REGION Network 5: Trạng thái cân Ag4
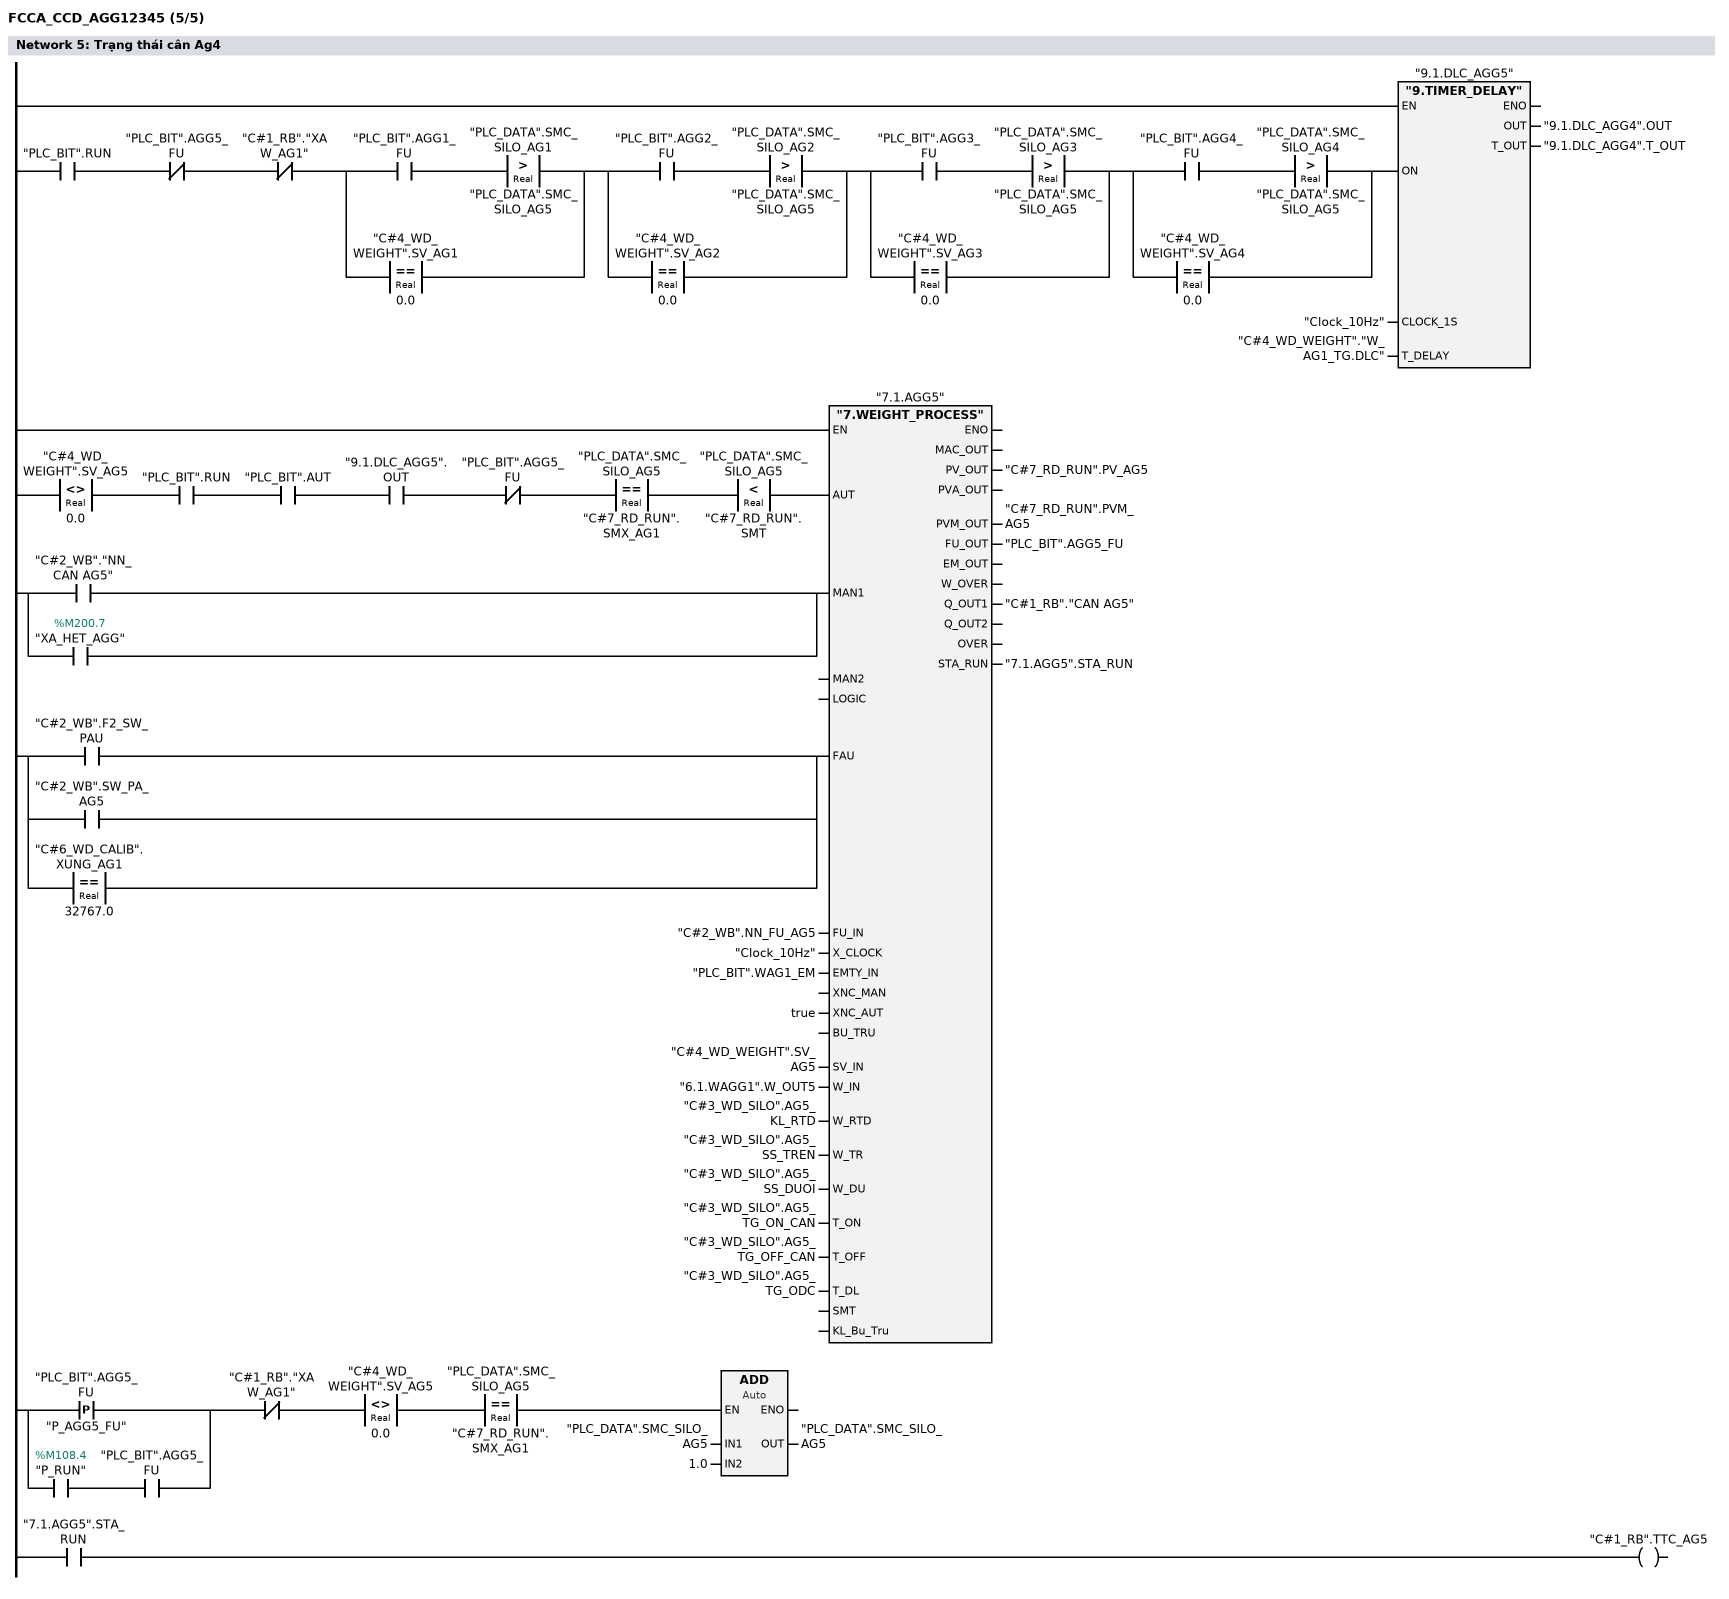
   RUNG wire#powerrail
      "9.1.DLC_AGG5"(ON := wire#w5, CLOCK_1S := "Clock_10Hz", T_DELAY := "C#4_WD_WEIGHT"."W_AG1_TG.DLC", OUT => "9.1.DLC_AGG4".OUT, T_OUT => "9.1.DLC_AGG4".T_OUT)
   END_RUNG
   RUNG wire#powerrail
      Contact( "PLC_BIT".RUN )
      I_Contact( "PLC_BIT".AGG5_FU )
      I_Contact( "C#1_RB"."XA W_AG1" )
      wire#w1
      Contact( "PLC_BIT".AGG1_FU )
      { S7_Templates := "SrcType := Real" } GT_Contact(in1 := "PLC_DATA".SMC_SILO_AG1, in2 := "PLC_DATA".SMC_SILO_AG5)
      wire#w2
      Contact( "PLC_BIT".AGG2_FU )
      { S7_Templates := "SrcType := Real" } GT_Contact(in1 := "PLC_DATA".SMC_SILO_AG2, in2 := "PLC_DATA".SMC_SILO_AG5)
      wire#w3
      Contact( "PLC_BIT".AGG3_FU )
      { S7_Templates := "SrcType := Real" } GT_Contact(in1 := "PLC_DATA".SMC_SILO_AG3, in2 := "PLC_DATA".SMC_SILO_AG5)
      wire#w4
      Contact( "PLC_BIT".AGG4_FU )
      { S7_Templates := "SrcType := Real" } GT_Contact(in1 := "PLC_DATA".SMC_SILO_AG4, in2 := "PLC_DATA".SMC_SILO_AG5)
   END_RUNG wire#w5
   RUNG wire#w1
      { S7_Templates := "SrcType := Real" } EQ_Contact(in1 := "C#4_WD_WEIGHT".SV_AG1, in2 := 0.0)
   END_RUNG wire#w2
   RUNG wire#w2
      { S7_Templates := "SrcType := Real" } EQ_Contact(in1 := "C#4_WD_WEIGHT".SV_AG2, in2 := 0.0)
   END_RUNG wire#w3
   RUNG wire#w3
      { S7_Templates := "SrcType := Real" } EQ_Contact(in1 := "C#4_WD_WEIGHT".SV_AG3, in2 := 0.0)
   END_RUNG wire#w4
   RUNG wire#w4
      { S7_Templates := "SrcType := Real" } EQ_Contact(in1 := "C#4_WD_WEIGHT".SV_AG4, in2 := 0.0)
   END_RUNG wire#w5
   RUNG wire#powerrail
      "7.1.AGG5"(AUT := wire#w6, MAN1 := wire#w7, FAU := wire#w8, MAN2 :=, LOGIC :=, FU_IN := "C#2_WB".NN_FU_AG5, X_CLOCK := "Clock_10Hz", EMTY_IN := "PLC_BIT".WAG1_EM, XNC_MAN :=, XNC_AUT := true, BU_TRU :=, SV_IN := "C#4_WD_WEIGHT".SV_AG5, W_IN := "6.1.WAGG1".W_OUT5, W_RTD := "C#3_WD_SILO".AG5_KL_RTD, W_TR := "C#3_WD_SILO".AG5_SS_TREN, W_DU := "C#3_WD_SILO".AG5_SS_DUOI, T_ON := "C#3_WD_SILO".AG5_TG_ON_CAN, T_OFF := "C#3_WD_SILO".AG5_TG_OFF_CAN, T_DL := "C#3_WD_SILO".AG5_TG_ODC, SMT :=, KL_Bu_Tru :=, MAC_OUT =>, PV_OUT => "C#7_RD_RUN".PV_AG5, PVA_OUT =>, PVM_OUT => "C#7_RD_RUN".PVM_AG5, FU_OUT => "PLC_BIT".AGG5_FU, EM_OUT =>, W_OVER =>, Q_OUT1 => "C#1_RB"."CAN AG5", Q_OUT2 =>, OVER =>, STA_RUN => "7.1.AGG5".STA_RUN)
   END_RUNG
   RUNG wire#powerrail
      { S7_Templates := "SrcType := Real" } NE_Contact(in1 := "C#4_WD_WEIGHT".SV_AG5, in2 := 0.0)
      Contact( "PLC_BIT".RUN )
      Contact( "PLC_BIT".AUT )
      Contact( "9.1.DLC_AGG5".OUT )
      I_Contact( "PLC_BIT".AGG5_FU )
      { S7_Templates := "SrcType := Real" } EQ_Contact(in1 := "PLC_DATA".SMC_SILO_AG5, in2 := "C#7_RD_RUN".SMX_AG1)
      { S7_Templates := "SrcType := Real" } LT_Contact(in1 := "PLC_DATA".SMC_SILO_AG5, in2 := "C#7_RD_RUN".SMT)
   END_RUNG wire#w6
   RUNG wire#powerrail
      Contact( "C#2_WB"."NN_CAN AG5" )
   END_RUNG wire#w7
   RUNG wire#powerrail
      Contact( "XA_HET_AGG" )
   END_RUNG wire#w7
   RUNG wire#powerrail
      Contact( "C#2_WB".F2_SW_PAU )
   END_RUNG wire#w8
   RUNG wire#powerrail
      Contact( "C#2_WB".SW_PA_AG5 )
   END_RUNG wire#w8
   RUNG wire#powerrail
      { S7_Templates := "SrcType := Real" } EQ_Contact(in1 := "C#6_WD_CALIB".XUNG_AG1, in2 := 32767.0)
   END_RUNG wire#w8
   RUNG wire#powerrail
      P_Contact(operand := "PLC_BIT".AGG5_FU, bit := "P_AGG5_FU")
      wire#w9
      I_Contact( "C#1_RB"."XA W_AG1" )
      { S7_Templates := "SrcType := Real" } NE_Contact(in1 := "C#4_WD_WEIGHT".SV_AG5, in2 := 0.0)
      { S7_Templates := "SrcType := Real" } EQ_Contact(in1 := "PLC_DATA".SMC_SILO_AG5, in2 := "C#7_RD_RUN".SMX_AG1)
      Add(in1 := "PLC_DATA".SMC_SILO_AG5, in2 := 1.0, out => "PLC_DATA".SMC_SILO_AG5)
   END_RUNG
   RUNG wire#powerrail
      Contact( "P_RUN" )
      Contact( "PLC_BIT".AGG5_FU )
   END_RUNG wire#w9
   RUNG wire#powerrail
      Contact( "7.1.AGG5".STA_RUN )
      Coil( "C#1_RB".TTC_AG5 )
   END_RUNG
   // the same network as SCL:
   "9.1.DLC_AGG5"(ON := "PLC_BIT".RUN AND NOT "PLC_BIT".AGG5_FU AND NOT "C#1_RB"."XA W_AG1" AND (("PLC_BIT".AGG1_FU AND ("PLC_DATA".SMC_SILO_AG1 > "PLC_DATA".SMC_SILO_AG5)) OR ("C#4_WD_WEIGHT".SV_AG1 = 0.0)) AND (("PLC_BIT".AGG2_FU AND ("PLC_DATA".SMC_SILO_AG2 > "PLC_DATA".SMC_SILO_AG5)) OR ("C#4_WD_WEIGHT".SV_AG2 = 0.0)) AND (("PLC_BIT".AGG3_FU AND ("PLC_DATA".SMC_SILO_AG3 > "PLC_DATA".SMC_SILO_AG5)) OR ("C#4_WD_WEIGHT".SV_AG3 = 0.0)) AND (("PLC_BIT".AGG4_FU AND ("PLC_DATA".SMC_SILO_AG4 > "PLC_DATA".SMC_SILO_AG5)) OR ("C#4_WD_WEIGHT".SV_AG4 = 0.0)),   // "9.TIMER_DELAY"
                  CLOCK_1S := "Clock_10Hz",
                  T_DELAY := "C#4_WD_WEIGHT"."W_AG1_TG.DLC",
                  OUT => "9.1.DLC_AGG4".OUT,
                  T_OUT => "9.1.DLC_AGG4".T_OUT);
   "7.1.AGG5"(AUT := ("C#4_WD_WEIGHT".SV_AG5 <> 0.0) AND "PLC_BIT".RUN AND "PLC_BIT".AUT AND "9.1.DLC_AGG5".OUT AND NOT "PLC_BIT".AGG5_FU AND ("PLC_DATA".SMC_SILO_AG5 = "C#7_RD_RUN".SMX_AG1) AND ("PLC_DATA".SMC_SILO_AG5 < "C#7_RD_RUN".SMT),   // "7.WEIGHT_PROCESS"
              MAN1 := "C#2_WB"."NN_CAN AG5" OR "XA_HET_AGG",
              FAU := "C#2_WB".F2_SW_PAU OR "C#2_WB".SW_PA_AG5 OR ("C#6_WD_CALIB".XUNG_AG1 = 32767.0),
              FU_IN := "C#2_WB".NN_FU_AG5,
              X_CLOCK := "Clock_10Hz",
              EMTY_IN := "PLC_BIT".WAG1_EM,
              XNC_AUT := true,
              SV_IN := "C#4_WD_WEIGHT".SV_AG5,
              W_IN := "6.1.WAGG1".W_OUT5,
              W_RTD := "C#3_WD_SILO".AG5_KL_RTD,
              W_TR := "C#3_WD_SILO".AG5_SS_TREN,
              W_DU := "C#3_WD_SILO".AG5_SS_DUOI,
              T_ON := "C#3_WD_SILO".AG5_TG_ON_CAN,
              T_OFF := "C#3_WD_SILO".AG5_TG_OFF_CAN,
              T_DL := "C#3_WD_SILO".AG5_TG_ODC,
              PV_OUT => "C#7_RD_RUN".PV_AG5,
              PVM_OUT => "C#7_RD_RUN".PVM_AG5,
              FU_OUT => "PLC_BIT".AGG5_FU,
              Q_OUT1 => "C#1_RB"."CAN AG5",
              STA_RUN => "7.1.AGG5".STA_RUN);
   #_w1 := "PLC_BIT".AGG5_FU AND NOT "P_AGG5_FU";   // rising edge of "PLC_BIT".AGG5_FU
   "P_AGG5_FU" := "PLC_BIT".AGG5_FU;
   IF (#_w1 OR ("P_RUN" AND "PLC_BIT".AGG5_FU)) AND NOT "C#1_RB"."XA W_AG1" AND ("C#4_WD_WEIGHT".SV_AG5 <> 0.0) AND ("PLC_DATA".SMC_SILO_AG5 = "C#7_RD_RUN".SMX_AG1) THEN
       "PLC_DATA".SMC_SILO_AG5 := "PLC_DATA".SMC_SILO_AG5 + 1.0;
   END_IF;
   "C#1_RB".TTC_AG5 := "7.1.AGG5".STA_RUN;
END_REGION
END_FUNCTION

FUNCTION_BLOCK "7.WEIGHT_PROCESS"   // FB7, LAD
{ S7_Optimized_Access := 'TRUE' }
VERSION : 0.1
// Chú ý:
// W_DU: nhập khối lượng giớ hạn dưới để tính SS_DUOI sai số dưới, ví dụ SV_IN cài là 1000kg, giới hạn dưới cài là W_DU=55kg, vì KL_BU=0.0 nên> SS_DUOI=1000-55=945kg
// W_RTD: cài đặt khối lượng rơi tự do, từ đó tính điểm cắt Rơi tự do, ví dụ W_RTD=95kg, khi đó điểm cắt Rơi tự do KL_RTD=1000-95=905kg
// Thực tế khi đó: cân sẽ được cân thô đến điểm cắt RTD là 905kg thì nó sẽ bắt đầu chuyển sang Cân Tinh,
// stored: AutoNumber false, CodeModifiedDate 2026-01-04T10:59:07.612582Z, CompileDate 2026-01-04T14:27:04.4561281Z, CreationDate 2024-10-12T12:36:08.0193576Z, DownloadWithoutReinit false, HandleErrorsWithinBlock false, InterfaceModifiedDate 2024-08-06T09:13:34.3012657Z, IsConsistent true, IsIECCheckEnabled false, IsKnowHowProtected false, IsRetainMemResEnabled false, IsWriteProtected false, LibraryConformanceStatus Warning: The object contains access to global data blocks., MemoryReserve 100, ModifiedDate 2026-01-04T11:31:32.9722655Z, ParameterModified 2024-08-06T08:53:48.4792275Z, PLCSimAdvancedSupport false, SetENOAutomatically False, StructureModified 2024-08-06T09:13:34.3012657Z, UDAEnableTagReadback false
   VAR_INPUT
      AUT : Bool;
      MAN1 : Bool;
      MAN2 : Bool;
      LOGIC : Bool;
      FAU : Bool;   // Tạm dừng cân trong mode Auto
      FU_IN : Bool;   // Nút nhấn báo đầy Silo (phần mềm ghi xuống)
      X_CLOCK : Bool;
      EMTY_IN : Bool;   // Nút nhấn (hoặc tín hiệu trên phần mềm) báo cân rỗng
      XNC_MAN : Bool;
      XNC_AUT : Bool;
      BU_TRU : Bool;   // Nếu =false thì CAN_DƯ luôn bằng 0
      SV_IN : Real;
      W_IN : Real;   // Khối lượng cân hiện tại
      W_RTD : Real;   // Khối lựng rơi tự do
      W_TR : Real;   // KL giới hạn trên
      W_DU : Real;   // KL giới hạn dưới
      T_ON : Real;   // Thời gian cân mở
      T_OFF : Real;   // Thời gian cân đóng
      T_DL : Real;   // Thời gian đợi rơi thêm
      SMT : Real;
      KL_Bu_Tru : Real;   // >0.0 là bù chủ động vào KL_BU, ngược lại sẽ dùng CAN DƯ
   END_VAR
   VAR_OUTPUT
      MAC_OUT : Real;
      PV_OUT : Real;
      PVA_OUT : Real;
      PVM_OUT : Real;
      FU_OUT : Bool;   // Báo cân đầy
      EM_OUT : Bool;
      W_OVER : Real;
      Q_OUT1 : Bool;
      Q_OUT2 : Bool;
      OVER : Bool;
      STA_RUN : Bool;
   END_VAR
   VAR RETAIN
      FU { ExternalAccessible := 'False'; ExternalVisible := 'False'; ExternalWritable := 'False'} : Bool;   // Bít nhớ báo cân đầy
      EM { ExternalAccessible := 'False'; ExternalVisible := 'False'; ExternalWritable := 'False'} : Bool;
      "CAN DU" { ExternalAccessible := 'False'; ExternalVisible := 'False'; ExternalWritable := 'False'} : Real;   // Nếu BU_TRU=false thì CAN_DU luôn =0
      PVA { ExternalAccessible := 'False'; ExternalVisible := 'False'; ExternalWritable := 'False'} : Real;
      PVM { ExternalAccessible := 'False'; ExternalVisible := 'False'; ExternalWritable := 'False'} : Real;
      TOFF { ExternalAccessible := 'False'; ExternalVisible := 'False'; ExternalWritable := 'False'} : Real;
      TON { ExternalAccessible := 'False'; ExternalVisible := 'False'; ExternalWritable := 'False'} : Real;
      T_DLFULL { ExternalAccessible := 'False'; ExternalVisible := 'False'; ExternalWritable := 'False'} : Real;   // Đếm thời gian báo đầy
      "T_DLT/T" { ExternalAccessible := 'False'; ExternalVisible := 'False'; ExternalWritable := 'False'} : Real;   // Đếm thời gian cho lượng rơi thêm
      KL_BU : Real;   // Nhập băng KL_tru_bu hoặc nếu cân bị Cân Dư
      CLK_DLE { ExternalAccessible := 'False'; ExternalVisible := 'False'; ExternalWritable := 'False'} : Bool;
      CLK_DLF { ExternalAccessible := 'False'; ExternalVisible := 'False'; ExternalWritable := 'False'} : Bool;
      "CLK_DLT/T" { ExternalAccessible := 'False'; ExternalVisible := 'False'; ExternalWritable := 'False'} : Bool;
      CLK_TT { ExternalAccessible := 'False'; ExternalVisible := 'False'; ExternalWritable := 'False'} : Bool;
      "TEMP_T/T" { ExternalAccessible := 'False'; ExternalVisible := 'False'; ExternalWritable := 'False'} : Bool;   // Hết thời gian đóng cân ==> mở cân
      "RUN_T/T" { ExternalAccessible := 'False'; ExternalVisible := 'False'; ExternalWritable := 'False'} : Bool;   // Bật chạy thô tinh sau khi hết thời gian đợi rơi thêm
   END_VAR
   VAR
      RUN_MAN : Bool;
      RUN_AUT : Bool;
      "CUA_T/T" : Bool;
      P_OUT1 : Bool;
      P_OUT2 : Bool;
      P_EMTY : Bool;
      P_FU : Bool;
   END_VAR
   VAR_TEMP
      "SS TREN" : Real;
      "SS DUOI" : Real;
      "KL RTD" : Real;   // Điểm cắt Rơi tự do
   END_VAR
   VAR_TEMP   // added for the SCL form of the ladder/FBD networks
      _w1 : Bool;
      _w2 : Bool;
      _w3 : Bool;
   END_VAR
BEGIN

REGION Network 1: MOVE MAC
   // Nếu BU_TRU=false thì CAN_Du luôn bằng 0, khi đó nếu KL_Bu_Tru không được nhập thì KL_BU luôn =0.0
   // Thực tế trong chưng trình này, các điều kiện đang khiến CAN_DU=0.0 và KL_BU=0.0
   // Khi đó SS_DUOI=SV_IN - W_DU
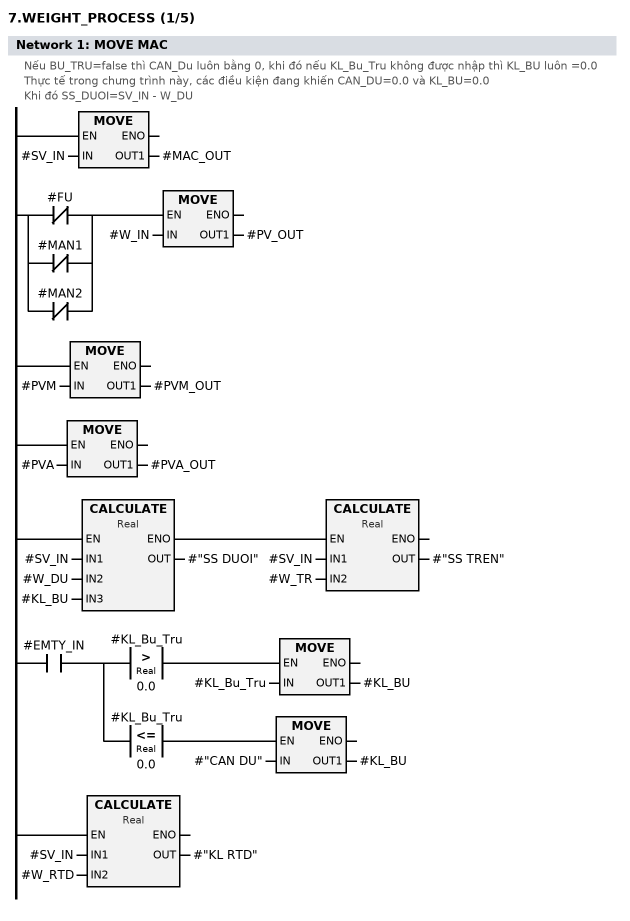
   RUNG wire#powerrail
      Move(in := #SV_IN, out1 => #MAC_OUT)
   END_RUNG
   RUNG wire#powerrail
      I_Contact( #FU )
      wire#w1
      Move(in := #W_IN, out1 => #PV_OUT)
   END_RUNG
   RUNG wire#powerrail
      I_Contact( #MAN1 )
   END_RUNG wire#w1
   RUNG wire#powerrail
      I_Contact( #MAN2 )
   END_RUNG wire#w1
   RUNG wire#powerrail
      Move(in := #PVM, out1 => #PVM_OUT)
   END_RUNG
   RUNG wire#powerrail
      Move(in := #PVA, out1 => #PVA_OUT)
   END_RUNG
   RUNG wire#powerrail
      { S7_Templates := "SrcType := Real"; S7_Expression := "IN1-IN2-IN3" } Calculate(in1 := #SV_IN, in2 := #W_DU, in3 := #KL_BU, out => #"SS DUOI")
      { S7_Templates := "SrcType := Real"; S7_Expression := "IN1+IN2" } Calculate(in1 := #SV_IN, in2 := #W_TR, out => #"SS TREN")
   END_RUNG
   RUNG wire#powerrail
      Contact( #EMTY_IN )
      wire#w2
      { S7_Templates := "SrcType := Real" } GT_Contact(in1 := #KL_Bu_Tru, in2 := 0.0)
      Move(in := #KL_Bu_Tru, out1 => #KL_BU)
   END_RUNG
   RUNG wire#w2
      { S7_Templates := "SrcType := Real" } LE_Contact(in1 := #KL_Bu_Tru, in2 := 0.0)
      Move(in := #"CAN DU", out1 => #KL_BU)
   END_RUNG
   RUNG wire#powerrail
      { S7_Templates := "SrcType := Real"; S7_Expression := "IN1-IN2" } Calculate(in1 := #SV_IN, in2 := #W_RTD, out => #"KL RTD")
   END_RUNG
   // the same network as SCL:
   #MAC_OUT := #SV_IN;
   IF NOT #FU OR NOT #MAN1 OR NOT #MAN2 THEN #PV_OUT := #W_IN; END_IF;
   #PVM_OUT := #PVM;
   #PVA_OUT := #PVA;
   #"SS DUOI" := #SV_IN-#W_DU-#KL_BU;
   #"SS TREN" := #SV_IN+#W_TR;
   IF #EMTY_IN AND (#KL_Bu_Tru > 0.0) THEN #KL_BU := #KL_Bu_Tru; END_IF;
   IF #EMTY_IN AND (#KL_Bu_Tru <= 0.0) THEN #KL_BU := #"CAN DU"; END_IF;
   #"KL RTD" := #SV_IN-#W_RTD;
END_REGION

REGION Network 2: KHOI LUONG CAN DU
   // Tính lượng CAN DƯ, khi cân FU, nếu vì lý do nào đó mà W_IN tiếp tục tăng, túc cân tiếp tục được nạp, thì  giá trị Dư đó xẽ được lưu lại vào biến #CAN DU
   // Báo tràn OVER: trong chế độ AUTO, nếu W_IN lớn hơn SS TRÊN sẽ báo tràn, khi bật FU_OUT thì không kích báo tràn tiếp được
   // Nhưng OVER này được giữ, nó chỉ bị reset khi xả cân, khi đó W_IN nhỏ hơn SS_TREN
   // W_OVER chính là lượng cân dư
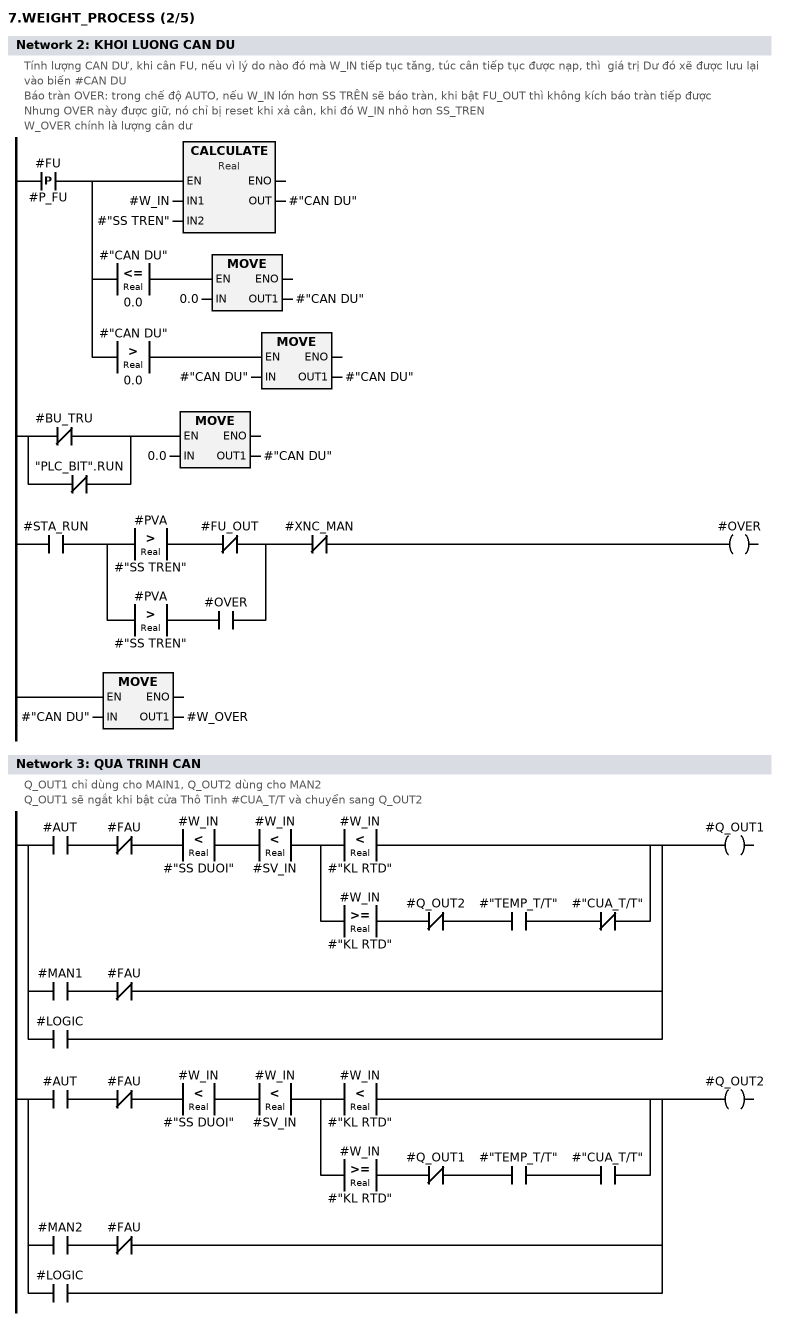
   RUNG wire#powerrail
      P_Contact(operand := #FU, bit := #P_FU)
      wire#w1
      { S7_Templates := "SrcType := Real"; S7_Expression := "IN1-IN2" } Calculate(in1 := #W_IN, in2 := #"SS TREN", out => #"CAN DU")
   END_RUNG
   RUNG wire#w1
      { S7_Templates := "SrcType := Real" } LE_Contact(in1 := #"CAN DU", in2 := 0.0)
      Move(in := 0.0, out1 => #"CAN DU")
   END_RUNG
   RUNG wire#w1
      { S7_Templates := "SrcType := Real" } GT_Contact(in1 := #"CAN DU", in2 := 0.0)
      Move(in := #"CAN DU", out1 => #"CAN DU")
   END_RUNG
   RUNG wire#powerrail
      I_Contact( #BU_TRU )
      wire#w2
      Move(in := 0.0, out1 => #"CAN DU")
   END_RUNG
   RUNG wire#powerrail
      I_Contact( "PLC_BIT".RUN )
   END_RUNG wire#w2
   RUNG wire#powerrail
      Contact( #STA_RUN )
      wire#w3
      { S7_Templates := "SrcType := Real" } GT_Contact(in1 := #PVA, in2 := #"SS TREN")
      I_Contact( #FU_OUT )
      wire#w4
      I_Contact( #XNC_MAN )
      Coil( #OVER )
   END_RUNG
   RUNG wire#w3
      { S7_Templates := "SrcType := Real" } GT_Contact(in1 := #PVA, in2 := #"SS TREN")
      Contact( #OVER )
   END_RUNG wire#w4
   RUNG wire#powerrail
      Move(in := #"CAN DU", out1 => #W_OVER)
   END_RUNG
   // the same network as SCL:
   #_w1 := #FU AND NOT #P_FU;   // rising edge of #FU
   #P_FU := #FU;
   IF #_w1 THEN #"CAN DU" := #W_IN-#"SS TREN"; END_IF;
   IF #_w1 AND (#"CAN DU" <= 0.0) THEN #"CAN DU" := 0.0; END_IF;
   IF #_w1 AND (#"CAN DU" > 0.0) THEN #"CAN DU" := #"CAN DU"; END_IF;
   IF NOT #BU_TRU OR NOT "PLC_BIT".RUN THEN #"CAN DU" := 0.0; END_IF;
   #OVER := #STA_RUN AND (((#PVA > #"SS TREN") AND NOT #FU_OUT) OR ((#PVA > #"SS TREN") AND #OVER)) AND NOT #XNC_MAN;
   #W_OVER := #"CAN DU";
END_REGION

REGION Network 3: QUA TRINH CAN
   // Q_OUT1 chỉ dùng cho MAIN1, Q_OUT2 dùng cho MAN2
   // Q_OUT1 sẽ ngắt khi bật cửa Thô Tinh #CUA_T/T và chuyển sang Q_OUT2
   RUNG wire#powerrail
      Contact( #AUT )
      I_Contact( #FAU )
      { S7_Templates := "SrcType := Real" } LT_Contact(in1 := #W_IN, in2 := #"SS DUOI")
      { S7_Templates := "SrcType := Real" } LT_Contact(in1 := #W_IN, in2 := #SV_IN)
      wire#w1
      { S7_Templates := "SrcType := Real" } LT_Contact(in1 := #W_IN, in2 := #"KL RTD")
      wire#w2
      Coil( #Q_OUT1 )
   END_RUNG
   RUNG wire#w1
      { S7_Templates := "SrcType := Real" } GE_Contact(in1 := #W_IN, in2 := #"KL RTD")
      I_Contact( #Q_OUT2 )
      Contact( #"TEMP_T/T" )
      I_Contact( #"CUA_T/T" )
   END_RUNG wire#w2
   RUNG wire#powerrail
      Contact( #MAN1 )
      I_Contact( #FAU )
   END_RUNG wire#w2
   RUNG wire#powerrail
      Contact( #LOGIC )
   END_RUNG wire#w2
   RUNG wire#powerrail
      Contact( #AUT )
      I_Contact( #FAU )
      { S7_Templates := "SrcType := Real" } LT_Contact(in1 := #W_IN, in2 := #"SS DUOI")
      { S7_Templates := "SrcType := Real" } LT_Contact(in1 := #W_IN, in2 := #SV_IN)
      wire#w3
      { S7_Templates := "SrcType := Real" } LT_Contact(in1 := #W_IN, in2 := #"KL RTD")
      wire#w4
      Coil( #Q_OUT2 )
   END_RUNG
   RUNG wire#w3
      { S7_Templates := "SrcType := Real" } GE_Contact(in1 := #W_IN, in2 := #"KL RTD")
      I_Contact( #Q_OUT1 )
      Contact( #"TEMP_T/T" )
      Contact( #"CUA_T/T" )
   END_RUNG wire#w4
   RUNG wire#powerrail
      Contact( #MAN2 )
      I_Contact( #FAU )
   END_RUNG wire#w4
   RUNG wire#powerrail
      Contact( #LOGIC )
   END_RUNG wire#w4
   // the same network as SCL:
   #Q_OUT1 := (#AUT AND NOT #FAU AND (#W_IN < #"SS DUOI") AND (#W_IN < #SV_IN) AND ((#W_IN < #"KL RTD") OR ((#W_IN >= #"KL RTD") AND NOT #Q_OUT2 AND #"TEMP_T/T" AND NOT #"CUA_T/T"))) OR (#MAN1 AND NOT #FAU) OR #LOGIC;
   #Q_OUT2 := (#AUT AND NOT #FAU AND (#W_IN < #"SS DUOI") AND (#W_IN < #SV_IN) AND ((#W_IN < #"KL RTD") OR ((#W_IN >= #"KL RTD") AND NOT #Q_OUT1 AND #"TEMP_T/T" AND #"CUA_T/T"))) OR (#MAN2 AND NOT #FAU) OR #LOGIC;
END_REGION

REGION Network 4: CHIA PV
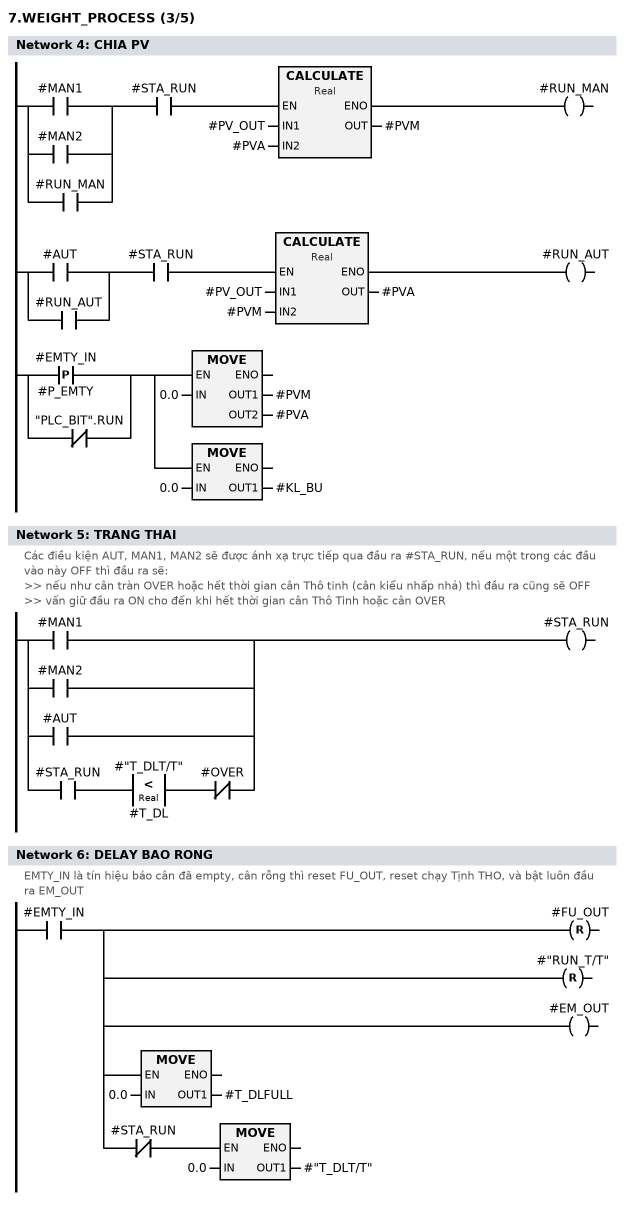
   RUNG wire#powerrail
      Contact( #MAN1 )
      wire#w1
      Contact( #STA_RUN )
      { S7_Templates := "SrcType := Real"; S7_Expression := "IN1-IN2" } Calculate(in1 := #PV_OUT, in2 := #PVA, out => #PVM)
      Coil( #RUN_MAN )
   END_RUNG
   RUNG wire#powerrail
      Contact( #MAN2 )
   END_RUNG wire#w1
   RUNG wire#powerrail
      Contact( #RUN_MAN )
   END_RUNG wire#w1
   RUNG wire#powerrail
      Contact( #AUT )
      wire#w2
      Contact( #STA_RUN )
      { S7_Templates := "SrcType := Real"; S7_Expression := "IN1-IN2" } Calculate(in1 := #PV_OUT, in2 := #PVM, out => #PVA)
      Coil( #RUN_AUT )
   END_RUNG
   RUNG wire#powerrail
      Contact( #RUN_AUT )
   END_RUNG wire#w2
   RUNG wire#powerrail
      P_Contact(operand := #EMTY_IN, bit := #P_EMTY)
      wire#w3
      Move(in := 0.0, out1 => #PVM, out2 => #PVA)
   END_RUNG
   RUNG wire#powerrail
      I_Contact( "PLC_BIT".RUN )
   END_RUNG wire#w3
   RUNG wire#w3
      Move(in := 0.0, out1 => #KL_BU)
   END_RUNG
   // the same network as SCL:
   #_w1 := (#MAN1 OR #MAN2 OR #RUN_MAN) AND #STA_RUN;
   IF #_w1 THEN #PVM := #PV_OUT-#PVA; END_IF;
   #RUN_MAN := #_w1;
   #_w2 := (#AUT OR #RUN_AUT) AND #STA_RUN;
   IF #_w2 THEN #PVA := #PV_OUT-#PVM; END_IF;
   #RUN_AUT := #_w2;
   #_w3 := #EMTY_IN AND NOT #P_EMTY;   // rising edge of #EMTY_IN
   #P_EMTY := #EMTY_IN;
   IF #_w3 OR NOT "PLC_BIT".RUN THEN
       #PVM := 0.0;
       #PVA := 0.0;
       #KL_BU := 0.0;
   END_IF;
END_REGION

REGION Network 5: TRANG THAI
   // Các điều kiện AUT, MAN1, MAN2 sẽ được ánh xạ trực tiếp qua đầu ra #STA_RUN, nếu một trong các đầu vào này OFF thì đầu ra sẽ:
   // >> nếu như cân tràn OVER hoặc hết thời gian cân Thô tinh (cân kiểu nhấp nhả) thì đầu ra cũng sẽ OFF
   // >> vấn giữ đầu ra ON cho đến khi hết thời gian cân Thô Tinh hoặc cân OVER
   RUNG wire#powerrail
      Contact( #MAN1 )
      wire#w1
      Coil( #STA_RUN )
   END_RUNG
   RUNG wire#powerrail
      Contact( #MAN2 )
   END_RUNG wire#w1
   RUNG wire#powerrail
      Contact( #AUT )
   END_RUNG wire#w1
   RUNG wire#powerrail
      Contact( #STA_RUN )
      { S7_Templates := "SrcType := Real" } LT_Contact(in1 := #"T_DLT/T", in2 := #T_DL)
      I_Contact( #OVER )
   END_RUNG wire#w1
   // the same network as SCL:
   #STA_RUN := #MAN1 OR #MAN2 OR #AUT OR (#STA_RUN AND (#"T_DLT/T" < #T_DL) AND NOT #OVER);
END_REGION

REGION Network 6: DELAY BAO RONG
   // EMTY_IN là tín hiệu báo cân đã empty, cân rỗng thì reset FU_OUT, reset chạy Tịnh THO, và bật luôn đầu ra EM_OUT
   RUNG wire#powerrail
      Contact( #EMTY_IN )
      wire#w1
      R_Coil( #FU_OUT )
   END_RUNG
   RUNG wire#w1
      R_Coil( #"RUN_T/T" )
   END_RUNG
   RUNG wire#w1
      Coil( #EM_OUT )
   END_RUNG
   RUNG wire#w1
      Move(in := 0.0, out1 => #T_DLFULL)
   END_RUNG
   RUNG wire#w1
      I_Contact( #STA_RUN )
      Move(in := 0.0, out1 => #"T_DLT/T")
   END_RUNG
   // the same network as SCL:
   IF #EMTY_IN THEN
       #FU_OUT := FALSE;
       #"RUN_T/T" := FALSE;
   END_IF;
   #EM_OUT := #EMTY_IN;
   IF #EMTY_IN THEN #T_DLFULL := 0.0; END_IF;
   IF #EMTY_IN AND NOT #STA_RUN THEN #"T_DLT/T" := 0.0; END_IF;
END_REGION

REGION Network 7: DELAY BAO DAY
   // Khi khối lượng đầu vào vượt qua sai số dưới, thì bắt đầu đếm để tình thời gian Delay trước khi báo FU
   // nếu thời gian đếm nó vượt qua giá trị cài đặt (cũng chính là thời gian đợi chơ lượng rơi thêm), thì SET ngõ ra #FU_OUT
   // 
   // Chú ý: chế độ MAN thì nó không báo FU
   // Cân FULL khi giá trị cân nó vượt qua SS_DUOI rồi đợi thêm một khoảng thời gian rơi thêm
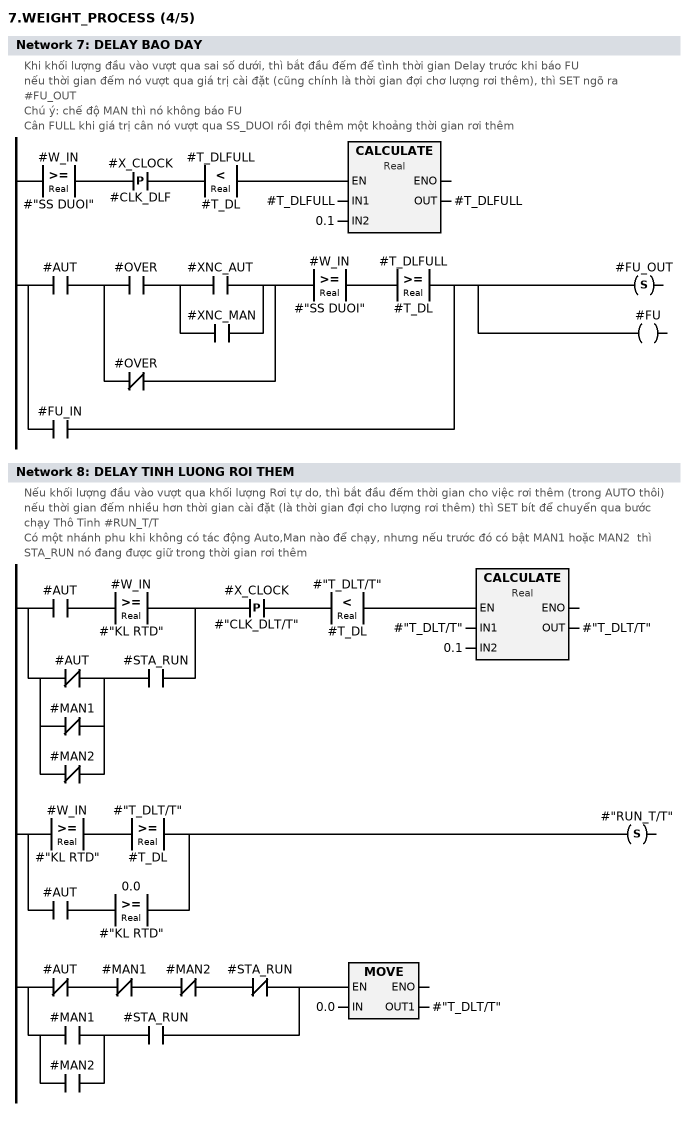
   RUNG wire#powerrail
      { S7_Templates := "SrcType := Real" } GE_Contact(in1 := #W_IN, in2 := #"SS DUOI")
      P_Contact(operand := #X_CLOCK, bit := #CLK_DLF)
      { S7_Templates := "SrcType := Real" } LT_Contact(in1 := #T_DLFULL, in2 := #T_DL)
      { S7_Templates := "SrcType := Real"; S7_Expression := "IN1+IN2" } Calculate(in1 := #T_DLFULL, in2 := 0.1, out => #T_DLFULL)
   END_RUNG
   RUNG wire#powerrail
      Contact( #AUT )
      wire#w1
      Contact( #OVER )
      wire#w2
      Contact( #XNC_AUT )
      wire#w3
      { S7_Templates := "SrcType := Real" } GE_Contact(in1 := #W_IN, in2 := #"SS DUOI")
      { S7_Templates := "SrcType := Real" } GE_Contact(in1 := #T_DLFULL, in2 := #T_DL)
      wire#w4
      S_Coil( #FU_OUT )
   END_RUNG
   RUNG wire#w2
      Contact( #XNC_MAN )
   END_RUNG wire#w3
   RUNG wire#w1
      I_Contact( #OVER )
   END_RUNG wire#w3
   RUNG wire#powerrail
      Contact( #FU_IN )
   END_RUNG wire#w4
   RUNG wire#w4
      Coil( #FU )
   END_RUNG
   // the same network as SCL:
   #_w1 := (#W_IN >= #"SS DUOI") AND #X_CLOCK AND NOT #CLK_DLF;   // rising edge of #X_CLOCK
   #CLK_DLF := #X_CLOCK;
   IF #_w1 AND (#T_DLFULL < #T_DL) THEN #T_DLFULL := #T_DLFULL+0.1; END_IF;
   #_w2 := (#AUT AND ((#OVER AND (#XNC_AUT OR #XNC_MAN)) OR NOT #OVER) AND (#W_IN >= #"SS DUOI") AND (#T_DLFULL >= #T_DL)) OR #FU_IN;
   IF #_w2 THEN #FU_OUT := TRUE; END_IF;
   #FU := #_w2;
END_REGION

REGION Network 8: DELAY TINH LUONG ROI THEM
   // Nếu khối lượng đầu vào vượt qua khối lượng Rơi tự do, thì bắt đầu đếm thời gian cho việc rơi thêm (trong AUTO thôi)
   // nếu thời gian đếm nhiều hơn thời gian cài đặt (là thời gian đợi cho lượng rơi thêm) thì SET bít để chuyển qua bước chạy Thô Tinh #RUN_T/T
   // 
   // Có một nhánh phu khi không có tác động Auto,Man nào để chạy, nhưng nếu trước đó có bật MAN1 hoặc MAN2  thì STA_RUN nó đang được giữ trong thời gian rơi thêm
   RUNG wire#powerrail
      Contact( #AUT )
      { S7_Templates := "SrcType := Real" } GE_Contact(in1 := #W_IN, in2 := #"KL RTD")
      wire#w1
      P_Contact(operand := #X_CLOCK, bit := #"CLK_DLT/T")
      { S7_Templates := "SrcType := Real" } LT_Contact(in1 := #"T_DLT/T", in2 := #T_DL)
      { S7_Templates := "SrcType := Real"; S7_Expression := "IN1+IN2" } Calculate(in1 := #"T_DLT/T", in2 := 0.1, out => #"T_DLT/T")
   END_RUNG
   RUNG wire#powerrail
      I_Contact( #AUT )
      wire#w2
      Contact( #STA_RUN )
   END_RUNG wire#w1
   RUNG wire#powerrail
      I_Contact( #MAN1 )
   END_RUNG wire#w2
   RUNG wire#powerrail
      I_Contact( #MAN2 )
   END_RUNG wire#w2
   RUNG wire#powerrail
      { S7_Templates := "SrcType := Real" } GE_Contact(in1 := #W_IN, in2 := #"KL RTD")
      { S7_Templates := "SrcType := Real" } GE_Contact(in1 := #"T_DLT/T", in2 := #T_DL)
      wire#w3
      S_Coil( #"RUN_T/T" )
   END_RUNG
   RUNG wire#powerrail
      Contact( #AUT )
      { S7_Templates := "SrcType := Real" } GE_Contact(in1 := 0.0, in2 := #"KL RTD")
   END_RUNG wire#w3
   RUNG wire#powerrail
      I_Contact( #AUT )
      I_Contact( #MAN1 )
      I_Contact( #MAN2 )
      I_Contact( #STA_RUN )
      wire#w4
      Move(in := 0.0, out1 => #"T_DLT/T")
   END_RUNG
   RUNG wire#powerrail
      Contact( #MAN1 )
      wire#w5
      Contact( #STA_RUN )
   END_RUNG wire#w4
   RUNG wire#powerrail
      Contact( #MAN2 )
   END_RUNG wire#w5
   // the same network as SCL:
   #_w1 := ((#AUT AND (#W_IN >= #"KL RTD")) OR ((NOT #AUT OR NOT #MAN1 OR NOT #MAN2) AND #STA_RUN)) AND #X_CLOCK AND NOT #"CLK_DLT/T";   // rising edge of #X_CLOCK
   #"CLK_DLT/T" := #X_CLOCK;
   IF #_w1 AND (#"T_DLT/T" < #T_DL) THEN #"T_DLT/T" := #"T_DLT/T"+0.1; END_IF;
   IF ((#W_IN >= #"KL RTD") AND (#"T_DLT/T" >= #T_DL)) OR (#AUT AND (0.0 >= #"KL RTD")) THEN
       #"RUN_T/T" := TRUE;
   END_IF;
   IF (NOT #AUT AND NOT #MAN1 AND NOT #MAN2 AND NOT #STA_RUN) OR ((#MAN1 OR #MAN2) AND #STA_RUN) THEN
       #"T_DLT/T" := 0.0;
   END_IF;
END_REGION

REGION Network 9: CAN THO TINH
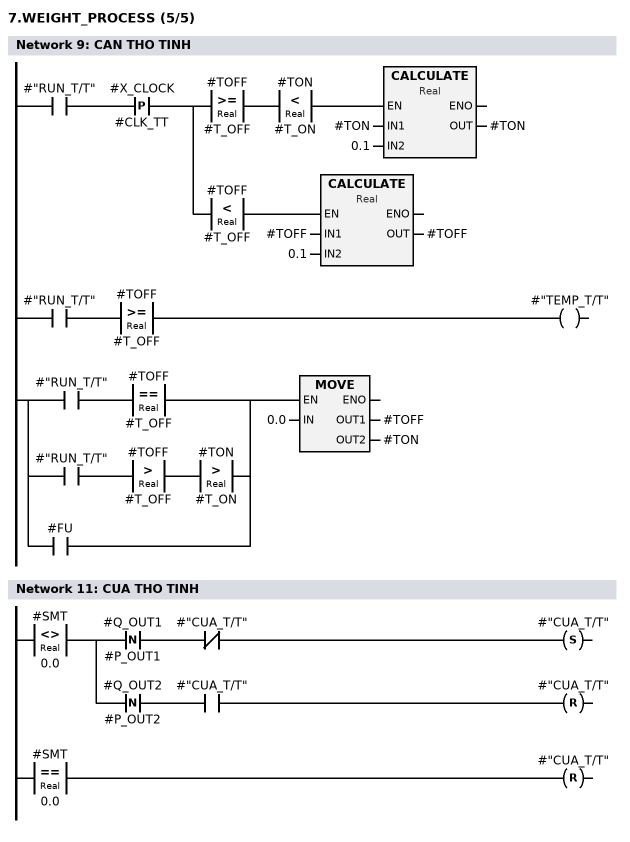
   RUNG wire#powerrail
      Contact( #"RUN_T/T" )
      P_Contact(operand := #X_CLOCK, bit := #CLK_TT)
      wire#w1
      { S7_Templates := "SrcType := Real" } GE_Contact(in1 := #TOFF, in2 := #T_OFF)
      { S7_Templates := "SrcType := Real" } LT_Contact(in1 := #TON, in2 := #T_ON)
      { S7_Templates := "SrcType := Real"; S7_Expression := "IN1+IN2" } Calculate(in1 := #TON, in2 := 0.1, out => #TON)
   END_RUNG
   RUNG wire#w1
      { S7_Templates := "SrcType := Real" } LT_Contact(in1 := #TOFF, in2 := #T_OFF)
      { S7_Templates := "SrcType := Real"; S7_Expression := "IN1+IN2" } Calculate(in1 := #TOFF, in2 := 0.1, out => #TOFF)
   END_RUNG
   RUNG wire#powerrail
      Contact( #"RUN_T/T" )
      { S7_Templates := "SrcType := Real" } GE_Contact(in1 := #TOFF, in2 := #T_OFF)
      Coil( #"TEMP_T/T" )
   END_RUNG
   RUNG wire#powerrail
      Contact( #"RUN_T/T" )
      { S7_Templates := "SrcType := Real" } EQ_Contact(in1 := #TOFF, in2 := #T_OFF)
      wire#w2
      Move(in := 0.0, out1 => #TOFF, out2 => #TON)
   END_RUNG
   RUNG wire#powerrail
      Contact( #"RUN_T/T" )
      { S7_Templates := "SrcType := Real" } GT_Contact(in1 := #TOFF, in2 := #T_OFF)
      { S7_Templates := "SrcType := Real" } GT_Contact(in1 := #TON, in2 := #T_ON)
   END_RUNG wire#w2
   RUNG wire#powerrail
      Contact( #FU )
   END_RUNG wire#w2
   // the same network as SCL:
   #_w1 := #"RUN_T/T" AND #X_CLOCK AND NOT #CLK_TT;   // rising edge of #X_CLOCK
   #CLK_TT := #X_CLOCK;
   IF #_w1 AND (#TOFF >= #T_OFF) AND (#TON < #T_ON) THEN #TON := #TON+0.1; END_IF;
   IF #_w1 AND (#TOFF < #T_OFF) THEN #TOFF := #TOFF+0.1; END_IF;
   #"TEMP_T/T" := #"RUN_T/T" AND (#TOFF >= #T_OFF);
   IF (#"RUN_T/T" AND (#TOFF = #T_OFF)) OR (#"RUN_T/T" AND (#TOFF > #T_OFF) AND (#TON > #T_ON)) OR #FU THEN
       #TOFF := 0.0;
       #TON := 0.0;
   END_IF;
END_REGION

REGION Network 10: CAN LOGIC
END_REGION

REGION Network 11: CUA THO TINH
   RUNG wire#powerrail
      { S7_Templates := "SrcType := Real" } NE_Contact(in1 := #SMT, in2 := 0.0)
      wire#w1
      N_Contact(operand := #Q_OUT1, bit := #P_OUT1)
      I_Contact( #"CUA_T/T" )
      S_Coil( #"CUA_T/T" )
   END_RUNG
   RUNG wire#w1
      N_Contact(operand := #Q_OUT2, bit := #P_OUT2)
      Contact( #"CUA_T/T" )
      R_Coil( #"CUA_T/T" )
   END_RUNG
   RUNG wire#powerrail
      { S7_Templates := "SrcType := Real" } EQ_Contact(in1 := #SMT, in2 := 0.0)
      R_Coil( #"CUA_T/T" )
   END_RUNG
   // the same network as SCL:
   #_w1 := #SMT <> 0.0;
   #_w2 := #_w1 AND NOT #Q_OUT1 AND #P_OUT1;   // falling edge of #Q_OUT1
   #P_OUT1 := #Q_OUT1;
   IF #_w2 AND NOT #"CUA_T/T" THEN #"CUA_T/T" := TRUE; END_IF;
   #_w3 := #_w1 AND NOT #Q_OUT2 AND #P_OUT2;   // falling edge of #Q_OUT2
   #P_OUT2 := #Q_OUT2;
   IF #_w3 AND #"CUA_T/T" THEN #"CUA_T/T" := FALSE; END_IF;
   IF #SMT = 0.0 THEN #"CUA_T/T" := FALSE; END_IF;
END_REGION
END_FUNCTION_BLOCK

FUNCTION "FCXL_CCD_FD1" : Void   // FC10, LAD
{ S7_Optimized_Access := 'TRUE' }
VERSION : 0.1
// stored: AutoNumber true, CodeModifiedDate 2026-01-04T14:27:05.4562814Z, CompileDate 2026-01-04T14:27:05.5189595Z, CreationDate 2024-10-13T15:07:34.9617085Z, HandleErrorsWithinBlock false, InterfaceModifiedDate 2024-08-08T03:13:40.4539851Z, IsConsistent true, IsIECCheckEnabled false, IsKnowHowProtected false, IsWriteProtected false, LibraryConformanceStatus Error: The block contains calls of single instances. Warning: The object contains access to global data blocks. Warning: The block contains direct access to inputs, outputs, bit memories, indirect access to the registry or indirect access to external memory areas that are unknown at the time of compilation., ModifiedDate 2026-01-04T14:27:05.4562814Z, ParameterModified 2024-08-08T03:13:40.4539851Z, PLCSimAdvancedSupport false, SetENOAutomatically False, StructureModified 2024-08-08T03:13:40.4539851Z, UDAEnableTagReadback false
   VAR_TEMP   // added for the SCL form of the ladder/FBD networks
      _w1 : Bool;
      _w2 : Bool;
      _w3 : Bool;
   END_VAR
BEGIN

REGION Network 1
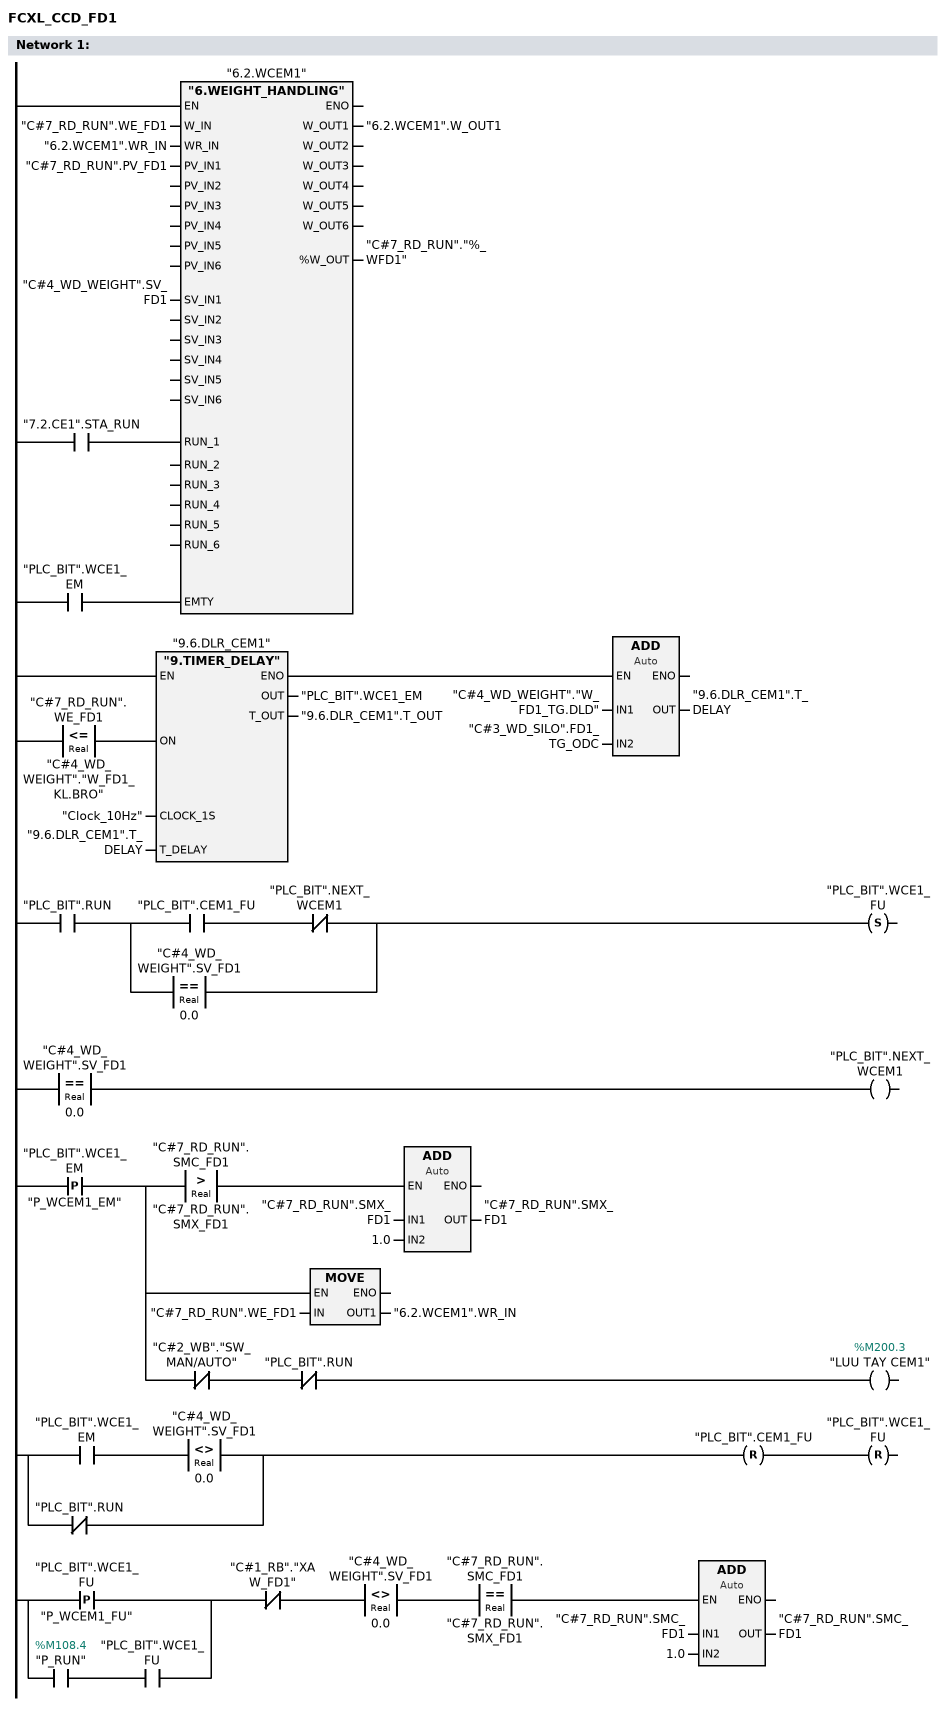
   RUNG wire#powerrail
      "6.2.WCEM1"(RUN_1 := wire#w1, EMTY := wire#w2, W_IN := "C#7_RD_RUN".WE_FD1, WR_IN := "6.2.WCEM1".WR_IN, PV_IN1 := "C#7_RD_RUN".PV_FD1, PV_IN2 :=, PV_IN3 :=, PV_IN4 :=, PV_IN5 :=, PV_IN6 :=, SV_IN1 := "C#4_WD_WEIGHT".SV_FD1, SV_IN2 :=, SV_IN3 :=, SV_IN4 :=, SV_IN5 :=, SV_IN6 :=, RUN_2 :=, RUN_3 :=, RUN_4 :=, RUN_5 :=, RUN_6 :=, W_OUT1 => "6.2.WCEM1".W_OUT1, W_OUT2 =>, W_OUT3 =>, W_OUT4 =>, W_OUT5 =>, W_OUT6 =>, "%W_OUT" => "C#7_RD_RUN"."%_WFD1")
   END_RUNG
   RUNG wire#powerrail
      Contact( "7.2.CE1".STA_RUN )
   END_RUNG wire#w1
   RUNG wire#powerrail
      Contact( "PLC_BIT".WCE1_EM )
   END_RUNG wire#w2
   RUNG wire#powerrail
      "9.6.DLR_CEM1"(ON := wire#w3, CLOCK_1S := "Clock_10Hz", T_DELAY := "9.6.DLR_CEM1".T_DELAY, OUT => "PLC_BIT".WCE1_EM, T_OUT => "9.6.DLR_CEM1".T_OUT)
      Add(in1 := "C#4_WD_WEIGHT"."W_FD1_TG.DLD", in2 := "C#3_WD_SILO".FD1_TG_ODC, out => "9.6.DLR_CEM1".T_DELAY)
   END_RUNG
   RUNG wire#powerrail
      { S7_Templates := "SrcType := Real" } LE_Contact(in1 := "C#7_RD_RUN".WE_FD1, in2 := "C#4_WD_WEIGHT"."W_FD1_KL.BRO")
   END_RUNG wire#w3
   RUNG wire#powerrail
      Contact( "PLC_BIT".RUN )
      wire#w4
      Contact( "PLC_BIT".CEM1_FU )
      I_Contact( "PLC_BIT".NEXT_WCEM1 )
      wire#w5
      S_Coil( "PLC_BIT".WCE1_FU )
   END_RUNG
   RUNG wire#w4
      { S7_Templates := "SrcType := Real" } EQ_Contact(in1 := "C#4_WD_WEIGHT".SV_FD1, in2 := 0.0)
   END_RUNG wire#w5
   RUNG wire#powerrail
      { S7_Templates := "SrcType := Real" } EQ_Contact(in1 := "C#4_WD_WEIGHT".SV_FD1, in2 := 0.0)
      Coil( "PLC_BIT".NEXT_WCEM1 )
   END_RUNG
   RUNG wire#powerrail
      P_Contact(operand := "PLC_BIT".WCE1_EM, bit := "P_WCEM1_EM")
      wire#w6
      { S7_Templates := "SrcType := Real" } GT_Contact(in1 := "C#7_RD_RUN".SMC_FD1, in2 := "C#7_RD_RUN".SMX_FD1)
      Add(in1 := "C#7_RD_RUN".SMX_FD1, in2 := 1.0, out => "C#7_RD_RUN".SMX_FD1)
   END_RUNG
   RUNG wire#w6
      Move(in := "C#7_RD_RUN".WE_FD1, out1 => "6.2.WCEM1".WR_IN)
   END_RUNG
   RUNG wire#w6
      I_Contact( "C#2_WB"."SW_MAN/AUTO" )
      I_Contact( "PLC_BIT".RUN )
      Coil( "LUU TAY CEM1" )
   END_RUNG
   RUNG wire#powerrail
      Contact( "PLC_BIT".WCE1_EM )
      { S7_Templates := "SrcType := Real" } NE_Contact(in1 := "C#4_WD_WEIGHT".SV_FD1, in2 := 0.0)
      wire#w7
      R_Coil( "PLC_BIT".CEM1_FU )
      R_Coil( "PLC_BIT".WCE1_FU )
   END_RUNG
   RUNG wire#powerrail
      I_Contact( "PLC_BIT".RUN )
   END_RUNG wire#w7
   RUNG wire#powerrail
      P_Contact(operand := "PLC_BIT".WCE1_FU, bit := "P_WCEM1_FU")
      wire#w8
      I_Contact( "C#1_RB"."XA W_FD1" )
      { S7_Templates := "SrcType := Real" } NE_Contact(in1 := "C#4_WD_WEIGHT".SV_FD1, in2 := 0.0)
      { S7_Templates := "SrcType := Real" } EQ_Contact(in1 := "C#7_RD_RUN".SMC_FD1, in2 := "C#7_RD_RUN".SMX_FD1)
      Add(in1 := "C#7_RD_RUN".SMC_FD1, in2 := 1.0, out => "C#7_RD_RUN".SMC_FD1)
   END_RUNG
   RUNG wire#powerrail
      Contact( "P_RUN" )
      Contact( "PLC_BIT".WCE1_FU )
   END_RUNG wire#w8
   // the same network as SCL:
   "6.2.WCEM1"(W_IN := "C#7_RD_RUN".WE_FD1,   // "6.WEIGHT_HANDLING"
               WR_IN := "6.2.WCEM1".WR_IN,
               PV_IN1 := "C#7_RD_RUN".PV_FD1,
               SV_IN1 := "C#4_WD_WEIGHT".SV_FD1,
               RUN_1 := "7.2.CE1".STA_RUN,
               EMTY := "PLC_BIT".WCE1_EM,
               W_OUT1 => "6.2.WCEM1".W_OUT1,
               "%W_OUT" => "C#7_RD_RUN"."%_WFD1");
   "9.6.DLR_CEM1"(ON := "C#7_RD_RUN".WE_FD1 <= "C#4_WD_WEIGHT"."W_FD1_KL.BRO",   // "9.TIMER_DELAY"
                  CLOCK_1S := "Clock_10Hz",
                  T_DELAY := "9.6.DLR_CEM1".T_DELAY,
                  OUT => "PLC_BIT".WCE1_EM,
                  T_OUT => "9.6.DLR_CEM1".T_OUT,
                  ENO => #_w1);
   IF #_w1 THEN "9.6.DLR_CEM1".T_DELAY := "C#4_WD_WEIGHT"."W_FD1_TG.DLD" + "C#3_WD_SILO".FD1_TG_ODC; END_IF;
   IF "PLC_BIT".RUN AND (("PLC_BIT".CEM1_FU AND NOT "PLC_BIT".NEXT_WCEM1) OR ("C#4_WD_WEIGHT".SV_FD1 = 0.0)) THEN
       "PLC_BIT".WCE1_FU := TRUE;
   END_IF;
   "PLC_BIT".NEXT_WCEM1 := "C#4_WD_WEIGHT".SV_FD1 = 0.0;
   #_w2 := "PLC_BIT".WCE1_EM AND NOT "P_WCEM1_EM";   // rising edge of "PLC_BIT".WCE1_EM
   "P_WCEM1_EM" := "PLC_BIT".WCE1_EM;
   IF #_w2 AND ("C#7_RD_RUN".SMC_FD1 > "C#7_RD_RUN".SMX_FD1) THEN
       "C#7_RD_RUN".SMX_FD1 := "C#7_RD_RUN".SMX_FD1 + 1.0;
   END_IF;
   IF #_w2 THEN "6.2.WCEM1".WR_IN := "C#7_RD_RUN".WE_FD1; END_IF;
   "LUU TAY CEM1" := #_w2 AND NOT "C#2_WB"."SW_MAN/AUTO" AND NOT "PLC_BIT".RUN;
   IF ("PLC_BIT".WCE1_EM AND ("C#4_WD_WEIGHT".SV_FD1 <> 0.0)) OR NOT "PLC_BIT".RUN THEN
       "PLC_BIT".CEM1_FU := FALSE;
       "PLC_BIT".WCE1_FU := FALSE;
   END_IF;
   #_w3 := "PLC_BIT".WCE1_FU AND NOT "P_WCEM1_FU";   // rising edge of "PLC_BIT".WCE1_FU
   "P_WCEM1_FU" := "PLC_BIT".WCE1_FU;
   IF (#_w3 OR ("P_RUN" AND "PLC_BIT".WCE1_FU)) AND NOT "C#1_RB"."XA W_FD1" AND ("C#4_WD_WEIGHT".SV_FD1 <> 0.0) AND ("C#7_RD_RUN".SMC_FD1 = "C#7_RD_RUN".SMX_FD1) THEN
       "C#7_RD_RUN".SMC_FD1 := "C#7_RD_RUN".SMC_FD1 + 1.0;
   END_IF;
END_REGION
END_FUNCTION

FUNCTION "FCCA_CCD_FD1" : Void   // FC12, LAD
{ S7_Optimized_Access := 'TRUE' }
VERSION : 0.1
// stored: AutoNumber true, CodeModifiedDate 2026-01-04T14:27:04.612364Z, CompileDate 2026-01-04T14:27:05.6125141Z, CreationDate 2024-10-13T15:07:34.9617085Z, HandleErrorsWithinBlock false, InterfaceModifiedDate 2024-08-08T03:19:31.8063857Z, IsConsistent true, IsIECCheckEnabled false, IsKnowHowProtected false, IsWriteProtected false, LibraryConformanceStatus Error: The block contains calls of single instances. Warning: The object contains access to global data blocks. Warning: The block contains direct access to inputs, outputs, bit memories, indirect access to the registry or indirect access to external memory areas that are unknown at the time of compilation., ModifiedDate 2026-01-04T14:27:04.612364Z, ParameterModified 2024-08-08T03:19:31.8063857Z, PLCSimAdvancedSupport false, SetENOAutomatically False, StructureModified 2024-08-08T03:19:31.8063857Z, UDAEnableTagReadback false
   VAR_TEMP   // added for the SCL form of the ladder/FBD networks
      _w1 : Bool;
   END_VAR
BEGIN

REGION Network 1: CAN XI MANG 1
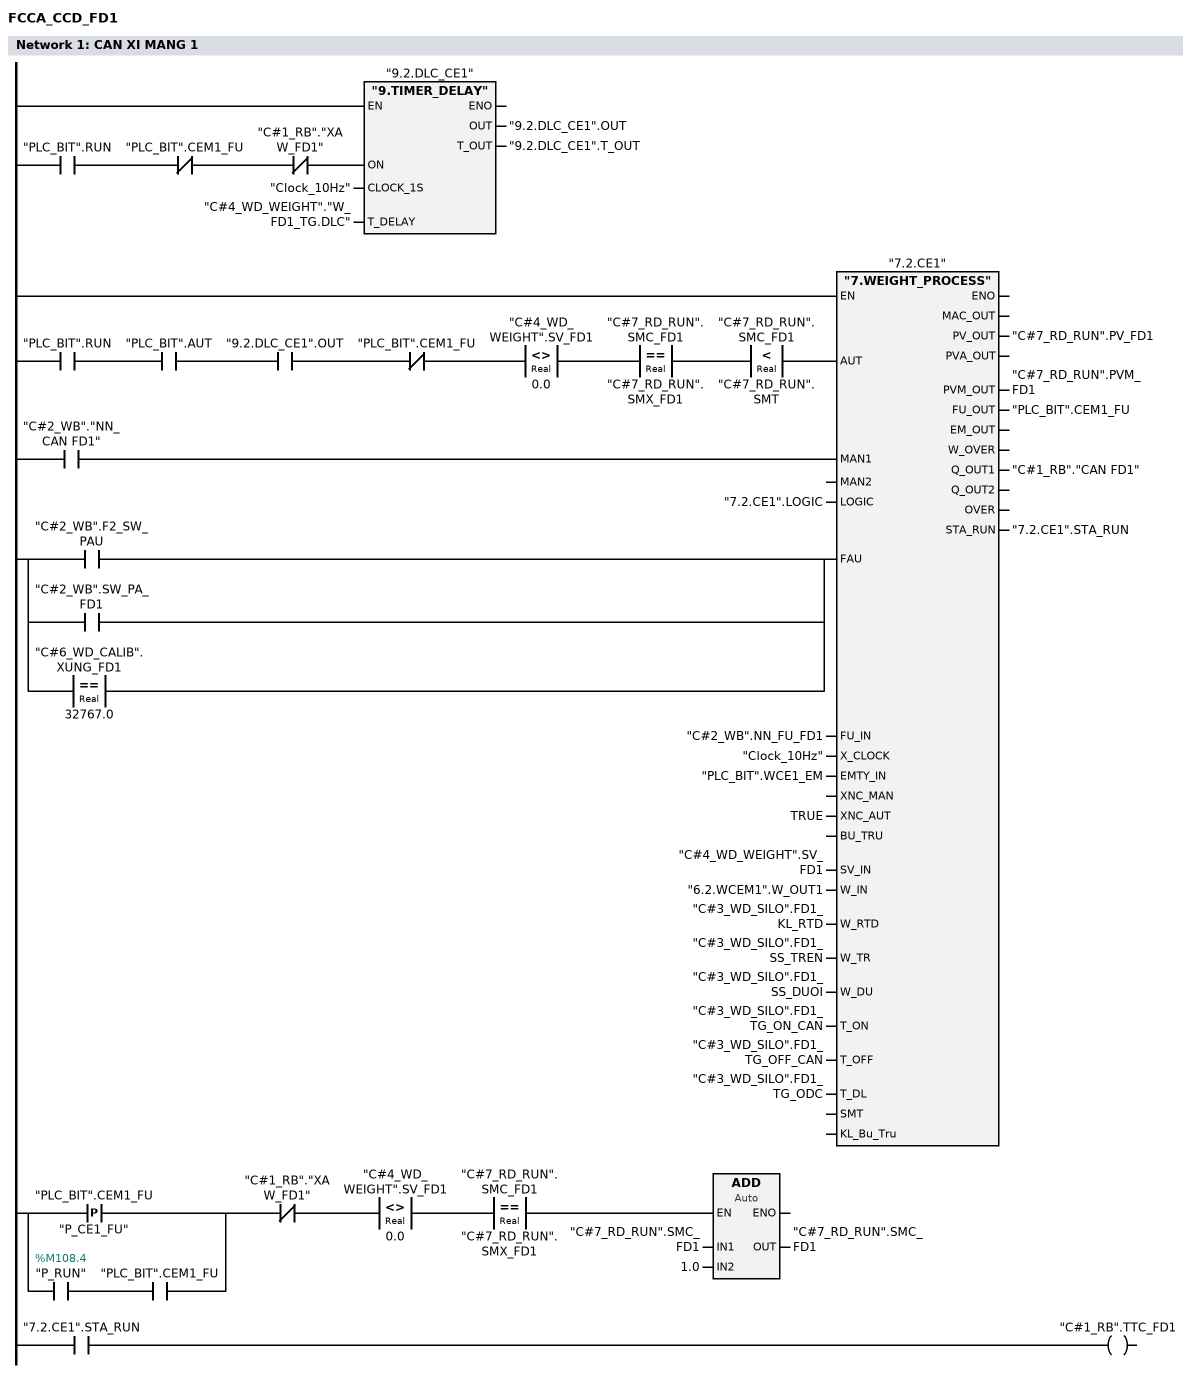
   RUNG wire#powerrail
      "9.2.DLC_CE1"(ON := wire#w1, CLOCK_1S := "Clock_10Hz", T_DELAY := "C#4_WD_WEIGHT"."W_FD1_TG.DLC", OUT => "9.2.DLC_CE1".OUT, T_OUT => "9.2.DLC_CE1".T_OUT)
   END_RUNG
   RUNG wire#powerrail
      Contact( "PLC_BIT".RUN )
      I_Contact( "PLC_BIT".CEM1_FU )
      I_Contact( "C#1_RB"."XA W_FD1" )
   END_RUNG wire#w1
   RUNG wire#powerrail
      "7.2.CE1"(AUT := wire#w2, MAN1 := wire#w3, FAU := wire#w4, MAN2 :=, LOGIC := "7.2.CE1".LOGIC, FU_IN := "C#2_WB".NN_FU_FD1, X_CLOCK := "Clock_10Hz", EMTY_IN := "PLC_BIT".WCE1_EM, XNC_MAN :=, XNC_AUT := TRUE, BU_TRU :=, SV_IN := "C#4_WD_WEIGHT".SV_FD1, W_IN := "6.2.WCEM1".W_OUT1, W_RTD := "C#3_WD_SILO".FD1_KL_RTD, W_TR := "C#3_WD_SILO".FD1_SS_TREN, W_DU := "C#3_WD_SILO".FD1_SS_DUOI, T_ON := "C#3_WD_SILO".FD1_TG_ON_CAN, T_OFF := "C#3_WD_SILO".FD1_TG_OFF_CAN, T_DL := "C#3_WD_SILO".FD1_TG_ODC, SMT :=, KL_Bu_Tru :=, MAC_OUT =>, PV_OUT => "C#7_RD_RUN".PV_FD1, PVA_OUT =>, PVM_OUT => "C#7_RD_RUN".PVM_FD1, FU_OUT => "PLC_BIT".CEM1_FU, EM_OUT =>, W_OVER =>, Q_OUT1 => "C#1_RB"."CAN FD1", Q_OUT2 =>, OVER =>, STA_RUN => "7.2.CE1".STA_RUN)
   END_RUNG
   RUNG wire#powerrail
      Contact( "PLC_BIT".RUN )
      Contact( "PLC_BIT".AUT )
      Contact( "9.2.DLC_CE1".OUT )
      I_Contact( "PLC_BIT".CEM1_FU )
      { S7_Templates := "SrcType := Real" } NE_Contact(in1 := "C#4_WD_WEIGHT".SV_FD1, in2 := 0.0)
      { S7_Templates := "SrcType := Real" } EQ_Contact(in1 := "C#7_RD_RUN".SMC_FD1, in2 := "C#7_RD_RUN".SMX_FD1)
      { S7_Templates := "SrcType := Real" } LT_Contact(in1 := "C#7_RD_RUN".SMC_FD1, in2 := "C#7_RD_RUN".SMT)
   END_RUNG wire#w2
   RUNG wire#powerrail
      Contact( "C#2_WB"."NN_CAN FD1" )
   END_RUNG wire#w3
   RUNG wire#powerrail
      Contact( "C#2_WB".F2_SW_PAU )
   END_RUNG wire#w4
   RUNG wire#powerrail
      Contact( "C#2_WB".SW_PA_FD1 )
   END_RUNG wire#w4
   RUNG wire#powerrail
      { S7_Templates := "SrcType := Real" } EQ_Contact(in1 := "C#6_WD_CALIB".XUNG_FD1, in2 := 32767.0)
   END_RUNG wire#w4
   RUNG wire#powerrail
      P_Contact(operand := "PLC_BIT".CEM1_FU, bit := "P_CE1_FU")
      wire#w5
      I_Contact( "C#1_RB"."XA W_FD1" )
      { S7_Templates := "SrcType := Real" } NE_Contact(in1 := "C#4_WD_WEIGHT".SV_FD1, in2 := 0.0)
      { S7_Templates := "SrcType := Real" } EQ_Contact(in1 := "C#7_RD_RUN".SMC_FD1, in2 := "C#7_RD_RUN".SMX_FD1)
      Add(in1 := "C#7_RD_RUN".SMC_FD1, in2 := 1.0, out => "C#7_RD_RUN".SMC_FD1)
   END_RUNG
   RUNG wire#powerrail
      Contact( "P_RUN" )
      Contact( "PLC_BIT".CEM1_FU )
   END_RUNG wire#w5
   RUNG wire#powerrail
      Contact( "7.2.CE1".STA_RUN )
      Coil( "C#1_RB".TTC_FD1 )
   END_RUNG
   // the same network as SCL:
   "9.2.DLC_CE1"(ON := "PLC_BIT".RUN AND NOT "PLC_BIT".CEM1_FU AND NOT "C#1_RB"."XA W_FD1",   // "9.TIMER_DELAY"
                 CLOCK_1S := "Clock_10Hz",
                 T_DELAY := "C#4_WD_WEIGHT"."W_FD1_TG.DLC",
                 OUT => "9.2.DLC_CE1".OUT,
                 T_OUT => "9.2.DLC_CE1".T_OUT);
   "7.2.CE1"(AUT := "PLC_BIT".RUN AND "PLC_BIT".AUT AND "9.2.DLC_CE1".OUT AND NOT "PLC_BIT".CEM1_FU AND ("C#4_WD_WEIGHT".SV_FD1 <> 0.0) AND ("C#7_RD_RUN".SMC_FD1 = "C#7_RD_RUN".SMX_FD1) AND ("C#7_RD_RUN".SMC_FD1 < "C#7_RD_RUN".SMT),   // "7.WEIGHT_PROCESS"
             MAN1 := "C#2_WB"."NN_CAN FD1",
             LOGIC := "7.2.CE1".LOGIC,
             FAU := "C#2_WB".F2_SW_PAU OR "C#2_WB".SW_PA_FD1 OR ("C#6_WD_CALIB".XUNG_FD1 = 32767.0),
             FU_IN := "C#2_WB".NN_FU_FD1,
             X_CLOCK := "Clock_10Hz",
             EMTY_IN := "PLC_BIT".WCE1_EM,
             XNC_AUT := TRUE,
             SV_IN := "C#4_WD_WEIGHT".SV_FD1,
             W_IN := "6.2.WCEM1".W_OUT1,
             W_RTD := "C#3_WD_SILO".FD1_KL_RTD,
             W_TR := "C#3_WD_SILO".FD1_SS_TREN,
             W_DU := "C#3_WD_SILO".FD1_SS_DUOI,
             T_ON := "C#3_WD_SILO".FD1_TG_ON_CAN,
             T_OFF := "C#3_WD_SILO".FD1_TG_OFF_CAN,
             T_DL := "C#3_WD_SILO".FD1_TG_ODC,
             PV_OUT => "C#7_RD_RUN".PV_FD1,
             PVM_OUT => "C#7_RD_RUN".PVM_FD1,
             FU_OUT => "PLC_BIT".CEM1_FU,
             Q_OUT1 => "C#1_RB"."CAN FD1",
             STA_RUN => "7.2.CE1".STA_RUN);
   #_w1 := "PLC_BIT".CEM1_FU AND NOT "P_CE1_FU";   // rising edge of "PLC_BIT".CEM1_FU
   "P_CE1_FU" := "PLC_BIT".CEM1_FU;
   IF (#_w1 OR ("P_RUN" AND "PLC_BIT".CEM1_FU)) AND NOT "C#1_RB"."XA W_FD1" AND ("C#4_WD_WEIGHT".SV_FD1 <> 0.0) AND ("C#7_RD_RUN".SMC_FD1 = "C#7_RD_RUN".SMX_FD1) THEN
       "C#7_RD_RUN".SMC_FD1 := "C#7_RD_RUN".SMC_FD1 + 1.0;
   END_IF;
   "C#1_RB".TTC_FD1 := "7.2.CE1".STA_RUN;
END_REGION
END_FUNCTION

FUNCTION "FCXL_CCD_AP1" : Void   // FC15, LAD
{ S7_Optimized_Access := 'TRUE' }
VERSION : 0.1
// stored: AutoNumber true, CodeModifiedDate 2026-01-04T14:27:05.6438339Z, CompileDate 2026-01-04T14:27:05.690726Z, CreationDate 2024-10-13T15:07:34.9617085Z, HandleErrorsWithinBlock false, InterfaceModifiedDate 2024-08-08T03:23:40.7447783Z, IsConsistent true, IsIECCheckEnabled false, IsKnowHowProtected false, IsWriteProtected false, LibraryConformanceStatus Error: The block contains calls of single instances. Warning: The object contains access to global data blocks. Warning: The block contains direct access to inputs, outputs, bit memories, indirect access to the registry or indirect access to external memory areas that are unknown at the time of compilation., ModifiedDate 2026-01-04T14:27:05.6438339Z, ParameterModified 2024-08-08T03:23:40.7447783Z, PLCSimAdvancedSupport false, SetENOAutomatically False, StructureModified 2024-08-08T03:23:40.7447783Z, UDAEnableTagReadback false
   VAR_TEMP   // added for the SCL form of the ladder/FBD networks
      _w1 : Bool;
      _w2 : Bool;
      _w3 : Bool;
   END_VAR
BEGIN

REGION Network 1
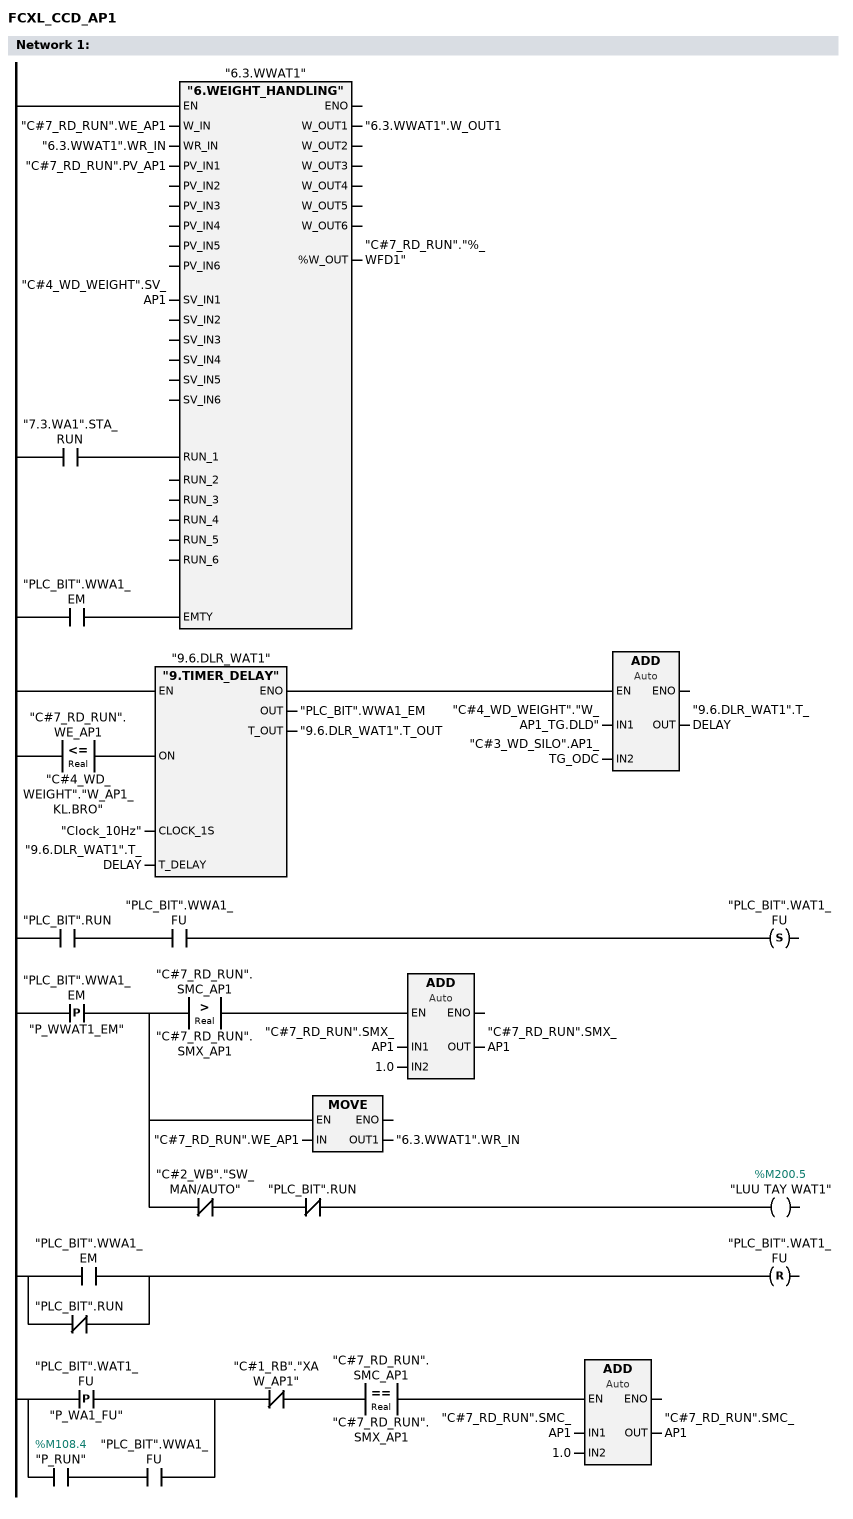
   RUNG wire#powerrail
      "6.3.WWAT1"(RUN_1 := wire#w1, EMTY := wire#w2, W_IN := "C#7_RD_RUN".WE_AP1, WR_IN := "6.3.WWAT1".WR_IN, PV_IN1 := "C#7_RD_RUN".PV_AP1, PV_IN2 :=, PV_IN3 :=, PV_IN4 :=, PV_IN5 :=, PV_IN6 :=, SV_IN1 := "C#4_WD_WEIGHT".SV_AP1, SV_IN2 :=, SV_IN3 :=, SV_IN4 :=, SV_IN5 :=, SV_IN6 :=, RUN_2 :=, RUN_3 :=, RUN_4 :=, RUN_5 :=, RUN_6 :=, W_OUT1 => "6.3.WWAT1".W_OUT1, W_OUT2 =>, W_OUT3 =>, W_OUT4 =>, W_OUT5 =>, W_OUT6 =>, "%W_OUT" => "C#7_RD_RUN"."%_WFD1")
   END_RUNG
   RUNG wire#powerrail
      Contact( "7.3.WA1".STA_RUN )
   END_RUNG wire#w1
   RUNG wire#powerrail
      Contact( "PLC_BIT".WWA1_EM )
   END_RUNG wire#w2
   RUNG wire#powerrail
      "9.6.DLR_WAT1"(ON := wire#w3, CLOCK_1S := "Clock_10Hz", T_DELAY := "9.6.DLR_WAT1".T_DELAY, OUT => "PLC_BIT".WWA1_EM, T_OUT => "9.6.DLR_WAT1".T_OUT)
      Add(in1 := "C#4_WD_WEIGHT"."W_AP1_TG.DLD", in2 := "C#3_WD_SILO".AP1_TG_ODC, out => "9.6.DLR_WAT1".T_DELAY)
   END_RUNG
   RUNG wire#powerrail
      { S7_Templates := "SrcType := Real" } LE_Contact(in1 := "C#7_RD_RUN".WE_AP1, in2 := "C#4_WD_WEIGHT"."W_AP1_KL.BRO")
   END_RUNG wire#w3
   RUNG wire#powerrail
      Contact( "PLC_BIT".RUN )
      Contact( "PLC_BIT".WWA1_FU )
      S_Coil( "PLC_BIT".WAT1_FU )
   END_RUNG
   RUNG wire#powerrail
      P_Contact(operand := "PLC_BIT".WWA1_EM, bit := "P_WWAT1_EM")
      wire#w4
      { S7_Templates := "SrcType := Real" } GT_Contact(in1 := "C#7_RD_RUN".SMC_AP1, in2 := "C#7_RD_RUN".SMX_AP1)
      Add(in1 := "C#7_RD_RUN".SMX_AP1, in2 := 1.0, out => "C#7_RD_RUN".SMX_AP1)
   END_RUNG
   RUNG wire#w4
      Move(in := "C#7_RD_RUN".WE_AP1, out1 => "6.3.WWAT1".WR_IN)
   END_RUNG
   RUNG wire#w4
      I_Contact( "C#2_WB"."SW_MAN/AUTO" )
      I_Contact( "PLC_BIT".RUN )
      Coil( "LUU TAY WAT1" )
   END_RUNG
   RUNG wire#powerrail
      Contact( "PLC_BIT".WWA1_EM )
      wire#w5
      R_Coil( "PLC_BIT".WAT1_FU )
   END_RUNG
   RUNG wire#powerrail
      I_Contact( "PLC_BIT".RUN )
   END_RUNG wire#w5
   RUNG wire#powerrail
      P_Contact(operand := "PLC_BIT".WAT1_FU, bit := "P_WA1_FU")
      wire#w6
      I_Contact( "C#1_RB"."XA W_AP1" )
      { S7_Templates := "SrcType := Real" } EQ_Contact(in1 := "C#7_RD_RUN".SMC_AP1, in2 := "C#7_RD_RUN".SMX_AP1)
      Add(in1 := "C#7_RD_RUN".SMC_AP1, in2 := 1.0, out => "C#7_RD_RUN".SMC_AP1)
   END_RUNG
   RUNG wire#powerrail
      Contact( "P_RUN" )
      Contact( "PLC_BIT".WWA1_FU )
   END_RUNG wire#w6
   // the same network as SCL:
   "6.3.WWAT1"(W_IN := "C#7_RD_RUN".WE_AP1,   // "6.WEIGHT_HANDLING"
               WR_IN := "6.3.WWAT1".WR_IN,
               PV_IN1 := "C#7_RD_RUN".PV_AP1,
               SV_IN1 := "C#4_WD_WEIGHT".SV_AP1,
               RUN_1 := "7.3.WA1".STA_RUN,
               EMTY := "PLC_BIT".WWA1_EM,
               W_OUT1 => "6.3.WWAT1".W_OUT1,
               "%W_OUT" => "C#7_RD_RUN"."%_WFD1");
   "9.6.DLR_WAT1"(ON := "C#7_RD_RUN".WE_AP1 <= "C#4_WD_WEIGHT"."W_AP1_KL.BRO",   // "9.TIMER_DELAY"
                  CLOCK_1S := "Clock_10Hz",
                  T_DELAY := "9.6.DLR_WAT1".T_DELAY,
                  OUT => "PLC_BIT".WWA1_EM,
                  T_OUT => "9.6.DLR_WAT1".T_OUT,
                  ENO => #_w1);
   IF #_w1 THEN "9.6.DLR_WAT1".T_DELAY := "C#4_WD_WEIGHT"."W_AP1_TG.DLD" + "C#3_WD_SILO".AP1_TG_ODC; END_IF;
   IF "PLC_BIT".RUN AND "PLC_BIT".WWA1_FU THEN "PLC_BIT".WAT1_FU := TRUE; END_IF;
   #_w2 := "PLC_BIT".WWA1_EM AND NOT "P_WWAT1_EM";   // rising edge of "PLC_BIT".WWA1_EM
   "P_WWAT1_EM" := "PLC_BIT".WWA1_EM;
   IF #_w2 AND ("C#7_RD_RUN".SMC_AP1 > "C#7_RD_RUN".SMX_AP1) THEN
       "C#7_RD_RUN".SMX_AP1 := "C#7_RD_RUN".SMX_AP1 + 1.0;
   END_IF;
   IF #_w2 THEN "6.3.WWAT1".WR_IN := "C#7_RD_RUN".WE_AP1; END_IF;
   "LUU TAY WAT1" := #_w2 AND NOT "C#2_WB"."SW_MAN/AUTO" AND NOT "PLC_BIT".RUN;
   IF "PLC_BIT".WWA1_EM OR NOT "PLC_BIT".RUN THEN "PLC_BIT".WAT1_FU := FALSE; END_IF;
   #_w3 := "PLC_BIT".WAT1_FU AND NOT "P_WA1_FU";   // rising edge of "PLC_BIT".WAT1_FU
   "P_WA1_FU" := "PLC_BIT".WAT1_FU;
   IF (#_w3 OR ("P_RUN" AND "PLC_BIT".WWA1_FU)) AND NOT "C#1_RB"."XA W_AP1" AND ("C#7_RD_RUN".SMC_AP1 = "C#7_RD_RUN".SMX_AP1) THEN
       "C#7_RD_RUN".SMC_AP1 := "C#7_RD_RUN".SMC_AP1 + 1.0;
   END_IF;
END_REGION
END_FUNCTION

FUNCTION "FCCA_CCD_AP1" : Void   // FC16, LAD
{ S7_Optimized_Access := 'TRUE' }
VERSION : 0.1
// stored: AutoNumber true, CodeModifiedDate 2026-01-04T14:27:04.5966227Z, CompileDate 2026-01-04T14:27:05.7689468Z, CreationDate 2024-10-13T15:07:34.9617085Z, HandleErrorsWithinBlock false, InterfaceModifiedDate 2024-08-08T03:24:33.8704482Z, IsConsistent true, IsIECCheckEnabled false, IsKnowHowProtected false, IsWriteProtected false, LibraryConformanceStatus Error: The block contains calls of single instances. Warning: The object contains access to global data blocks. Warning: The block contains direct access to inputs, outputs, bit memories, indirect access to the registry or indirect access to external memory areas that are unknown at the time of compilation., ModifiedDate 2026-01-06T10:18:41.758331Z, ParameterModified 2024-08-08T03:24:33.8704482Z, PLCSimAdvancedSupport false, SetENOAutomatically False, StructureModified 2024-08-08T03:24:33.8704482Z, UDAEnableTagReadback false
BEGIN

REGION Network 1: Trạng thái cân Nước 1 hoặc AP1
   // Đầu tiên nó sẽ đợi một khoảng thời gian gọi là Thời gian trễ cân, sau đó nó mới đủ điều kiện để cân
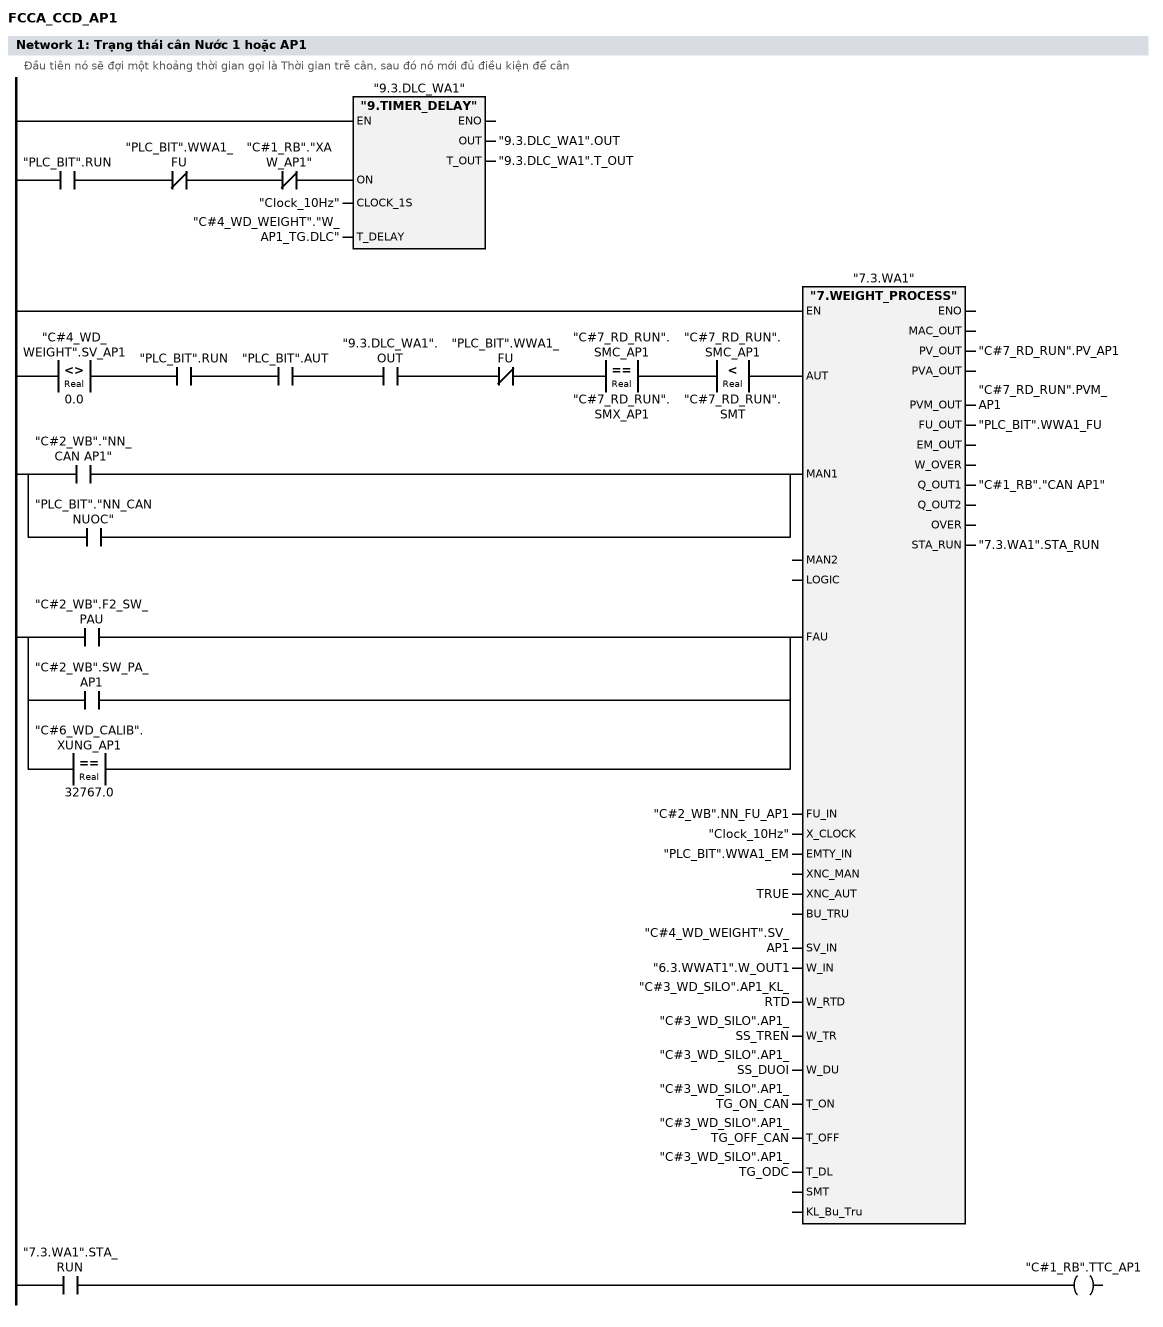
   RUNG wire#powerrail
      "9.3.DLC_WA1"(ON := wire#w1, CLOCK_1S := "Clock_10Hz", T_DELAY := "C#4_WD_WEIGHT"."W_AP1_TG.DLC", OUT => "9.3.DLC_WA1".OUT, T_OUT => "9.3.DLC_WA1".T_OUT)
   END_RUNG
   RUNG wire#powerrail
      Contact( "PLC_BIT".RUN )
      I_Contact( "PLC_BIT".WWA1_FU )
      I_Contact( "C#1_RB"."XA W_AP1" )
   END_RUNG wire#w1
   RUNG wire#powerrail
      "7.3.WA1"(AUT := wire#w2, MAN1 := wire#w3, FAU := wire#w4, MAN2 :=, LOGIC :=, FU_IN := "C#2_WB".NN_FU_AP1, X_CLOCK := "Clock_10Hz", EMTY_IN := "PLC_BIT".WWA1_EM, XNC_MAN :=, XNC_AUT := TRUE, BU_TRU :=, SV_IN := "C#4_WD_WEIGHT".SV_AP1, W_IN := "6.3.WWAT1".W_OUT1, W_RTD := "C#3_WD_SILO".AP1_KL_RTD, W_TR := "C#3_WD_SILO".AP1_SS_TREN, W_DU := "C#3_WD_SILO".AP1_SS_DUOI, T_ON := "C#3_WD_SILO".AP1_TG_ON_CAN, T_OFF := "C#3_WD_SILO".AP1_TG_OFF_CAN, T_DL := "C#3_WD_SILO".AP1_TG_ODC, SMT :=, KL_Bu_Tru :=, MAC_OUT =>, PV_OUT => "C#7_RD_RUN".PV_AP1, PVA_OUT =>, PVM_OUT => "C#7_RD_RUN".PVM_AP1, FU_OUT => "PLC_BIT".WWA1_FU, EM_OUT =>, W_OVER =>, Q_OUT1 => "C#1_RB"."CAN AP1", Q_OUT2 =>, OVER =>, STA_RUN => "7.3.WA1".STA_RUN)
   END_RUNG
   RUNG wire#powerrail
      { S7_Templates := "SrcType := Real" } NE_Contact(in1 := "C#4_WD_WEIGHT".SV_AP1, in2 := 0.0)
      Contact( "PLC_BIT".RUN )
      Contact( "PLC_BIT".AUT )
      Contact( "9.3.DLC_WA1".OUT )
      I_Contact( "PLC_BIT".WWA1_FU )
      { S7_Templates := "SrcType := Real" } EQ_Contact(in1 := "C#7_RD_RUN".SMC_AP1, in2 := "C#7_RD_RUN".SMX_AP1)
      { S7_Templates := "SrcType := Real" } LT_Contact(in1 := "C#7_RD_RUN".SMC_AP1, in2 := "C#7_RD_RUN".SMT)
   END_RUNG wire#w2
   RUNG wire#powerrail
      Contact( "C#2_WB"."NN_CAN AP1" )
   END_RUNG wire#w3
   RUNG wire#powerrail
      Contact( "PLC_BIT"."NN_CAN NUOC" )
   END_RUNG wire#w3
   RUNG wire#powerrail
      Contact( "C#2_WB".F2_SW_PAU )
   END_RUNG wire#w4
   RUNG wire#powerrail
      Contact( "C#2_WB".SW_PA_AP1 )
   END_RUNG wire#w4
   RUNG wire#powerrail
      { S7_Templates := "SrcType := Real" } EQ_Contact(in1 := "C#6_WD_CALIB".XUNG_AP1, in2 := 32767.0)
   END_RUNG wire#w4
   RUNG wire#powerrail
      Contact( "7.3.WA1".STA_RUN )
      Coil( "C#1_RB".TTC_AP1 )
   END_RUNG
   // the same network as SCL:
   "9.3.DLC_WA1"(ON := "PLC_BIT".RUN AND NOT "PLC_BIT".WWA1_FU AND NOT "C#1_RB"."XA W_AP1",   // "9.TIMER_DELAY"
                 CLOCK_1S := "Clock_10Hz",
                 T_DELAY := "C#4_WD_WEIGHT"."W_AP1_TG.DLC",
                 OUT => "9.3.DLC_WA1".OUT,
                 T_OUT => "9.3.DLC_WA1".T_OUT);
   "7.3.WA1"(AUT := ("C#4_WD_WEIGHT".SV_AP1 <> 0.0) AND "PLC_BIT".RUN AND "PLC_BIT".AUT AND "9.3.DLC_WA1".OUT AND NOT "PLC_BIT".WWA1_FU AND ("C#7_RD_RUN".SMC_AP1 = "C#7_RD_RUN".SMX_AP1) AND ("C#7_RD_RUN".SMC_AP1 < "C#7_RD_RUN".SMT),   // "7.WEIGHT_PROCESS"
             MAN1 := "C#2_WB"."NN_CAN AP1" OR "PLC_BIT"."NN_CAN NUOC",
             FAU := "C#2_WB".F2_SW_PAU OR "C#2_WB".SW_PA_AP1 OR ("C#6_WD_CALIB".XUNG_AP1 = 32767.0),
             FU_IN := "C#2_WB".NN_FU_AP1,
             X_CLOCK := "Clock_10Hz",
             EMTY_IN := "PLC_BIT".WWA1_EM,
             XNC_AUT := TRUE,
             SV_IN := "C#4_WD_WEIGHT".SV_AP1,
             W_IN := "6.3.WWAT1".W_OUT1,
             W_RTD := "C#3_WD_SILO".AP1_KL_RTD,
             W_TR := "C#3_WD_SILO".AP1_SS_TREN,
             W_DU := "C#3_WD_SILO".AP1_SS_DUOI,
             T_ON := "C#3_WD_SILO".AP1_TG_ON_CAN,
             T_OFF := "C#3_WD_SILO".AP1_TG_OFF_CAN,
             T_DL := "C#3_WD_SILO".AP1_TG_ODC,
             PV_OUT => "C#7_RD_RUN".PV_AP1,
             PVM_OUT => "C#7_RD_RUN".PVM_AP1,
             FU_OUT => "PLC_BIT".WWA1_FU,
             Q_OUT1 => "C#1_RB"."CAN AP1",
             STA_RUN => "7.3.WA1".STA_RUN);
   "C#1_RB".TTC_AP1 := "7.3.WA1".STA_RUN;
END_REGION
END_FUNCTION

FUNCTION "FCXL_CCD_SB1" : Void   // FC17, LAD
{ S7_Optimized_Access := 'TRUE' }
VERSION : 0.1
// stored: AutoNumber true, CodeModifiedDate 2026-01-04T14:27:05.8156344Z, CompileDate 2026-01-04T14:27:05.8623022Z, CreationDate 2024-10-13T15:07:34.9617085Z, HandleErrorsWithinBlock false, InterfaceModifiedDate 2024-08-08T03:53:18.695573Z, IsConsistent true, IsIECCheckEnabled false, IsKnowHowProtected false, IsWriteProtected false, LibraryConformanceStatus Error: The block contains calls of single instances. Warning: The object contains access to global data blocks. Warning: The block contains direct access to inputs, outputs, bit memories, indirect access to the registry or indirect access to external memory areas that are unknown at the time of compilation., ModifiedDate 2026-01-04T14:27:05.8156344Z, ParameterModified 2024-08-08T03:53:18.695573Z, PLCSimAdvancedSupport false, SetENOAutomatically False, StructureModified 2024-08-08T03:53:18.695573Z, UDAEnableTagReadback false
   VAR_TEMP   // added for the SCL form of the ladder/FBD networks
      _w1 : Bool;
      _w2 : Bool;
      _w3 : Bool;
   END_VAR
BEGIN

REGION Network 1
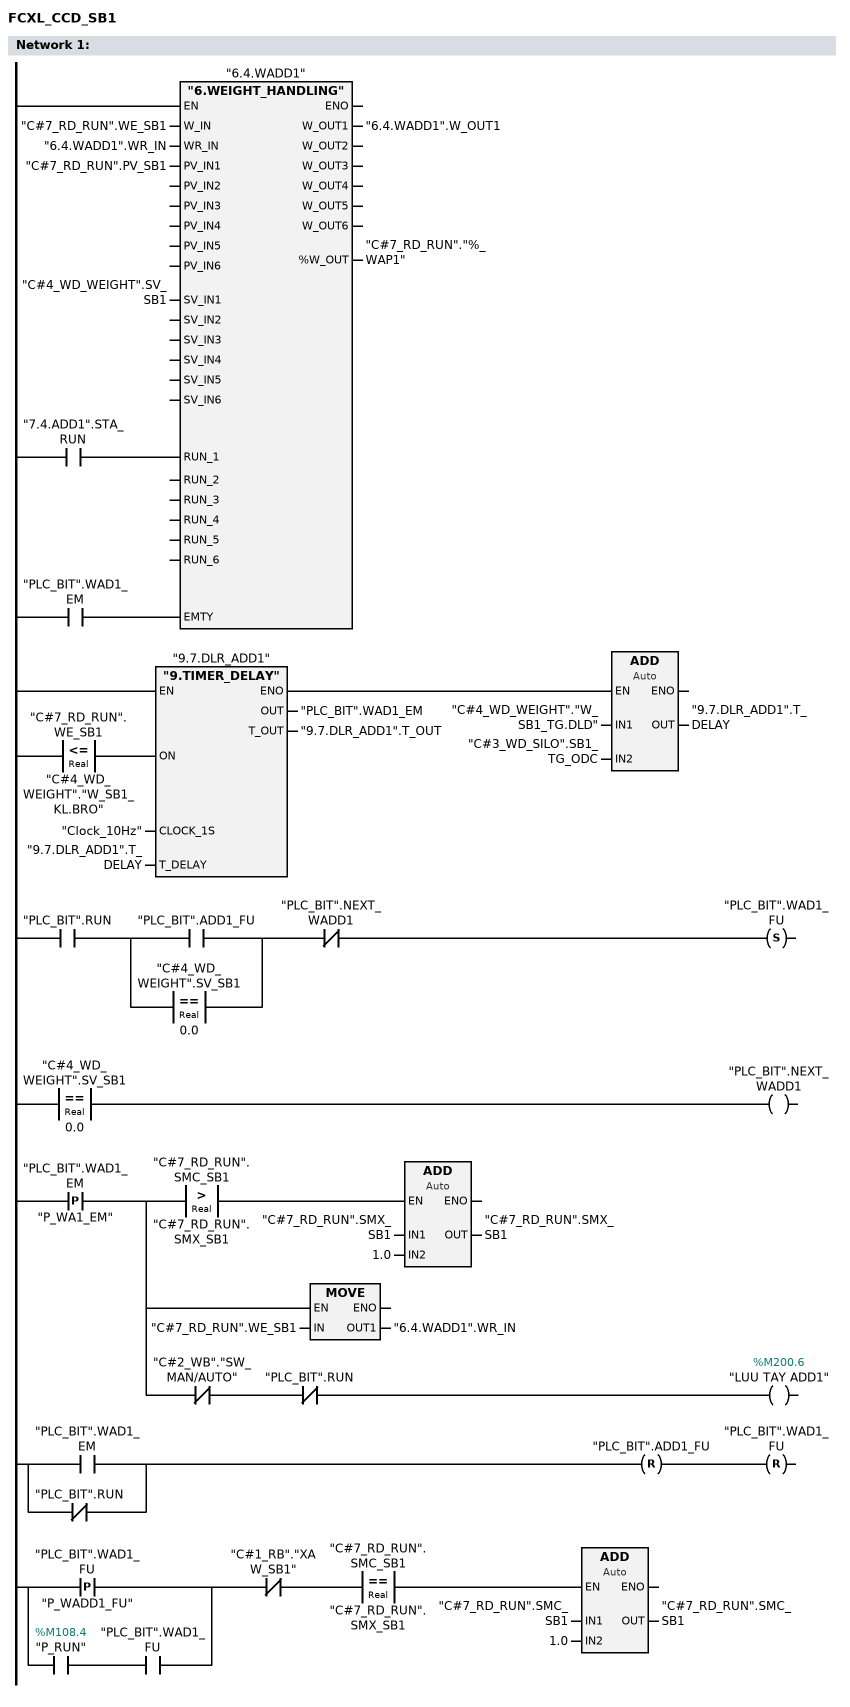
   RUNG wire#powerrail
      "6.4.WADD1"(RUN_1 := wire#w1, EMTY := wire#w2, W_IN := "C#7_RD_RUN".WE_SB1, WR_IN := "6.4.WADD1".WR_IN, PV_IN1 := "C#7_RD_RUN".PV_SB1, PV_IN2 :=, PV_IN3 :=, PV_IN4 :=, PV_IN5 :=, PV_IN6 :=, SV_IN1 := "C#4_WD_WEIGHT".SV_SB1, SV_IN2 :=, SV_IN3 :=, SV_IN4 :=, SV_IN5 :=, SV_IN6 :=, RUN_2 :=, RUN_3 :=, RUN_4 :=, RUN_5 :=, RUN_6 :=, W_OUT1 => "6.4.WADD1".W_OUT1, W_OUT2 =>, W_OUT3 =>, W_OUT4 =>, W_OUT5 =>, W_OUT6 =>, "%W_OUT" => "C#7_RD_RUN"."%_WAP1")
   END_RUNG
   RUNG wire#powerrail
      Contact( "7.4.ADD1".STA_RUN )
   END_RUNG wire#w1
   RUNG wire#powerrail
      Contact( "PLC_BIT".WAD1_EM )
   END_RUNG wire#w2
   RUNG wire#powerrail
      "9.7.DLR_ADD1"(ON := wire#w3, CLOCK_1S := "Clock_10Hz", T_DELAY := "9.7.DLR_ADD1".T_DELAY, OUT => "PLC_BIT".WAD1_EM, T_OUT => "9.7.DLR_ADD1".T_OUT)
      Add(in1 := "C#4_WD_WEIGHT"."W_SB1_TG.DLD", in2 := "C#3_WD_SILO".SB1_TG_ODC, out => "9.7.DLR_ADD1".T_DELAY)
   END_RUNG
   RUNG wire#powerrail
      { S7_Templates := "SrcType := Real" } LE_Contact(in1 := "C#7_RD_RUN".WE_SB1, in2 := "C#4_WD_WEIGHT"."W_SB1_KL.BRO")
   END_RUNG wire#w3
   RUNG wire#powerrail
      Contact( "PLC_BIT".RUN )
      wire#w4
      Contact( "PLC_BIT".ADD1_FU )
      wire#w5
      I_Contact( "PLC_BIT".NEXT_WADD1 )
      S_Coil( "PLC_BIT".WAD1_FU )
   END_RUNG
   RUNG wire#w4
      { S7_Templates := "SrcType := Real" } EQ_Contact(in1 := "C#4_WD_WEIGHT".SV_SB1, in2 := 0.0)
   END_RUNG wire#w5
   RUNG wire#powerrail
      { S7_Templates := "SrcType := Real" } EQ_Contact(in1 := "C#4_WD_WEIGHT".SV_SB1, in2 := 0.0)
      Coil( "PLC_BIT".NEXT_WADD1 )
   END_RUNG
   RUNG wire#powerrail
      P_Contact(operand := "PLC_BIT".WAD1_EM, bit := "P_WA1_EM")
      wire#w6
      { S7_Templates := "SrcType := Real" } GT_Contact(in1 := "C#7_RD_RUN".SMC_SB1, in2 := "C#7_RD_RUN".SMX_SB1)
      Add(in1 := "C#7_RD_RUN".SMX_SB1, in2 := 1.0, out => "C#7_RD_RUN".SMX_SB1)
   END_RUNG
   RUNG wire#w6
      Move(in := "C#7_RD_RUN".WE_SB1, out1 => "6.4.WADD1".WR_IN)
   END_RUNG
   RUNG wire#w6
      I_Contact( "C#2_WB"."SW_MAN/AUTO" )
      I_Contact( "PLC_BIT".RUN )
      Coil( "LUU TAY ADD1" )
   END_RUNG
   RUNG wire#powerrail
      Contact( "PLC_BIT".WAD1_EM )
      wire#w7
      R_Coil( "PLC_BIT".ADD1_FU )
      R_Coil( "PLC_BIT".WAD1_FU )
   END_RUNG
   RUNG wire#powerrail
      I_Contact( "PLC_BIT".RUN )
   END_RUNG wire#w7
   RUNG wire#powerrail
      P_Contact(operand := "PLC_BIT".WAD1_FU, bit := "P_WADD1_FU")
      wire#w8
      I_Contact( "C#1_RB"."XA W_SB1" )
      { S7_Templates := "SrcType := Real" } EQ_Contact(in1 := "C#7_RD_RUN".SMC_SB1, in2 := "C#7_RD_RUN".SMX_SB1)
      Add(in1 := "C#7_RD_RUN".SMC_SB1, in2 := 1.0, out => "C#7_RD_RUN".SMC_SB1)
   END_RUNG
   RUNG wire#powerrail
      Contact( "P_RUN" )
      Contact( "PLC_BIT".WAD1_FU )
   END_RUNG wire#w8
   // the same network as SCL:
   "6.4.WADD1"(W_IN := "C#7_RD_RUN".WE_SB1,   // "6.WEIGHT_HANDLING"
               WR_IN := "6.4.WADD1".WR_IN,
               PV_IN1 := "C#7_RD_RUN".PV_SB1,
               SV_IN1 := "C#4_WD_WEIGHT".SV_SB1,
               RUN_1 := "7.4.ADD1".STA_RUN,
               EMTY := "PLC_BIT".WAD1_EM,
               W_OUT1 => "6.4.WADD1".W_OUT1,
               "%W_OUT" => "C#7_RD_RUN"."%_WAP1");
   "9.7.DLR_ADD1"(ON := "C#7_RD_RUN".WE_SB1 <= "C#4_WD_WEIGHT"."W_SB1_KL.BRO",   // "9.TIMER_DELAY"
                  CLOCK_1S := "Clock_10Hz",
                  T_DELAY := "9.7.DLR_ADD1".T_DELAY,
                  OUT => "PLC_BIT".WAD1_EM,
                  T_OUT => "9.7.DLR_ADD1".T_OUT,
                  ENO => #_w1);
   IF #_w1 THEN "9.7.DLR_ADD1".T_DELAY := "C#4_WD_WEIGHT"."W_SB1_TG.DLD" + "C#3_WD_SILO".SB1_TG_ODC; END_IF;
   IF "PLC_BIT".RUN AND ("PLC_BIT".ADD1_FU OR ("C#4_WD_WEIGHT".SV_SB1 = 0.0)) AND NOT "PLC_BIT".NEXT_WADD1 THEN
       "PLC_BIT".WAD1_FU := TRUE;
   END_IF;
   "PLC_BIT".NEXT_WADD1 := "C#4_WD_WEIGHT".SV_SB1 = 0.0;
   #_w2 := "PLC_BIT".WAD1_EM AND NOT "P_WA1_EM";   // rising edge of "PLC_BIT".WAD1_EM
   "P_WA1_EM" := "PLC_BIT".WAD1_EM;
   IF #_w2 AND ("C#7_RD_RUN".SMC_SB1 > "C#7_RD_RUN".SMX_SB1) THEN
       "C#7_RD_RUN".SMX_SB1 := "C#7_RD_RUN".SMX_SB1 + 1.0;
   END_IF;
   IF #_w2 THEN "6.4.WADD1".WR_IN := "C#7_RD_RUN".WE_SB1; END_IF;
   "LUU TAY ADD1" := #_w2 AND NOT "C#2_WB"."SW_MAN/AUTO" AND NOT "PLC_BIT".RUN;
   IF "PLC_BIT".WAD1_EM OR NOT "PLC_BIT".RUN THEN
       "PLC_BIT".ADD1_FU := FALSE;
       "PLC_BIT".WAD1_FU := FALSE;
   END_IF;
   #_w3 := "PLC_BIT".WAD1_FU AND NOT "P_WADD1_FU";   // rising edge of "PLC_BIT".WAD1_FU
   "P_WADD1_FU" := "PLC_BIT".WAD1_FU;
   IF (#_w3 OR ("P_RUN" AND "PLC_BIT".WAD1_FU)) AND NOT "C#1_RB"."XA W_SB1" AND ("C#7_RD_RUN".SMC_SB1 = "C#7_RD_RUN".SMX_SB1) THEN
       "C#7_RD_RUN".SMC_SB1 := "C#7_RD_RUN".SMC_SB1 + 1.0;
   END_IF;
END_REGION
END_FUNCTION

FUNCTION "FCCA_CCD_SB1" : Void   // FC18, LAD
{ S7_Optimized_Access := 'TRUE' }
VERSION : 0.1
// stored: AutoNumber true, CodeModifiedDate 2026-01-04T14:27:06.1596668Z, CompileDate 2026-01-04T14:27:06.2063851Z, CreationDate 2024-10-13T15:07:34.9617085Z, HandleErrorsWithinBlock false, InterfaceModifiedDate 2024-08-08T03:53:53.300462Z, IsConsistent true, IsIECCheckEnabled false, IsKnowHowProtected false, IsWriteProtected false, LibraryConformanceStatus Error: The block contains calls of single instances. Warning: The object contains access to global data blocks. Warning: The block contains direct access to inputs, outputs, bit memories, indirect access to the registry or indirect access to external memory areas that are unknown at the time of compilation., ModifiedDate 2026-01-04T14:27:06.1596668Z, ParameterModified 2024-08-08T03:53:53.300462Z, PLCSimAdvancedSupport false, SetENOAutomatically False, StructureModified 2024-08-08T03:53:53.300462Z, UDAEnableTagReadback false
BEGIN

REGION Network 1: CAN PHU GIA 1
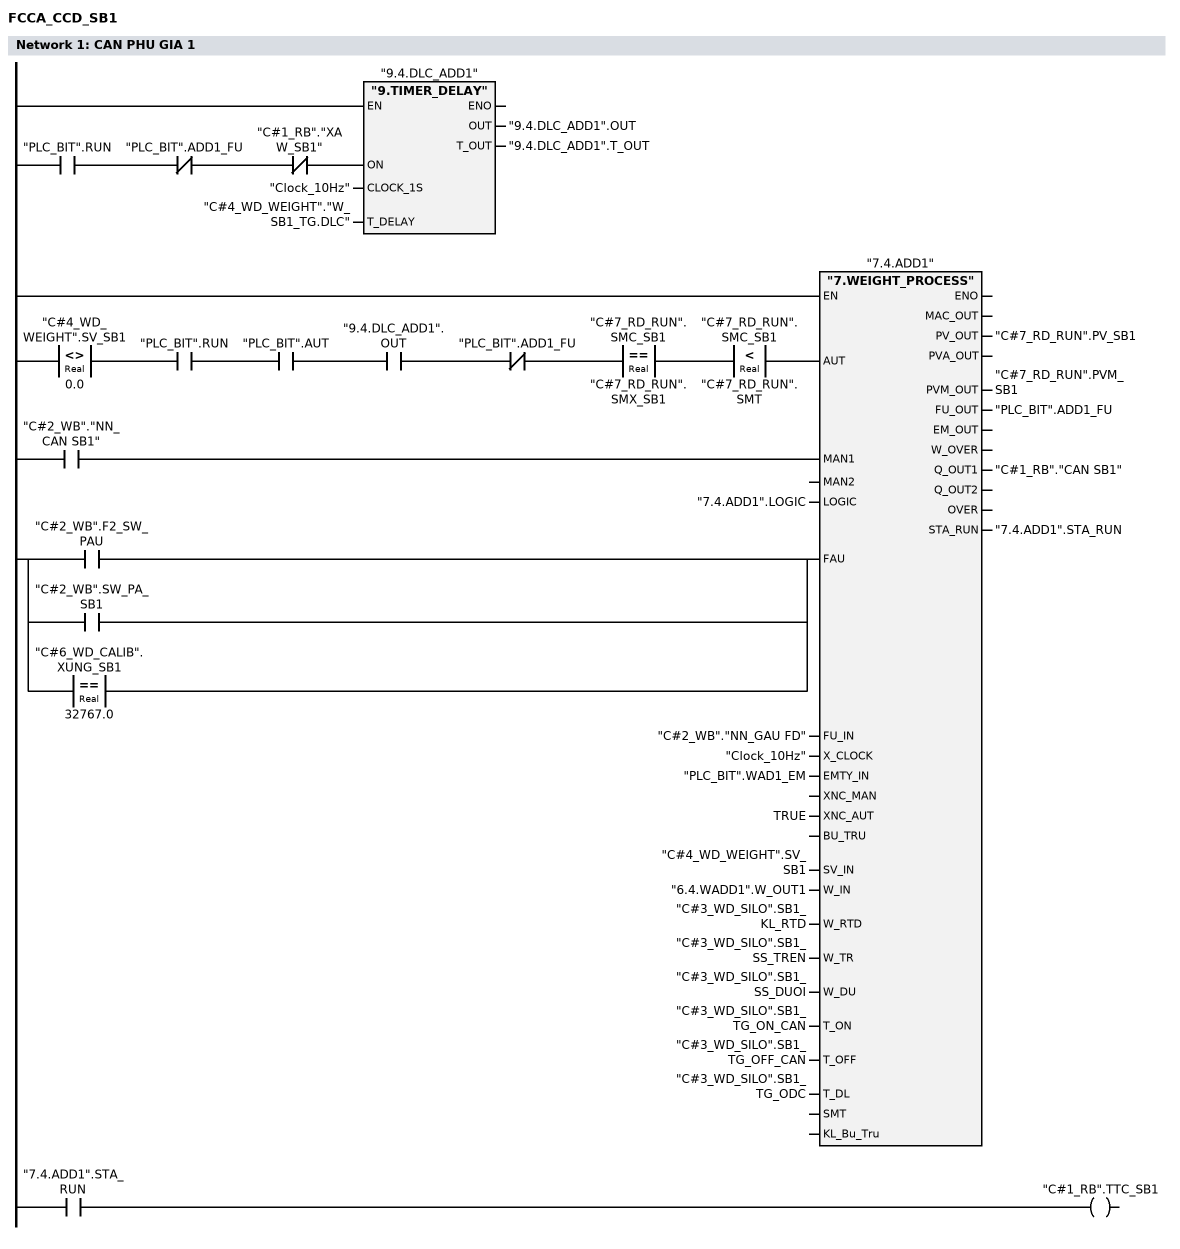
   RUNG wire#powerrail
      "9.4.DLC_ADD1"(ON := wire#w1, CLOCK_1S := "Clock_10Hz", T_DELAY := "C#4_WD_WEIGHT"."W_SB1_TG.DLC", OUT => "9.4.DLC_ADD1".OUT, T_OUT => "9.4.DLC_ADD1".T_OUT)
   END_RUNG
   RUNG wire#powerrail
      Contact( "PLC_BIT".RUN )
      I_Contact( "PLC_BIT".ADD1_FU )
      I_Contact( "C#1_RB"."XA W_SB1" )
   END_RUNG wire#w1
   RUNG wire#powerrail
      "7.4.ADD1"(AUT := wire#w2, MAN1 := wire#w3, FAU := wire#w4, MAN2 :=, LOGIC := "7.4.ADD1".LOGIC, FU_IN := "C#2_WB"."NN_GAU FD", X_CLOCK := "Clock_10Hz", EMTY_IN := "PLC_BIT".WAD1_EM, XNC_MAN :=, XNC_AUT := TRUE, BU_TRU :=, SV_IN := "C#4_WD_WEIGHT".SV_SB1, W_IN := "6.4.WADD1".W_OUT1, W_RTD := "C#3_WD_SILO".SB1_KL_RTD, W_TR := "C#3_WD_SILO".SB1_SS_TREN, W_DU := "C#3_WD_SILO".SB1_SS_DUOI, T_ON := "C#3_WD_SILO".SB1_TG_ON_CAN, T_OFF := "C#3_WD_SILO".SB1_TG_OFF_CAN, T_DL := "C#3_WD_SILO".SB1_TG_ODC, SMT :=, KL_Bu_Tru :=, MAC_OUT =>, PV_OUT => "C#7_RD_RUN".PV_SB1, PVA_OUT =>, PVM_OUT => "C#7_RD_RUN".PVM_SB1, FU_OUT => "PLC_BIT".ADD1_FU, EM_OUT =>, W_OVER =>, Q_OUT1 => "C#1_RB"."CAN SB1", Q_OUT2 =>, OVER =>, STA_RUN => "7.4.ADD1".STA_RUN)
   END_RUNG
   RUNG wire#powerrail
      { S7_Templates := "SrcType := Real" } NE_Contact(in1 := "C#4_WD_WEIGHT".SV_SB1, in2 := 0.0)
      Contact( "PLC_BIT".RUN )
      Contact( "PLC_BIT".AUT )
      Contact( "9.4.DLC_ADD1".OUT )
      I_Contact( "PLC_BIT".ADD1_FU )
      { S7_Templates := "SrcType := Real" } EQ_Contact(in1 := "C#7_RD_RUN".SMC_SB1, in2 := "C#7_RD_RUN".SMX_SB1)
      { S7_Templates := "SrcType := Real" } LT_Contact(in1 := "C#7_RD_RUN".SMC_SB1, in2 := "C#7_RD_RUN".SMT)
   END_RUNG wire#w2
   RUNG wire#powerrail
      Contact( "C#2_WB"."NN_CAN SB1" )
   END_RUNG wire#w3
   RUNG wire#powerrail
      Contact( "C#2_WB".F2_SW_PAU )
   END_RUNG wire#w4
   RUNG wire#powerrail
      Contact( "C#2_WB".SW_PA_SB1 )
   END_RUNG wire#w4
   RUNG wire#powerrail
      { S7_Templates := "SrcType := Real" } EQ_Contact(in1 := "C#6_WD_CALIB".XUNG_SB1, in2 := 32767.0)
   END_RUNG wire#w4
   RUNG wire#powerrail
      Contact( "7.4.ADD1".STA_RUN )
      Coil( "C#1_RB".TTC_SB1 )
   END_RUNG
   // the same network as SCL:
   "9.4.DLC_ADD1"(ON := "PLC_BIT".RUN AND NOT "PLC_BIT".ADD1_FU AND NOT "C#1_RB"."XA W_SB1",   // "9.TIMER_DELAY"
                  CLOCK_1S := "Clock_10Hz",
                  T_DELAY := "C#4_WD_WEIGHT"."W_SB1_TG.DLC",
                  OUT => "9.4.DLC_ADD1".OUT,
                  T_OUT => "9.4.DLC_ADD1".T_OUT);
   "7.4.ADD1"(AUT := ("C#4_WD_WEIGHT".SV_SB1 <> 0.0) AND "PLC_BIT".RUN AND "PLC_BIT".AUT AND "9.4.DLC_ADD1".OUT AND NOT "PLC_BIT".ADD1_FU AND ("C#7_RD_RUN".SMC_SB1 = "C#7_RD_RUN".SMX_SB1) AND ("C#7_RD_RUN".SMC_SB1 < "C#7_RD_RUN".SMT),   // "7.WEIGHT_PROCESS"
              MAN1 := "C#2_WB"."NN_CAN SB1",
              LOGIC := "7.4.ADD1".LOGIC,
              FAU := "C#2_WB".F2_SW_PAU OR "C#2_WB".SW_PA_SB1 OR ("C#6_WD_CALIB".XUNG_SB1 = 32767.0),
              FU_IN := "C#2_WB"."NN_GAU FD",
              X_CLOCK := "Clock_10Hz",
              EMTY_IN := "PLC_BIT".WAD1_EM,
              XNC_AUT := TRUE,
              SV_IN := "C#4_WD_WEIGHT".SV_SB1,
              W_IN := "6.4.WADD1".W_OUT1,
              W_RTD := "C#3_WD_SILO".SB1_KL_RTD,
              W_TR := "C#3_WD_SILO".SB1_SS_TREN,
              W_DU := "C#3_WD_SILO".SB1_SS_DUOI,
              T_ON := "C#3_WD_SILO".SB1_TG_ON_CAN,
              T_OFF := "C#3_WD_SILO".SB1_TG_OFF_CAN,
              T_DL := "C#3_WD_SILO".SB1_TG_ODC,
              PV_OUT => "C#7_RD_RUN".PV_SB1,
              PVM_OUT => "C#7_RD_RUN".PVM_SB1,
              FU_OUT => "PLC_BIT".ADD1_FU,
              Q_OUT1 => "C#1_RB"."CAN SB1",
              STA_RUN => "7.4.ADD1".STA_RUN);
   "C#1_RB".TTC_SB1 := "7.4.ADD1".STA_RUN;
END_REGION
END_FUNCTION

FUNCTION "5. QUA TRINH NAP LIEU" : Void   // FC5, LAD
{ S7_Optimized_Access := 'TRUE' }
VERSION : 0.1
// stored: AutoNumber true, CodeModifiedDate 2026-01-04T14:27:05.1436831Z, CompileDate 2026-01-04T14:27:05.2841536Z, CreationDate 2024-10-14T18:21:08.2031131Z, HandleErrorsWithinBlock false, InterfaceModifiedDate 2023-12-12T15:54:48.677177Z, IsConsistent true, IsIECCheckEnabled false, IsKnowHowProtected false, IsWriteProtected false, LibraryConformanceStatus Warning: The object contains access to global data blocks. Warning: The block contains direct access to inputs, outputs, bit memories, indirect access to the registry or indirect access to external memory areas that are unknown at the time of compilation., ModifiedDate 2026-01-04T14:27:05.1436831Z, ParameterModified 2023-12-12T15:54:48.677177Z, PLCSimAdvancedSupport false, SetENOAutomatically False, StructureModified 2023-12-12T15:54:48.677177Z, UDAEnableTagReadback false
   VAR_OUTPUT
      XA_PTG : Bool;
      XA_CEM1 : Bool;
      XA_CEM2 : Bool;
      XA_WAT1 : Bool;
      XA_WAT2 : Bool;
      XA_ADD1 : Bool;
      XA_ADD2 : Bool;
   END_VAR
BEGIN

REGION Network 1: Van xả phễu chờ
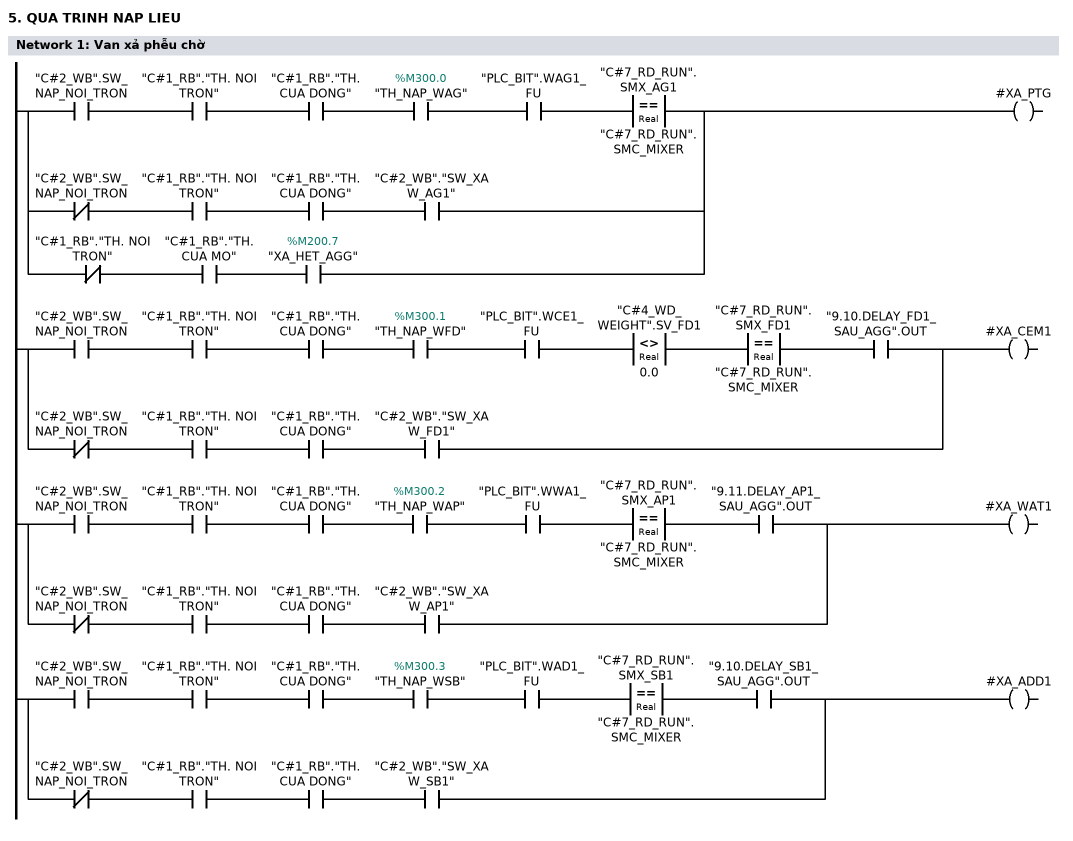
   RUNG wire#powerrail
      Contact( "C#2_WB".SW_NAP_NOI_TRON )
      Contact( "C#1_RB"."TH. NOI TRON" )
      Contact( "C#1_RB"."TH. CUA DONG" )
      Contact( "TH_NAP_WAG" )
      Contact( "PLC_BIT".WAG1_FU )
      { S7_Templates := "SrcType := Real" } EQ_Contact(in1 := "C#7_RD_RUN".SMX_AG1, in2 := "C#7_RD_RUN".SMC_MIXER)
      wire#w1
      Coil( #XA_PTG )
   END_RUNG
   RUNG wire#powerrail
      I_Contact( "C#2_WB".SW_NAP_NOI_TRON )
      Contact( "C#1_RB"."TH. NOI TRON" )
      Contact( "C#1_RB"."TH. CUA DONG" )
      Contact( "C#2_WB"."SW_XA W_AG1" )
   END_RUNG wire#w1
   RUNG wire#powerrail
      I_Contact( "C#1_RB"."TH. NOI TRON" )
      Contact( "C#1_RB"."TH. CUA MO" )
      Contact( "XA_HET_AGG" )
   END_RUNG wire#w1
   RUNG wire#powerrail
      Contact( "C#2_WB".SW_NAP_NOI_TRON )
      Contact( "C#1_RB"."TH. NOI TRON" )
      Contact( "C#1_RB"."TH. CUA DONG" )
      Contact( "TH_NAP_WFD" )
      Contact( "PLC_BIT".WCE1_FU )
      { S7_Templates := "SrcType := Real" } NE_Contact(in1 := "C#4_WD_WEIGHT".SV_FD1, in2 := 0.0)
      { S7_Templates := "SrcType := Real" } EQ_Contact(in1 := "C#7_RD_RUN".SMX_FD1, in2 := "C#7_RD_RUN".SMC_MIXER)
      Contact( "9.10.DELAY_FD1_SAU_AGG".OUT )
      wire#w2
      Coil( #XA_CEM1 )
   END_RUNG
   RUNG wire#powerrail
      I_Contact( "C#2_WB".SW_NAP_NOI_TRON )
      Contact( "C#1_RB"."TH. NOI TRON" )
      Contact( "C#1_RB"."TH. CUA DONG" )
      Contact( "C#2_WB"."SW_XA W_FD1" )
   END_RUNG wire#w2
   RUNG wire#powerrail
      Contact( "C#2_WB".SW_NAP_NOI_TRON )
      Contact( "C#1_RB"."TH. NOI TRON" )
      Contact( "C#1_RB"."TH. CUA DONG" )
      Contact( "TH_NAP_WAP" )
      Contact( "PLC_BIT".WWA1_FU )
      { S7_Templates := "SrcType := Real" } EQ_Contact(in1 := "C#7_RD_RUN".SMX_AP1, in2 := "C#7_RD_RUN".SMC_MIXER)
      Contact( "9.11.DELAY_AP1_SAU_AGG".OUT )
      wire#w3
      Coil( #XA_WAT1 )
   END_RUNG
   RUNG wire#powerrail
      I_Contact( "C#2_WB".SW_NAP_NOI_TRON )
      Contact( "C#1_RB"."TH. NOI TRON" )
      Contact( "C#1_RB"."TH. CUA DONG" )
      Contact( "C#2_WB"."SW_XA W_AP1" )
   END_RUNG wire#w3
   RUNG wire#powerrail
      Contact( "C#2_WB".SW_NAP_NOI_TRON )
      Contact( "C#1_RB"."TH. NOI TRON" )
      Contact( "C#1_RB"."TH. CUA DONG" )
      Contact( "TH_NAP_WSB" )
      Contact( "PLC_BIT".WAD1_FU )
      { S7_Templates := "SrcType := Real" } EQ_Contact(in1 := "C#7_RD_RUN".SMX_SB1, in2 := "C#7_RD_RUN".SMC_MIXER)
      Contact( "9.10.DELAY_SB1_SAU_AGG".OUT )
      wire#w4
      Coil( #XA_ADD1 )
   END_RUNG
   RUNG wire#powerrail
      I_Contact( "C#2_WB".SW_NAP_NOI_TRON )
      Contact( "C#1_RB"."TH. NOI TRON" )
      Contact( "C#1_RB"."TH. CUA DONG" )
      Contact( "C#2_WB"."SW_XA W_SB1" )
   END_RUNG wire#w4
   // the same network as SCL:
   #XA_PTG := ("C#2_WB".SW_NAP_NOI_TRON AND "C#1_RB"."TH. NOI TRON" AND "C#1_RB"."TH. CUA DONG" AND "TH_NAP_WAG" AND "PLC_BIT".WAG1_FU AND ("C#7_RD_RUN".SMX_AG1 = "C#7_RD_RUN".SMC_MIXER)) OR (NOT "C#2_WB".SW_NAP_NOI_TRON AND "C#1_RB"."TH. NOI TRON" AND "C#1_RB"."TH. CUA DONG" AND "C#2_WB"."SW_XA W_AG1") OR (NOT "C#1_RB"."TH. NOI TRON" AND "C#1_RB"."TH. CUA MO" AND "XA_HET_AGG");
   #XA_CEM1 := ("C#2_WB".SW_NAP_NOI_TRON AND "C#1_RB"."TH. NOI TRON" AND "C#1_RB"."TH. CUA DONG" AND "TH_NAP_WFD" AND "PLC_BIT".WCE1_FU AND ("C#4_WD_WEIGHT".SV_FD1 <> 0.0) AND ("C#7_RD_RUN".SMX_FD1 = "C#7_RD_RUN".SMC_MIXER) AND "9.10.DELAY_FD1_SAU_AGG".OUT) OR (NOT "C#2_WB".SW_NAP_NOI_TRON AND "C#1_RB"."TH. NOI TRON" AND "C#1_RB"."TH. CUA DONG" AND "C#2_WB"."SW_XA W_FD1");
   #XA_WAT1 := ("C#2_WB".SW_NAP_NOI_TRON AND "C#1_RB"."TH. NOI TRON" AND "C#1_RB"."TH. CUA DONG" AND "TH_NAP_WAP" AND "PLC_BIT".WWA1_FU AND ("C#7_RD_RUN".SMX_AP1 = "C#7_RD_RUN".SMC_MIXER) AND "9.11.DELAY_AP1_SAU_AGG".OUT) OR (NOT "C#2_WB".SW_NAP_NOI_TRON AND "C#1_RB"."TH. NOI TRON" AND "C#1_RB"."TH. CUA DONG" AND "C#2_WB"."SW_XA W_AP1");
   #XA_ADD1 := ("C#2_WB".SW_NAP_NOI_TRON AND "C#1_RB"."TH. NOI TRON" AND "C#1_RB"."TH. CUA DONG" AND "TH_NAP_WSB" AND "PLC_BIT".WAD1_FU AND ("C#7_RD_RUN".SMX_SB1 = "C#7_RD_RUN".SMC_MIXER) AND "9.10.DELAY_SB1_SAU_AGG".OUT) OR (NOT "C#2_WB".SW_NAP_NOI_TRON AND "C#1_RB"."TH. NOI TRON" AND "C#1_RB"."TH. CUA DONG" AND "C#2_WB"."SW_XA W_SB1");
END_REGION
END_FUNCTION

FUNCTION "7. SAVE_REPORT" : Void   // FC7, LAD
{ S7_Optimized_Access := 'TRUE' }
VERSION : 0.1
// stored: AutoNumber false, CodeModifiedDate 2026-01-04T14:27:05.3313004Z, CompileDate 2026-01-04T14:27:05.4091731Z, CreationDate 2024-10-14T18:51:22.4750735Z, HandleErrorsWithinBlock false, InterfaceModifiedDate 2023-12-15T06:44:57.8941631Z, IsConsistent true, IsIECCheckEnabled false, IsKnowHowProtected false, IsWriteProtected false, LibraryConformanceStatus Warning: The object contains access to global data blocks. Warning: The block contains direct access to inputs, outputs, bit memories, indirect access to the registry or indirect access to external memory areas that are unknown at the time of compilation., ModifiedDate 2026-01-04T14:27:05.3313004Z, ParameterModified 2023-12-15T06:44:57.8941631Z, PLCSimAdvancedSupport false, SetENOAutomatically False, StructureModified 2023-12-15T06:44:57.8941631Z, UDAEnableTagReadback false
   VAR_TEMP   // added for the SCL form of the ladder/FBD networks
      _w1 : Bool;
   END_VAR
BEGIN

REGION Network 1: Lưu dữ liệu Cốt liệu
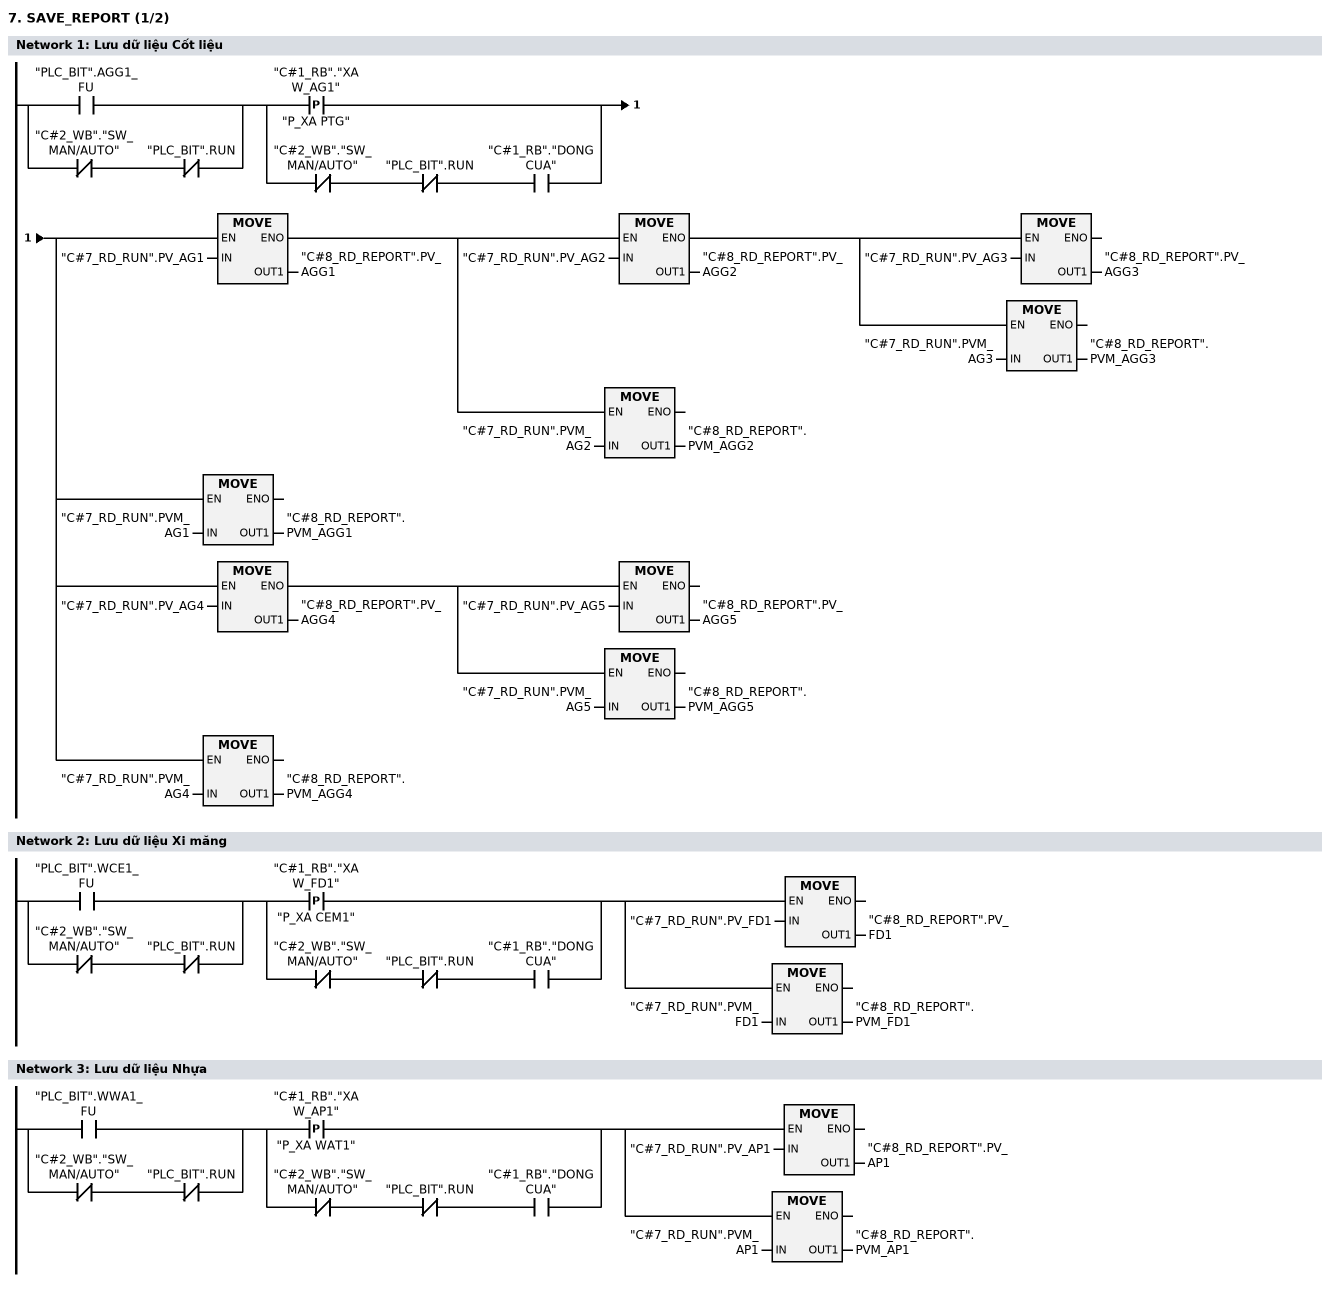
   RUNG wire#powerrail
      Contact( "PLC_BIT".AGG1_FU )
      wire#w1
      P_Contact(operand := "C#1_RB"."XA W_AG1", bit := "P_XA PTG")
      wire#w2
      Move(in := "C#7_RD_RUN".PV_AG1, out1 => "C#8_RD_REPORT".PV_AGG1)
      wire#w3
      Move(in := "C#7_RD_RUN".PV_AG2, out1 => "C#8_RD_REPORT".PV_AGG2)
      wire#w4
      Move(in := "C#7_RD_RUN".PV_AG3, out1 => "C#8_RD_REPORT".PV_AGG3)
   END_RUNG
   RUNG wire#powerrail
      I_Contact( "C#2_WB"."SW_MAN/AUTO" )
      I_Contact( "PLC_BIT".RUN )
   END_RUNG wire#w1
   RUNG wire#w1
      I_Contact( "C#2_WB"."SW_MAN/AUTO" )
      I_Contact( "PLC_BIT".RUN )
      Contact( "C#1_RB"."DONG CUA" )
   END_RUNG wire#w2
   RUNG wire#w4
      Move(in := "C#7_RD_RUN".PVM_AG3, out1 => "C#8_RD_REPORT".PVM_AGG3)
   END_RUNG
   RUNG wire#w3
      Move(in := "C#7_RD_RUN".PVM_AG2, out1 => "C#8_RD_REPORT".PVM_AGG2)
   END_RUNG
   RUNG wire#w2
      Move(in := "C#7_RD_RUN".PVM_AG1, out1 => "C#8_RD_REPORT".PVM_AGG1)
   END_RUNG
   RUNG wire#w2
      Move(in := "C#7_RD_RUN".PV_AG4, out1 => "C#8_RD_REPORT".PV_AGG4)
      wire#w5
      Move(in := "C#7_RD_RUN".PV_AG5, out1 => "C#8_RD_REPORT".PV_AGG5)
   END_RUNG
   RUNG wire#w5
      Move(in := "C#7_RD_RUN".PVM_AG5, out1 => "C#8_RD_REPORT".PVM_AGG5)
   END_RUNG
   RUNG wire#w2
      Move(in := "C#7_RD_RUN".PVM_AG4, out1 => "C#8_RD_REPORT".PVM_AGG4)
   END_RUNG
   // the same network as SCL:
   #_w1 := ("PLC_BIT".AGG1_FU OR (NOT "C#2_WB"."SW_MAN/AUTO" AND NOT "PLC_BIT".RUN)) AND "C#1_RB"."XA W_AG1" AND NOT "P_XA PTG";   // rising edge of "C#1_RB"."XA W_AG1"
   "P_XA PTG" := "C#1_RB"."XA W_AG1";
   IF #_w1 OR (("PLC_BIT".AGG1_FU OR (NOT "C#2_WB"."SW_MAN/AUTO" AND NOT "PLC_BIT".RUN)) AND NOT "C#2_WB"."SW_MAN/AUTO" AND NOT "PLC_BIT".RUN AND "C#1_RB"."DONG CUA") THEN
       "C#8_RD_REPORT".PV_AGG1 := "C#7_RD_RUN".PV_AG1;
       "C#8_RD_REPORT".PV_AGG2 := "C#7_RD_RUN".PV_AG2;
       "C#8_RD_REPORT".PV_AGG3 := "C#7_RD_RUN".PV_AG3;
       "C#8_RD_REPORT".PVM_AGG3 := "C#7_RD_RUN".PVM_AG3;
       "C#8_RD_REPORT".PVM_AGG2 := "C#7_RD_RUN".PVM_AG2;
       "C#8_RD_REPORT".PVM_AGG1 := "C#7_RD_RUN".PVM_AG1;
       "C#8_RD_REPORT".PV_AGG4 := "C#7_RD_RUN".PV_AG4;
       "C#8_RD_REPORT".PV_AGG5 := "C#7_RD_RUN".PV_AG5;
       "C#8_RD_REPORT".PVM_AGG5 := "C#7_RD_RUN".PVM_AG5;
       "C#8_RD_REPORT".PVM_AGG4 := "C#7_RD_RUN".PVM_AG4;
   END_IF;
END_REGION

REGION Network 2: Lưu dữ liệu Xi măng
   RUNG wire#powerrail
      Contact( "PLC_BIT".WCE1_FU )
      wire#w1
      P_Contact(operand := "C#1_RB"."XA W_FD1", bit := "P_XA CEM1")
      wire#w2
      Move(in := "C#7_RD_RUN".PV_FD1, out1 => "C#8_RD_REPORT".PV_FD1)
   END_RUNG
   RUNG wire#powerrail
      I_Contact( "C#2_WB"."SW_MAN/AUTO" )
      I_Contact( "PLC_BIT".RUN )
   END_RUNG wire#w1
   RUNG wire#w1
      I_Contact( "C#2_WB"."SW_MAN/AUTO" )
      I_Contact( "PLC_BIT".RUN )
      Contact( "C#1_RB"."DONG CUA" )
   END_RUNG wire#w2
   RUNG wire#w2
      Move(in := "C#7_RD_RUN".PVM_FD1, out1 => "C#8_RD_REPORT".PVM_FD1)
   END_RUNG
   // the same network as SCL:
   #_w1 := ("PLC_BIT".WCE1_FU OR (NOT "C#2_WB"."SW_MAN/AUTO" AND NOT "PLC_BIT".RUN)) AND "C#1_RB"."XA W_FD1" AND NOT "P_XA CEM1";   // rising edge of "C#1_RB"."XA W_FD1"
   "P_XA CEM1" := "C#1_RB"."XA W_FD1";
   IF #_w1 OR (("PLC_BIT".WCE1_FU OR (NOT "C#2_WB"."SW_MAN/AUTO" AND NOT "PLC_BIT".RUN)) AND NOT "C#2_WB"."SW_MAN/AUTO" AND NOT "PLC_BIT".RUN AND "C#1_RB"."DONG CUA") THEN
       "C#8_RD_REPORT".PV_FD1 := "C#7_RD_RUN".PV_FD1;
       "C#8_RD_REPORT".PVM_FD1 := "C#7_RD_RUN".PVM_FD1;
   END_IF;
END_REGION

REGION Network 3: Lưu dữ liệu Nhựa
   RUNG wire#powerrail
      Contact( "PLC_BIT".WWA1_FU )
      wire#w1
      P_Contact(operand := "C#1_RB"."XA W_AP1", bit := "P_XA WAT1")
      wire#w2
      Move(in := "C#7_RD_RUN".PV_AP1, out1 => "C#8_RD_REPORT".PV_AP1)
   END_RUNG
   RUNG wire#powerrail
      I_Contact( "C#2_WB"."SW_MAN/AUTO" )
      I_Contact( "PLC_BIT".RUN )
   END_RUNG wire#w1
   RUNG wire#w1
      I_Contact( "C#2_WB"."SW_MAN/AUTO" )
      I_Contact( "PLC_BIT".RUN )
      Contact( "C#1_RB"."DONG CUA" )
   END_RUNG wire#w2
   RUNG wire#w2
      Move(in := "C#7_RD_RUN".PVM_AP1, out1 => "C#8_RD_REPORT".PVM_AP1)
   END_RUNG
   // the same network as SCL:
   #_w1 := ("PLC_BIT".WWA1_FU OR (NOT "C#2_WB"."SW_MAN/AUTO" AND NOT "PLC_BIT".RUN)) AND "C#1_RB"."XA W_AP1" AND NOT "P_XA WAT1";   // rising edge of "C#1_RB"."XA W_AP1"
   "P_XA WAT1" := "C#1_RB"."XA W_AP1";
   IF #_w1 OR (("PLC_BIT".WWA1_FU OR (NOT "C#2_WB"."SW_MAN/AUTO" AND NOT "PLC_BIT".RUN)) AND NOT "C#2_WB"."SW_MAN/AUTO" AND NOT "PLC_BIT".RUN AND "C#1_RB"."DONG CUA") THEN
       "C#8_RD_REPORT".PV_AP1 := "C#7_RD_RUN".PV_AP1;
       "C#8_RD_REPORT".PVM_AP1 := "C#7_RD_RUN".PVM_AP1;
   END_IF;
END_REGION

REGION Network 4: Lưu dữ liệu Phụ gia SBS
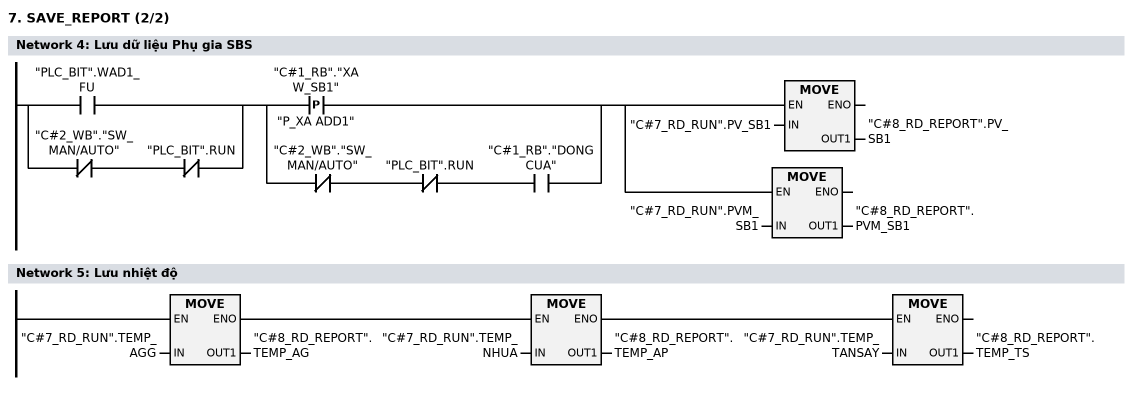
   RUNG wire#powerrail
      Contact( "PLC_BIT".WAD1_FU )
      wire#w1
      P_Contact(operand := "C#1_RB"."XA W_SB1", bit := "P_XA ADD1")
      wire#w2
      Move(in := "C#7_RD_RUN".PV_SB1, out1 => "C#8_RD_REPORT".PV_SB1)
   END_RUNG
   RUNG wire#powerrail
      I_Contact( "C#2_WB"."SW_MAN/AUTO" )
      I_Contact( "PLC_BIT".RUN )
   END_RUNG wire#w1
   RUNG wire#w1
      I_Contact( "C#2_WB"."SW_MAN/AUTO" )
      I_Contact( "PLC_BIT".RUN )
      Contact( "C#1_RB"."DONG CUA" )
   END_RUNG wire#w2
   RUNG wire#w2
      Move(in := "C#7_RD_RUN".PVM_SB1, out1 => "C#8_RD_REPORT".PVM_SB1)
   END_RUNG
   // the same network as SCL:
   #_w1 := ("PLC_BIT".WAD1_FU OR (NOT "C#2_WB"."SW_MAN/AUTO" AND NOT "PLC_BIT".RUN)) AND "C#1_RB"."XA W_SB1" AND NOT "P_XA ADD1";   // rising edge of "C#1_RB"."XA W_SB1"
   "P_XA ADD1" := "C#1_RB"."XA W_SB1";
   IF #_w1 OR (("PLC_BIT".WAD1_FU OR (NOT "C#2_WB"."SW_MAN/AUTO" AND NOT "PLC_BIT".RUN)) AND NOT "C#2_WB"."SW_MAN/AUTO" AND NOT "PLC_BIT".RUN AND "C#1_RB"."DONG CUA") THEN
       "C#8_RD_REPORT".PV_SB1 := "C#7_RD_RUN".PV_SB1;
       "C#8_RD_REPORT".PVM_SB1 := "C#7_RD_RUN".PVM_SB1;
   END_IF;
END_REGION

REGION Network 5: Lưu nhiệt độ
   RUNG wire#powerrail
      Move(in := "C#7_RD_RUN".TEMP_AGG, out1 => "C#8_RD_REPORT".TEMP_AG)
      Move(in := "C#7_RD_RUN".TEMP_NHUA, out1 => "C#8_RD_REPORT".TEMP_AP)
      Move(in := "C#7_RD_RUN".TEMP_TANSAY, out1 => "C#8_RD_REPORT".TEMP_TS)
   END_RUNG
   // the same network as SCL:
   "C#8_RD_REPORT".TEMP_AG := "C#7_RD_RUN".TEMP_AGG;
   "C#8_RD_REPORT".TEMP_AP := "C#7_RD_RUN".TEMP_NHUA;
   "C#8_RD_REPORT".TEMP_TS := "C#7_RD_RUN".TEMP_TANSAY;
END_REGION
END_FUNCTION

ORGANIZATION_BLOCK "Main"   // OB123, LAD, ProgramCycle
TITLE = "Main Program Sweep (Cycle)"
{ S7_Optimized_Access := 'TRUE' }
VERSION : 0.1
// stored: AutoNumber true, CodeModifiedDate 2026-01-15T16:25:55.6274482Z, CompileDate 2026-01-15T16:25:55.6406611Z, ConstantName OB_Main, CreationDate 2026-01-15T16:14:49.4586784Z, EventClass Program cycle, HandleErrorsWithinBlock false, InterfaceModifiedDate 2026-01-15T16:25:47.5430699Z, IsConsistent true, IsIECCheckEnabled false, IsKnowHowProtected false, IsWriteProtected false, ModifiedDate 2026-01-15T16:25:55.6274482Z, ParameterModified 2008-07-21T16:55:08.419547Z, PLCSimAdvancedSupport false, PriorityNumber 1, ProcessImagePartNumber 65535, SetENOAutomatically False, StructureModified 2008-07-21T16:55:08.419547Z
   VAR_INPUT
      Initial_Call : Bool;   // Initial call of this OB
      Remanence : Bool;   // =True, if remanent data are available
   END_VAR
BEGIN
END_ORGANIZATION_BLOCK

FUNCTION_BLOCK "10.TIMER_CLOCK"   // FB10, LAD
{ S7_Optimized_Access := 'TRUE' }
VERSION : 0.1
// stored: AutoNumber false, CodeModifiedDate 2025-08-27T17:13:37.9521369Z, CompileDate 2025-08-30T17:40:34.6172449Z, CreationDate 2024-10-12T12:36:08.0193576Z, DownloadWithoutReinit false, HandleErrorsWithinBlock false, InterfaceModifiedDate 2023-08-14T08:08:19.3737097Z, IsConsistent true, IsIECCheckEnabled false, IsKnowHowProtected false, IsRetainMemResEnabled false, IsWriteProtected false, LibraryConformanceStatus The object is library-conformant., MemoryReserve 100, ModifiedDate 2025-08-27T17:13:37.9521369Z, ParameterModified 2022-05-24T16:04:05.0982286Z, PLCSimAdvancedSupport false, SetENOAutomatically False, StructureModified 2023-08-14T08:08:19.3737097Z, UDAEnableTagReadback false
   VAR_INPUT
      ON : Bool;
      CLOCK_1S : Bool;
      T_ON : Real;
      T_OFF : Real;
   END_VAR
   VAR_OUTPUT
      OUT : Bool;
   END_VAR
   VAR RETAIN
      TON : Real;
      TOFF : Real;
   END_VAR
   VAR
      CLK1 : Bool;
   END_VAR
   VAR_TEMP   // added for the SCL form of the ladder/FBD networks
      _w1 : Bool;
   END_VAR
BEGIN

REGION Network 1
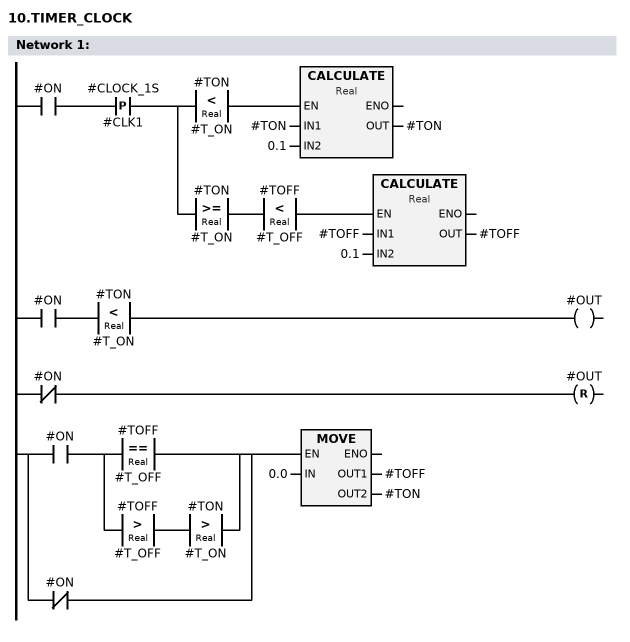
   RUNG wire#powerrail
      Contact( #ON )
      P_Contact(operand := #CLOCK_1S, bit := #CLK1)
      wire#w1
      { S7_Templates := "SrcType := Real" } LT_Contact(in1 := #TON, in2 := #T_ON)
      { S7_Templates := "SrcType := Real"; S7_Expression := "IN1+IN2" } Calculate(in1 := #TON, in2 := 0.1, out => #TON)
   END_RUNG
   RUNG wire#w1
      { S7_Templates := "SrcType := Real" } GE_Contact(in1 := #TON, in2 := #T_ON)
      { S7_Templates := "SrcType := Real" } LT_Contact(in1 := #TOFF, in2 := #T_OFF)
      { S7_Templates := "SrcType := Real"; S7_Expression := "IN1+IN2" } Calculate(in1 := #TOFF, in2 := 0.1, out => #TOFF)
   END_RUNG
   RUNG wire#powerrail
      Contact( #ON )
      { S7_Templates := "SrcType := Real" } LT_Contact(in1 := #TON, in2 := #T_ON)
      Coil( #OUT )
   END_RUNG
   RUNG wire#powerrail
      I_Contact( #ON )
      R_Coil( #OUT )
   END_RUNG
   RUNG wire#powerrail
      Contact( #ON )
      wire#w2
      { S7_Templates := "SrcType := Real" } EQ_Contact(in1 := #TOFF, in2 := #T_OFF)
      wire#w3
      Move(in := 0.0, out1 => #TOFF, out2 => #TON)
   END_RUNG
   RUNG wire#w2
      { S7_Templates := "SrcType := Real" } GT_Contact(in1 := #TOFF, in2 := #T_OFF)
      { S7_Templates := "SrcType := Real" } GT_Contact(in1 := #TON, in2 := #T_ON)
   END_RUNG wire#w3
   RUNG wire#powerrail
      I_Contact( #ON )
   END_RUNG wire#w3
   // the same network as SCL:
   #_w1 := #ON AND #CLOCK_1S AND NOT #CLK1;   // rising edge of #CLOCK_1S
   #CLK1 := #CLOCK_1S;
   IF #_w1 AND (#TON < #T_ON) THEN #TON := #TON+0.1; END_IF;
   IF #_w1 AND (#TON >= #T_ON) AND (#TOFF < #T_OFF) THEN #TOFF := #TOFF+0.1; END_IF;
   #OUT := #ON AND (#TON < #T_ON);
   IF NOT #ON THEN #OUT := FALSE; END_IF;
   IF (#ON AND ((#TOFF = #T_OFF) OR ((#TOFF > #T_OFF) AND (#TON > #T_ON)))) OR NOT #ON THEN
       #TOFF := 0.0;
       #TON := 0.0;
   END_IF;
END_REGION
END_FUNCTION_BLOCK

FUNCTION_BLOCK "11. LOGIC CAN"   // FB11, LAD
{ S7_Optimized_Access := 'TRUE' }
VERSION : 0.1
// stored: AutoNumber true, CodeModifiedDate 2025-08-27T17:14:05.4937984Z, CompileDate 2025-08-30T17:40:35.0335687Z, CreationDate 2024-10-12T12:36:08.0193576Z, DownloadWithoutReinit false, HandleErrorsWithinBlock false, InterfaceModifiedDate 2023-12-21T19:23:23.4270206Z, IsConsistent true, IsIECCheckEnabled false, IsKnowHowProtected false, IsRetainMemResEnabled false, IsWriteProtected false, LibraryConformanceStatus The object is library-conformant., MemoryReserve 100, ModifiedDate 2025-08-27T17:14:05.4937984Z, ParameterModified 2023-12-21T19:23:23.4270206Z, PLCSimAdvancedSupport false, SetENOAutomatically False, StructureModified 2023-12-21T19:23:23.4270206Z, UDAEnableTagReadback false
   VAR_INPUT
      LOGIC_1 : Real;
      LOGIC_2 : Real;
      LOGIC_3 : Real;
      "THC_1.1" : Bool;
      "THC_1.2" : Bool;
      "THC_2.1" : Bool;
      "THC_2.2" : Bool;
      "THC_3.1" : Bool;
      "THC_3.2" : Bool;
      "THC_4.1" : Bool;
      "THC_4.2" : Bool;
      "THC_5.1" : Bool;
      "THC_5.2" : Bool;
      "THC_6.1" : Bool;
      "THC_6.2" : Bool;
   END_VAR
   VAR_OUTPUT
      "OUT_LGOIC_1.1" : Bool;
      "OUT_LGOIC_1.2" : Bool;
      "OUT_LGOIC_2.1" : Bool;
      "OUT_LGOIC_2.2" : Bool;
      "OUT_LGOIC_3.1" : Bool;
      "OUT_LGOIC_3.2" : Bool;
      "OUT_LGOIC_4.1" : Bool;
      "OUT_LGOIC_4.2" : Bool;
      "OUT_LGOIC_5.1" : Bool;
      "OUT_LGOIC_5.2" : Bool;
      "OUT_LGOIC_6.1" : Bool;
      "OUT_LGOIC_6.2" : Bool;
   END_VAR
BEGIN

REGION Network 1: OUT1
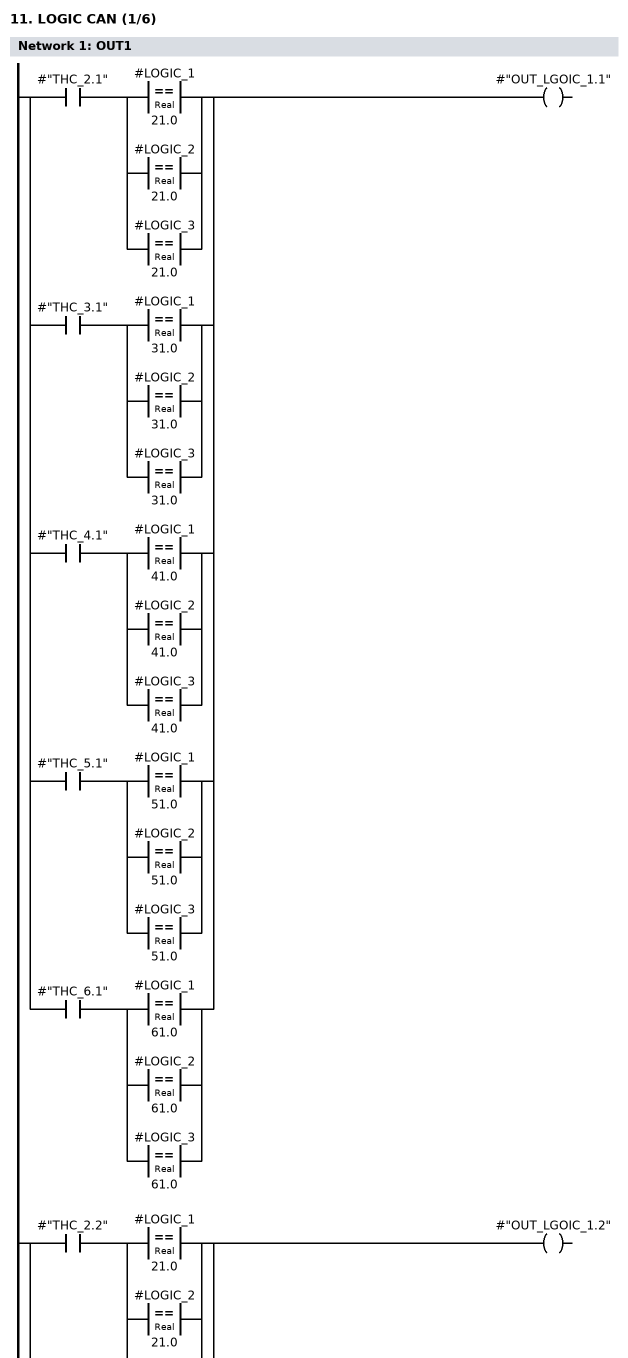
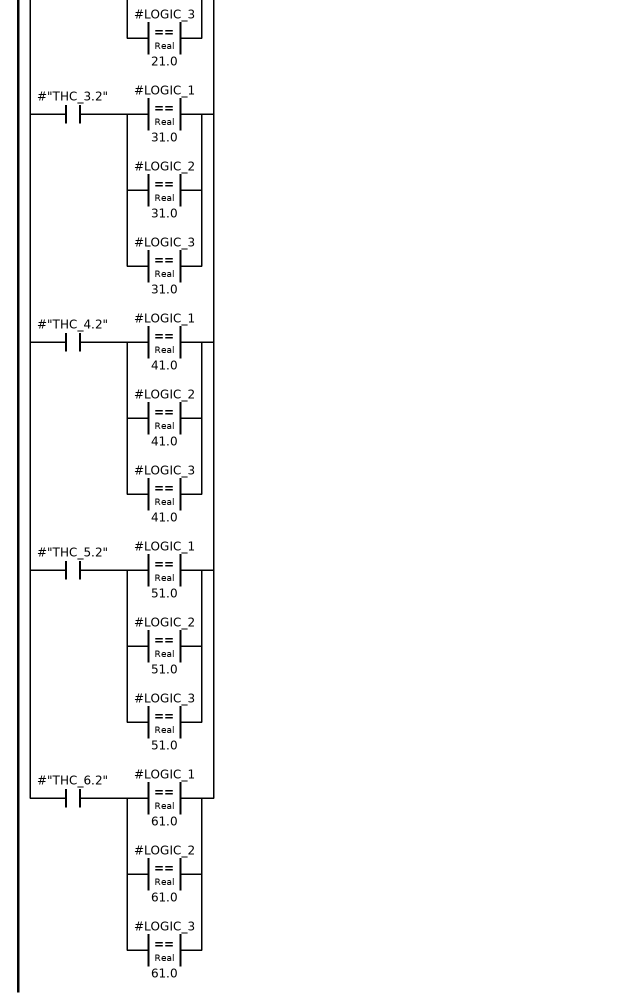
   RUNG wire#powerrail
      Contact( #"THC_2.1" )
      wire#w1
      { S7_Templates := "SrcType := Real" } EQ_Contact(in1 := #LOGIC_1, in2 := 21.0)
      wire#w2
      Coil( #"OUT_LGOIC_1.1" )
   END_RUNG
   RUNG wire#w1
      { S7_Templates := "SrcType := Real" } EQ_Contact(in1 := #LOGIC_2, in2 := 21.0)
   END_RUNG wire#w2
   RUNG wire#w1
      { S7_Templates := "SrcType := Real" } EQ_Contact(in1 := #LOGIC_3, in2 := 21.0)
   END_RUNG wire#w2
   RUNG wire#powerrail
      Contact( #"THC_3.1" )
      wire#w3
      { S7_Templates := "SrcType := Real" } EQ_Contact(in1 := #LOGIC_1, in2 := 31.0)
   END_RUNG wire#w2
   RUNG wire#w3
      { S7_Templates := "SrcType := Real" } EQ_Contact(in1 := #LOGIC_2, in2 := 31.0)
   END_RUNG wire#w2
   RUNG wire#w3
      { S7_Templates := "SrcType := Real" } EQ_Contact(in1 := #LOGIC_3, in2 := 31.0)
   END_RUNG wire#w2
   RUNG wire#powerrail
      Contact( #"THC_4.1" )
      wire#w4
      { S7_Templates := "SrcType := Real" } EQ_Contact(in1 := #LOGIC_1, in2 := 41.0)
   END_RUNG wire#w2
   RUNG wire#w4
      { S7_Templates := "SrcType := Real" } EQ_Contact(in1 := #LOGIC_2, in2 := 41.0)
   END_RUNG wire#w2
   RUNG wire#w4
      { S7_Templates := "SrcType := Real" } EQ_Contact(in1 := #LOGIC_3, in2 := 41.0)
   END_RUNG wire#w2
   RUNG wire#powerrail
      Contact( #"THC_5.1" )
      wire#w5
      { S7_Templates := "SrcType := Real" } EQ_Contact(in1 := #LOGIC_1, in2 := 51.0)
   END_RUNG wire#w2
   RUNG wire#w5
      { S7_Templates := "SrcType := Real" } EQ_Contact(in1 := #LOGIC_2, in2 := 51.0)
   END_RUNG wire#w2
   RUNG wire#w5
      { S7_Templates := "SrcType := Real" } EQ_Contact(in1 := #LOGIC_3, in2 := 51.0)
   END_RUNG wire#w2
   RUNG wire#powerrail
      Contact( #"THC_6.1" )
      wire#w6
      { S7_Templates := "SrcType := Real" } EQ_Contact(in1 := #LOGIC_1, in2 := 61.0)
   END_RUNG wire#w2
   RUNG wire#w6
      { S7_Templates := "SrcType := Real" } EQ_Contact(in1 := #LOGIC_2, in2 := 61.0)
   END_RUNG wire#w2
   RUNG wire#w6
      { S7_Templates := "SrcType := Real" } EQ_Contact(in1 := #LOGIC_3, in2 := 61.0)
   END_RUNG wire#w2
   RUNG wire#powerrail
      Contact( #"THC_2.2" )
      wire#w7
      { S7_Templates := "SrcType := Real" } EQ_Contact(in1 := #LOGIC_1, in2 := 21.0)
      wire#w8
      Coil( #"OUT_LGOIC_1.2" )
   END_RUNG
   RUNG wire#w7
      { S7_Templates := "SrcType := Real" } EQ_Contact(in1 := #LOGIC_2, in2 := 21.0)
   END_RUNG wire#w8
   RUNG wire#w7
      { S7_Templates := "SrcType := Real" } EQ_Contact(in1 := #LOGIC_3, in2 := 21.0)
   END_RUNG wire#w8
   RUNG wire#powerrail
      Contact( #"THC_3.2" )
      wire#w9
      { S7_Templates := "SrcType := Real" } EQ_Contact(in1 := #LOGIC_1, in2 := 31.0)
   END_RUNG wire#w8
   RUNG wire#w9
      { S7_Templates := "SrcType := Real" } EQ_Contact(in1 := #LOGIC_2, in2 := 31.0)
   END_RUNG wire#w8
   RUNG wire#w9
      { S7_Templates := "SrcType := Real" } EQ_Contact(in1 := #LOGIC_3, in2 := 31.0)
   END_RUNG wire#w8
   RUNG wire#powerrail
      Contact( #"THC_4.2" )
      wire#w10
      { S7_Templates := "SrcType := Real" } EQ_Contact(in1 := #LOGIC_1, in2 := 41.0)
   END_RUNG wire#w8
   RUNG wire#w10
      { S7_Templates := "SrcType := Real" } EQ_Contact(in1 := #LOGIC_2, in2 := 41.0)
   END_RUNG wire#w8
   RUNG wire#w10
      { S7_Templates := "SrcType := Real" } EQ_Contact(in1 := #LOGIC_3, in2 := 41.0)
   END_RUNG wire#w8
   RUNG wire#powerrail
      Contact( #"THC_5.2" )
      wire#w11
      { S7_Templates := "SrcType := Real" } EQ_Contact(in1 := #LOGIC_1, in2 := 51.0)
   END_RUNG wire#w8
   RUNG wire#w11
      { S7_Templates := "SrcType := Real" } EQ_Contact(in1 := #LOGIC_2, in2 := 51.0)
   END_RUNG wire#w8
   RUNG wire#w11
      { S7_Templates := "SrcType := Real" } EQ_Contact(in1 := #LOGIC_3, in2 := 51.0)
   END_RUNG wire#w8
   RUNG wire#powerrail
      Contact( #"THC_6.2" )
      wire#w12
      { S7_Templates := "SrcType := Real" } EQ_Contact(in1 := #LOGIC_1, in2 := 61.0)
   END_RUNG wire#w8
   RUNG wire#w12
      { S7_Templates := "SrcType := Real" } EQ_Contact(in1 := #LOGIC_2, in2 := 61.0)
   END_RUNG wire#w8
   RUNG wire#w12
      { S7_Templates := "SrcType := Real" } EQ_Contact(in1 := #LOGIC_3, in2 := 61.0)
   END_RUNG wire#w8
   // the same network as SCL:
   #"OUT_LGOIC_1.1" := (#"THC_2.1" AND ((#LOGIC_1 = 21.0) OR (#LOGIC_2 = 21.0) OR (#LOGIC_3 = 21.0))) OR (#"THC_3.1" AND ((#LOGIC_1 = 31.0) OR (#LOGIC_2 = 31.0) OR (#LOGIC_3 = 31.0))) OR (#"THC_4.1" AND ((#LOGIC_1 = 41.0) OR (#LOGIC_2 = 41.0) OR (#LOGIC_3 = 41.0))) OR (#"THC_5.1" AND ((#LOGIC_1 = 51.0) OR (#LOGIC_2 = 51.0) OR (#LOGIC_3 = 51.0))) OR (#"THC_6.1" AND ((#LOGIC_1 = 61.0) OR (#LOGIC_2 = 61.0) OR (#LOGIC_3 = 61.0)));
   #"OUT_LGOIC_1.2" := (#"THC_2.2" AND ((#LOGIC_1 = 21.0) OR (#LOGIC_2 = 21.0) OR (#LOGIC_3 = 21.0))) OR (#"THC_3.2" AND ((#LOGIC_1 = 31.0) OR (#LOGIC_2 = 31.0) OR (#LOGIC_3 = 31.0))) OR (#"THC_4.2" AND ((#LOGIC_1 = 41.0) OR (#LOGIC_2 = 41.0) OR (#LOGIC_3 = 41.0))) OR (#"THC_5.2" AND ((#LOGIC_1 = 51.0) OR (#LOGIC_2 = 51.0) OR (#LOGIC_3 = 51.0))) OR (#"THC_6.2" AND ((#LOGIC_1 = 61.0) OR (#LOGIC_2 = 61.0) OR (#LOGIC_3 = 61.0)));
END_REGION

REGION Network 2: OUT2
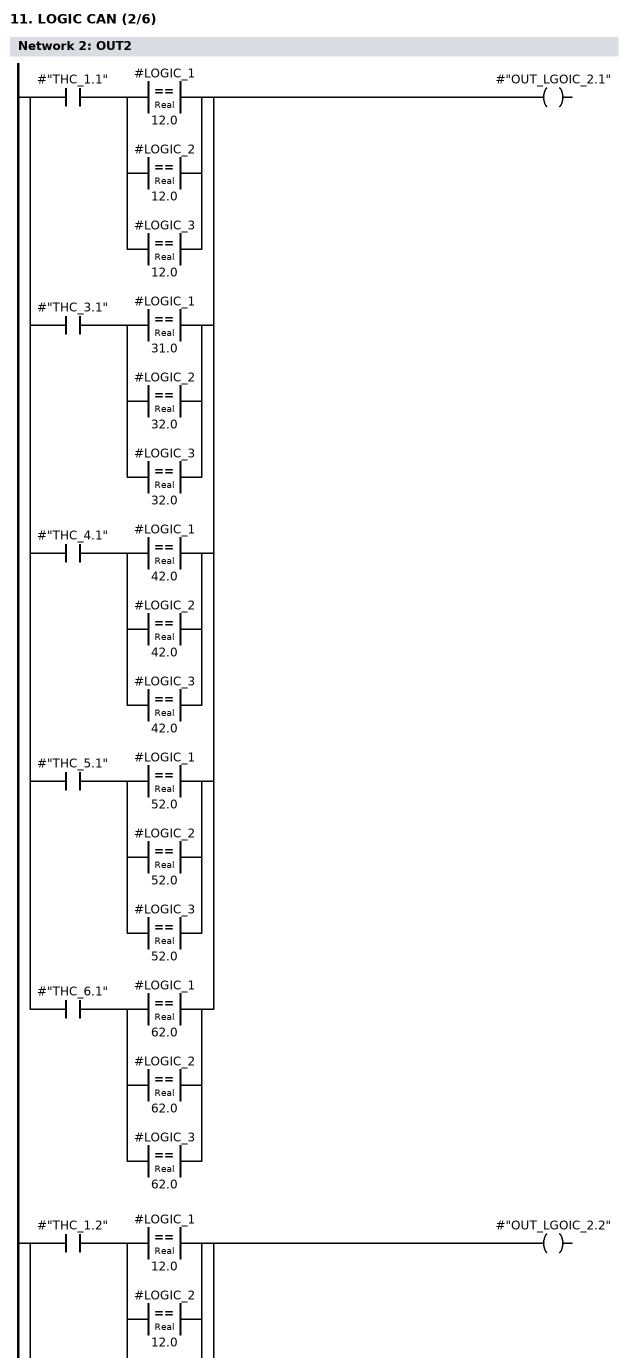
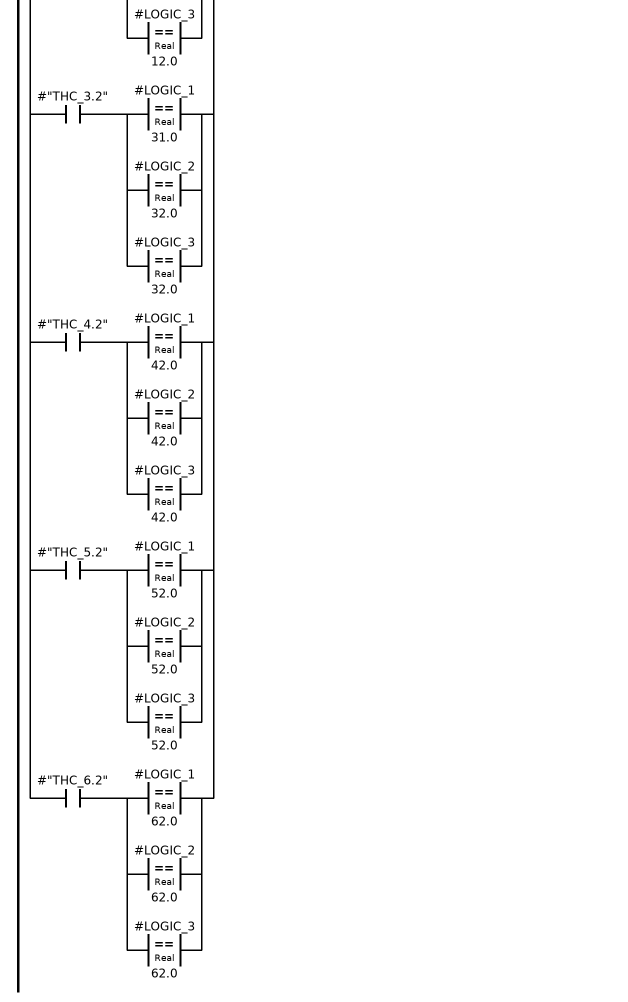
   RUNG wire#powerrail
      Contact( #"THC_1.1" )
      wire#w1
      { S7_Templates := "SrcType := Real" } EQ_Contact(in1 := #LOGIC_1, in2 := 12.0)
      wire#w2
      Coil( #"OUT_LGOIC_2.1" )
   END_RUNG
   RUNG wire#w1
      { S7_Templates := "SrcType := Real" } EQ_Contact(in1 := #LOGIC_2, in2 := 12.0)
   END_RUNG wire#w2
   RUNG wire#w1
      { S7_Templates := "SrcType := Real" } EQ_Contact(in1 := #LOGIC_3, in2 := 12.0)
   END_RUNG wire#w2
   RUNG wire#powerrail
      Contact( #"THC_3.1" )
      wire#w3
      { S7_Templates := "SrcType := Real" } EQ_Contact(in1 := #LOGIC_1, in2 := 31.0)
   END_RUNG wire#w2
   RUNG wire#w3
      { S7_Templates := "SrcType := Real" } EQ_Contact(in1 := #LOGIC_2, in2 := 32.0)
   END_RUNG wire#w2
   RUNG wire#w3
      { S7_Templates := "SrcType := Real" } EQ_Contact(in1 := #LOGIC_3, in2 := 32.0)
   END_RUNG wire#w2
   RUNG wire#powerrail
      Contact( #"THC_4.1" )
      wire#w4
      { S7_Templates := "SrcType := Real" } EQ_Contact(in1 := #LOGIC_1, in2 := 42.0)
   END_RUNG wire#w2
   RUNG wire#w4
      { S7_Templates := "SrcType := Real" } EQ_Contact(in1 := #LOGIC_2, in2 := 42.0)
   END_RUNG wire#w2
   RUNG wire#w4
      { S7_Templates := "SrcType := Real" } EQ_Contact(in1 := #LOGIC_3, in2 := 42.0)
   END_RUNG wire#w2
   RUNG wire#powerrail
      Contact( #"THC_5.1" )
      wire#w5
      { S7_Templates := "SrcType := Real" } EQ_Contact(in1 := #LOGIC_1, in2 := 52.0)
   END_RUNG wire#w2
   RUNG wire#w5
      { S7_Templates := "SrcType := Real" } EQ_Contact(in1 := #LOGIC_2, in2 := 52.0)
   END_RUNG wire#w2
   RUNG wire#w5
      { S7_Templates := "SrcType := Real" } EQ_Contact(in1 := #LOGIC_3, in2 := 52.0)
   END_RUNG wire#w2
   RUNG wire#powerrail
      Contact( #"THC_6.1" )
      wire#w6
      { S7_Templates := "SrcType := Real" } EQ_Contact(in1 := #LOGIC_1, in2 := 62.0)
   END_RUNG wire#w2
   RUNG wire#w6
      { S7_Templates := "SrcType := Real" } EQ_Contact(in1 := #LOGIC_2, in2 := 62.0)
   END_RUNG wire#w2
   RUNG wire#w6
      { S7_Templates := "SrcType := Real" } EQ_Contact(in1 := #LOGIC_3, in2 := 62.0)
   END_RUNG wire#w2
   RUNG wire#powerrail
      Contact( #"THC_1.2" )
      wire#w7
      { S7_Templates := "SrcType := Real" } EQ_Contact(in1 := #LOGIC_1, in2 := 12.0)
      wire#w8
      Coil( #"OUT_LGOIC_2.2" )
   END_RUNG
   RUNG wire#w7
      { S7_Templates := "SrcType := Real" } EQ_Contact(in1 := #LOGIC_2, in2 := 12.0)
   END_RUNG wire#w8
   RUNG wire#w7
      { S7_Templates := "SrcType := Real" } EQ_Contact(in1 := #LOGIC_3, in2 := 12.0)
   END_RUNG wire#w8
   RUNG wire#powerrail
      Contact( #"THC_3.2" )
      wire#w9
      { S7_Templates := "SrcType := Real" } EQ_Contact(in1 := #LOGIC_1, in2 := 31.0)
   END_RUNG wire#w8
   RUNG wire#w9
      { S7_Templates := "SrcType := Real" } EQ_Contact(in1 := #LOGIC_2, in2 := 32.0)
   END_RUNG wire#w8
   RUNG wire#w9
      { S7_Templates := "SrcType := Real" } EQ_Contact(in1 := #LOGIC_3, in2 := 32.0)
   END_RUNG wire#w8
   RUNG wire#powerrail
      Contact( #"THC_4.2" )
      wire#w10
      { S7_Templates := "SrcType := Real" } EQ_Contact(in1 := #LOGIC_1, in2 := 42.0)
   END_RUNG wire#w8
   RUNG wire#w10
      { S7_Templates := "SrcType := Real" } EQ_Contact(in1 := #LOGIC_2, in2 := 42.0)
   END_RUNG wire#w8
   RUNG wire#w10
      { S7_Templates := "SrcType := Real" } EQ_Contact(in1 := #LOGIC_3, in2 := 42.0)
   END_RUNG wire#w8
   RUNG wire#powerrail
      Contact( #"THC_5.2" )
      wire#w11
      { S7_Templates := "SrcType := Real" } EQ_Contact(in1 := #LOGIC_1, in2 := 52.0)
   END_RUNG wire#w8
   RUNG wire#w11
      { S7_Templates := "SrcType := Real" } EQ_Contact(in1 := #LOGIC_2, in2 := 52.0)
   END_RUNG wire#w8
   RUNG wire#w11
      { S7_Templates := "SrcType := Real" } EQ_Contact(in1 := #LOGIC_3, in2 := 52.0)
   END_RUNG wire#w8
   RUNG wire#powerrail
      Contact( #"THC_6.2" )
      wire#w12
      { S7_Templates := "SrcType := Real" } EQ_Contact(in1 := #LOGIC_1, in2 := 62.0)
   END_RUNG wire#w8
   RUNG wire#w12
      { S7_Templates := "SrcType := Real" } EQ_Contact(in1 := #LOGIC_2, in2 := 62.0)
   END_RUNG wire#w8
   RUNG wire#w12
      { S7_Templates := "SrcType := Real" } EQ_Contact(in1 := #LOGIC_3, in2 := 62.0)
   END_RUNG wire#w8
   // the same network as SCL:
   #"OUT_LGOIC_2.1" := (#"THC_1.1" AND ((#LOGIC_1 = 12.0) OR (#LOGIC_2 = 12.0) OR (#LOGIC_3 = 12.0))) OR (#"THC_3.1" AND ((#LOGIC_1 = 31.0) OR (#LOGIC_2 = 32.0) OR (#LOGIC_3 = 32.0))) OR (#"THC_4.1" AND ((#LOGIC_1 = 42.0) OR (#LOGIC_2 = 42.0) OR (#LOGIC_3 = 42.0))) OR (#"THC_5.1" AND ((#LOGIC_1 = 52.0) OR (#LOGIC_2 = 52.0) OR (#LOGIC_3 = 52.0))) OR (#"THC_6.1" AND ((#LOGIC_1 = 62.0) OR (#LOGIC_2 = 62.0) OR (#LOGIC_3 = 62.0)));
   #"OUT_LGOIC_2.2" := (#"THC_1.2" AND ((#LOGIC_1 = 12.0) OR (#LOGIC_2 = 12.0) OR (#LOGIC_3 = 12.0))) OR (#"THC_3.2" AND ((#LOGIC_1 = 31.0) OR (#LOGIC_2 = 32.0) OR (#LOGIC_3 = 32.0))) OR (#"THC_4.2" AND ((#LOGIC_1 = 42.0) OR (#LOGIC_2 = 42.0) OR (#LOGIC_3 = 42.0))) OR (#"THC_5.2" AND ((#LOGIC_1 = 52.0) OR (#LOGIC_2 = 52.0) OR (#LOGIC_3 = 52.0))) OR (#"THC_6.2" AND ((#LOGIC_1 = 62.0) OR (#LOGIC_2 = 62.0) OR (#LOGIC_3 = 62.0)));
END_REGION

REGION Network 3: OUT3
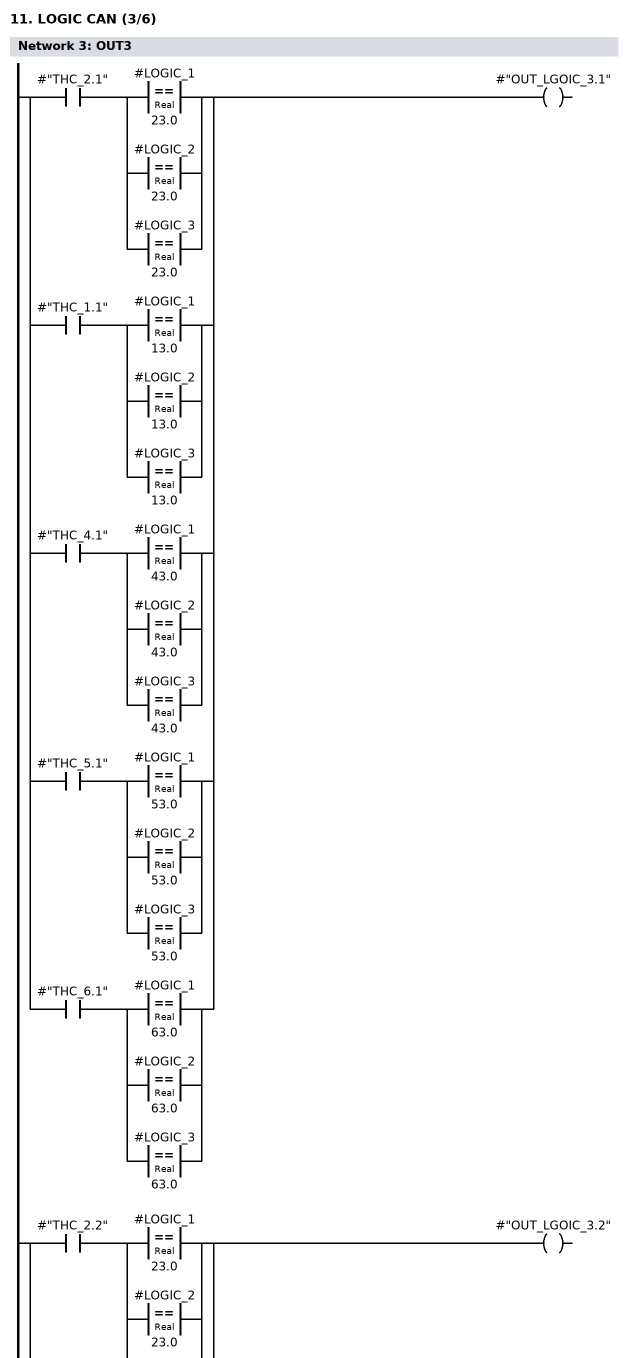
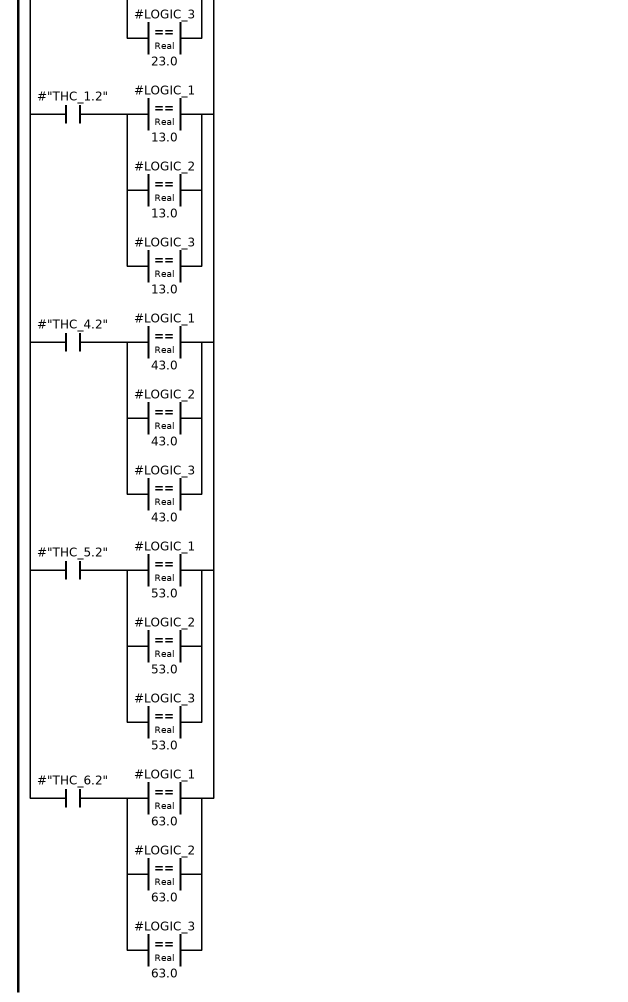
   RUNG wire#powerrail
      Contact( #"THC_2.1" )
      wire#w1
      { S7_Templates := "SrcType := Real" } EQ_Contact(in1 := #LOGIC_1, in2 := 23.0)
      wire#w2
      Coil( #"OUT_LGOIC_3.1" )
   END_RUNG
   RUNG wire#w1
      { S7_Templates := "SrcType := Real" } EQ_Contact(in1 := #LOGIC_2, in2 := 23.0)
   END_RUNG wire#w2
   RUNG wire#w1
      { S7_Templates := "SrcType := Real" } EQ_Contact(in1 := #LOGIC_3, in2 := 23.0)
   END_RUNG wire#w2
   RUNG wire#powerrail
      Contact( #"THC_1.1" )
      wire#w3
      { S7_Templates := "SrcType := Real" } EQ_Contact(in1 := #LOGIC_1, in2 := 13.0)
   END_RUNG wire#w2
   RUNG wire#w3
      { S7_Templates := "SrcType := Real" } EQ_Contact(in1 := #LOGIC_2, in2 := 13.0)
   END_RUNG wire#w2
   RUNG wire#w3
      { S7_Templates := "SrcType := Real" } EQ_Contact(in1 := #LOGIC_3, in2 := 13.0)
   END_RUNG wire#w2
   RUNG wire#powerrail
      Contact( #"THC_4.1" )
      wire#w4
      { S7_Templates := "SrcType := Real" } EQ_Contact(in1 := #LOGIC_1, in2 := 43.0)
   END_RUNG wire#w2
   RUNG wire#w4
      { S7_Templates := "SrcType := Real" } EQ_Contact(in1 := #LOGIC_2, in2 := 43.0)
   END_RUNG wire#w2
   RUNG wire#w4
      { S7_Templates := "SrcType := Real" } EQ_Contact(in1 := #LOGIC_3, in2 := 43.0)
   END_RUNG wire#w2
   RUNG wire#powerrail
      Contact( #"THC_5.1" )
      wire#w5
      { S7_Templates := "SrcType := Real" } EQ_Contact(in1 := #LOGIC_1, in2 := 53.0)
   END_RUNG wire#w2
   RUNG wire#w5
      { S7_Templates := "SrcType := Real" } EQ_Contact(in1 := #LOGIC_2, in2 := 53.0)
   END_RUNG wire#w2
   RUNG wire#w5
      { S7_Templates := "SrcType := Real" } EQ_Contact(in1 := #LOGIC_3, in2 := 53.0)
   END_RUNG wire#w2
   RUNG wire#powerrail
      Contact( #"THC_6.1" )
      wire#w6
      { S7_Templates := "SrcType := Real" } EQ_Contact(in1 := #LOGIC_1, in2 := 63.0)
   END_RUNG wire#w2
   RUNG wire#w6
      { S7_Templates := "SrcType := Real" } EQ_Contact(in1 := #LOGIC_2, in2 := 63.0)
   END_RUNG wire#w2
   RUNG wire#w6
      { S7_Templates := "SrcType := Real" } EQ_Contact(in1 := #LOGIC_3, in2 := 63.0)
   END_RUNG wire#w2
   RUNG wire#powerrail
      Contact( #"THC_2.2" )
      wire#w7
      { S7_Templates := "SrcType := Real" } EQ_Contact(in1 := #LOGIC_1, in2 := 23.0)
      wire#w8
      Coil( #"OUT_LGOIC_3.2" )
   END_RUNG
   RUNG wire#w7
      { S7_Templates := "SrcType := Real" } EQ_Contact(in1 := #LOGIC_2, in2 := 23.0)
   END_RUNG wire#w8
   RUNG wire#w7
      { S7_Templates := "SrcType := Real" } EQ_Contact(in1 := #LOGIC_3, in2 := 23.0)
   END_RUNG wire#w8
   RUNG wire#powerrail
      Contact( #"THC_1.2" )
      wire#w9
      { S7_Templates := "SrcType := Real" } EQ_Contact(in1 := #LOGIC_1, in2 := 13.0)
   END_RUNG wire#w8
   RUNG wire#w9
      { S7_Templates := "SrcType := Real" } EQ_Contact(in1 := #LOGIC_2, in2 := 13.0)
   END_RUNG wire#w8
   RUNG wire#w9
      { S7_Templates := "SrcType := Real" } EQ_Contact(in1 := #LOGIC_3, in2 := 13.0)
   END_RUNG wire#w8
   RUNG wire#powerrail
      Contact( #"THC_4.2" )
      wire#w10
      { S7_Templates := "SrcType := Real" } EQ_Contact(in1 := #LOGIC_1, in2 := 43.0)
   END_RUNG wire#w8
   RUNG wire#w10
      { S7_Templates := "SrcType := Real" } EQ_Contact(in1 := #LOGIC_2, in2 := 43.0)
   END_RUNG wire#w8
   RUNG wire#w10
      { S7_Templates := "SrcType := Real" } EQ_Contact(in1 := #LOGIC_3, in2 := 43.0)
   END_RUNG wire#w8
   RUNG wire#powerrail
      Contact( #"THC_5.2" )
      wire#w11
      { S7_Templates := "SrcType := Real" } EQ_Contact(in1 := #LOGIC_1, in2 := 53.0)
   END_RUNG wire#w8
   RUNG wire#w11
      { S7_Templates := "SrcType := Real" } EQ_Contact(in1 := #LOGIC_2, in2 := 53.0)
   END_RUNG wire#w8
   RUNG wire#w11
      { S7_Templates := "SrcType := Real" } EQ_Contact(in1 := #LOGIC_3, in2 := 53.0)
   END_RUNG wire#w8
   RUNG wire#powerrail
      Contact( #"THC_6.2" )
      wire#w12
      { S7_Templates := "SrcType := Real" } EQ_Contact(in1 := #LOGIC_1, in2 := 63.0)
   END_RUNG wire#w8
   RUNG wire#w12
      { S7_Templates := "SrcType := Real" } EQ_Contact(in1 := #LOGIC_2, in2 := 63.0)
   END_RUNG wire#w8
   RUNG wire#w12
      { S7_Templates := "SrcType := Real" } EQ_Contact(in1 := #LOGIC_3, in2 := 63.0)
   END_RUNG wire#w8
   // the same network as SCL:
   #"OUT_LGOIC_3.1" := (#"THC_2.1" AND ((#LOGIC_1 = 23.0) OR (#LOGIC_2 = 23.0) OR (#LOGIC_3 = 23.0))) OR (#"THC_1.1" AND ((#LOGIC_1 = 13.0) OR (#LOGIC_2 = 13.0) OR (#LOGIC_3 = 13.0))) OR (#"THC_4.1" AND ((#LOGIC_1 = 43.0) OR (#LOGIC_2 = 43.0) OR (#LOGIC_3 = 43.0))) OR (#"THC_5.1" AND ((#LOGIC_1 = 53.0) OR (#LOGIC_2 = 53.0) OR (#LOGIC_3 = 53.0))) OR (#"THC_6.1" AND ((#LOGIC_1 = 63.0) OR (#LOGIC_2 = 63.0) OR (#LOGIC_3 = 63.0)));
   #"OUT_LGOIC_3.2" := (#"THC_2.2" AND ((#LOGIC_1 = 23.0) OR (#LOGIC_2 = 23.0) OR (#LOGIC_3 = 23.0))) OR (#"THC_1.2" AND ((#LOGIC_1 = 13.0) OR (#LOGIC_2 = 13.0) OR (#LOGIC_3 = 13.0))) OR (#"THC_4.2" AND ((#LOGIC_1 = 43.0) OR (#LOGIC_2 = 43.0) OR (#LOGIC_3 = 43.0))) OR (#"THC_5.2" AND ((#LOGIC_1 = 53.0) OR (#LOGIC_2 = 53.0) OR (#LOGIC_3 = 53.0))) OR (#"THC_6.2" AND ((#LOGIC_1 = 63.0) OR (#LOGIC_2 = 63.0) OR (#LOGIC_3 = 63.0)));
END_REGION

